// TIA Portal V17 export
// export: Created 2025-06-20T11:17:40.9768226Z, ExportSetting WithDefaults, DisplayName Totally Integrated Automation Portal, DisplayVersion V17 Update 8, DisplayName TIA Portal Openness, DisplayVersion V17 Update 8, DisplayName TIA Portal Version Control Interface, DisplayVersion V17, DisplayName SINAMICS Startdrive Advanced, DisplayVersion V17 SP2, DisplayName SINAMICS Startdrive G110M, G120, G120C, G120D, G120P, G115D, DisplayVersion V17 SP2, DisplayName SINAMICS Startdrive G130, G150, S120, S150, SINAMICS MV, S210, DisplayVersion V17 SP2, DisplayName STEP 7 Professional, DisplayVersion V17 Update 8, DisplayName SINUMERIK ONE STEP 7 Toolbox, DisplayVersion V17 Update 12, DisplayName SINUMERIK ONE PLC Basic Program Plus, DisplayVersion V17 Update 12, DisplayName SINUMERIK 840D sl STEP 7 Toolbox, DisplayVersion V17 Update 12, DisplayName STEP 7 Safety, DisplayVersion V17 Update 6, DisplayName WinCC Advanced, DisplayVersion V17 Update 8
FUNCTION "FC16017_METHOD_CALLS_U3_MEAS_STA_MEAS_N" : Void   // FC16017, LAD
{ S7_Optimized_Access := 'FALSE' }
VERSION : 0.1
// stored: AutoNumber false, IsIECCheckEnabled false, SetENOAutomatically false, UDAEnableTagReadback false
   VAR_TEMP
      AUX_WSTRING_PART_ID_MEAS_STA : WString;
      AUX_WCHARS : Array[0..63] of WChar;
      index : Int;
      AUX_ALARMS : Bool;
      STATUS_BLKMOV : Int;   // STATUS BLKMOV
      ZERO : Int;
   END_VAR
   VAR CONSTANT
      VERSIONS_MAJOR : UInt := 2;
      VERSIONS_MINOR : UInt;
      FC_NUMBER : DInt := 16017;
   END_VAR
   VAR_TEMP   // added for the SCL form of the ladder/FBD networks
      _w1 : Bool;
      _w2 : Bool;
   END_VAR
BEGIN

REGION Network 1: ZERO
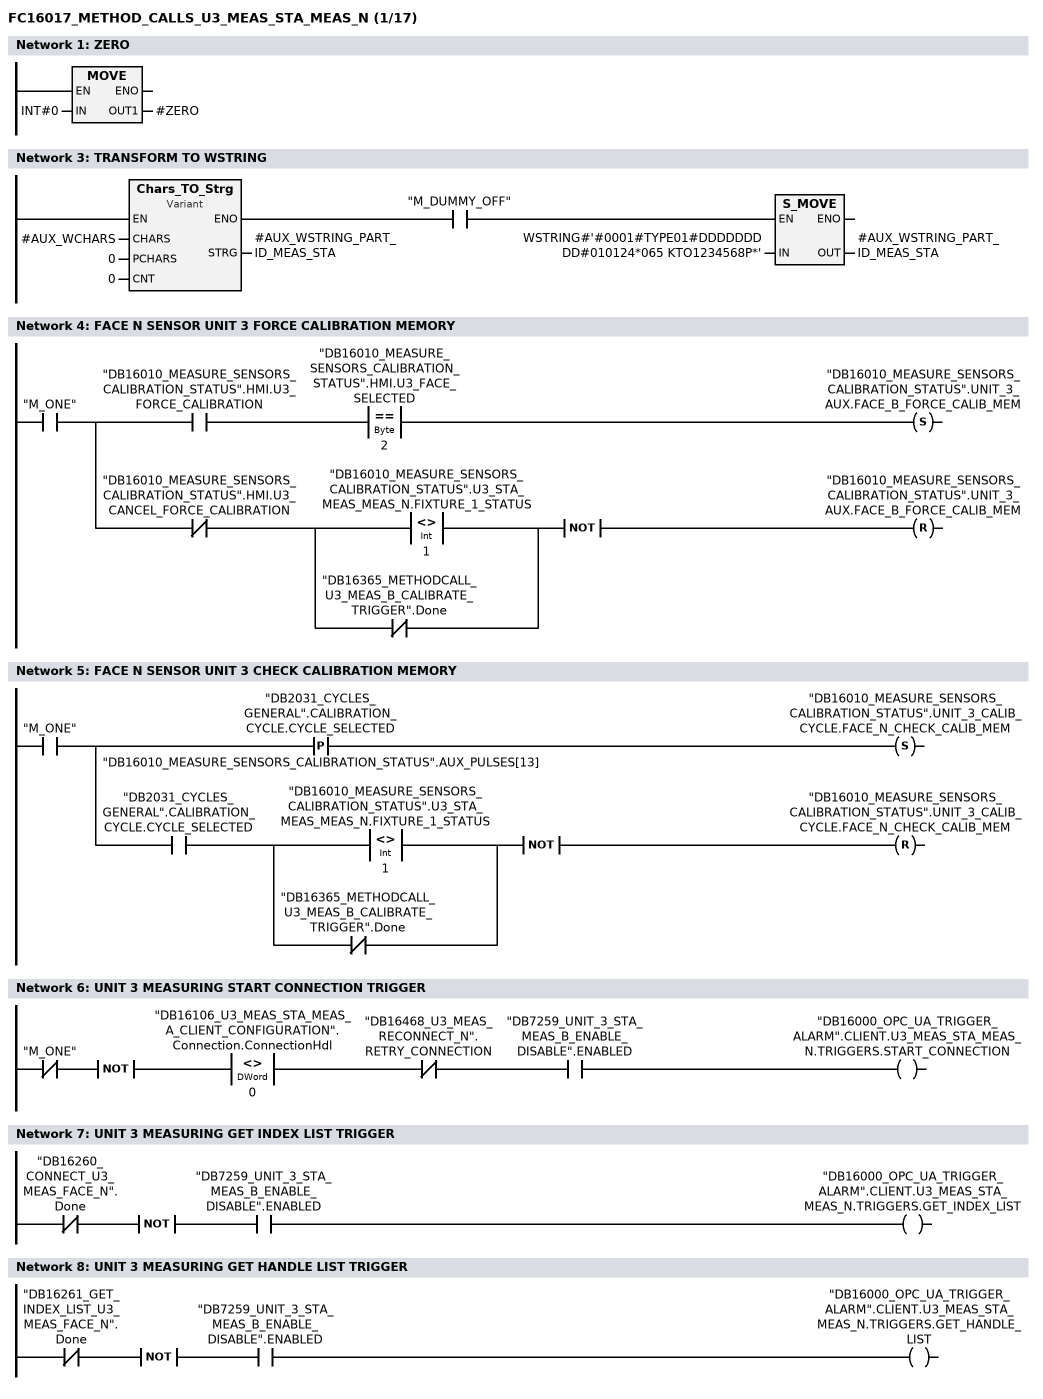
   RUNG wire#powerrail
      { S7_GenerateENO := "TRUE" } Move(in := INT#0, out1 => #ZERO)
   END_RUNG
   // the same network as SCL:
   #ZERO := INT#0;
END_REGION

REGION Network 2 (SCL): TRANSFORM TO WCHARS
   FOR #index := 0 TO 63 DO
       #AUX_WCHARS[#index] := CHAR_TO_WCHAR("DB8000_PART_STATUS".UNIT_3.FIXTURE_1.PART_A.PART_ID[#index]);
   END_FOR;
END_REGION

REGION Network 3: TRANSFORM TO WSTRING
   RUNG wire#powerrail
      { S7_Templates := "[ptr_type := Variant, str_type := WString]" } Chars_TO_Strg(Chars := #AUX_WCHARS, pChars := 0, Cnt := 0, Strg => #AUX_WSTRING_PART_ID_MEAS_STA)
      Contact( "M_DUMMY_OFF" )
      S_Move(in := WSTRING#'#0001#TYPE01#DDDDDDDDD#010124*065 KTO1234568P*', out => #AUX_WSTRING_PART_ID_MEAS_STA)
   END_RUNG
   // the same network as SCL:
   Chars_TO_Strg(Chars := #AUX_WCHARS,
                 pChars := 0,
                 Cnt := 0,
                 Strg => #AUX_WSTRING_PART_ID_MEAS_STA,
                 ENO => #_w1);
   IF #_w1 AND "M_DUMMY_OFF" THEN
       #AUX_WSTRING_PART_ID_MEAS_STA := WSTRING#'#0001#TYPE01#DDDDDDDDD#010124*065 KTO1234568P*';
   END_IF;
END_REGION

REGION Network 4: FACE N SENSOR UNIT 3 FORCE CALIBRATION MEMORY
   RUNG wire#powerrail
      Contact( "M_ONE" )
      wire#w1
      Contact( "DB16010_MEASURE_SENSORS_CALIBRATION_STATUS".HMI.U3_FORCE_CALIBRATION )
      { S7_Templates := "SrcType := Byte" } EQ_Contact(in1 := "DB16010_MEASURE_SENSORS_CALIBRATION_STATUS".HMI.U3_FACE_SELECTED, in2 := 2)
      S_Coil( "DB16010_MEASURE_SENSORS_CALIBRATION_STATUS".UNIT_3_AUX.FACE_B_FORCE_CALIB_MEM )
   END_RUNG
   RUNG wire#w1
      I_Contact( "DB16010_MEASURE_SENSORS_CALIBRATION_STATUS".HMI.U3_CANCEL_FORCE_CALIBRATION )
      wire#w2
      { S7_Templates := "SrcType := Int" } NE_Contact(in1 := "DB16010_MEASURE_SENSORS_CALIBRATION_STATUS".U3_STA_MEAS_MEAS_N.FIXTURE_1_STATUS, in2 := 1)
      wire#w3
      Not()
      R_Coil( "DB16010_MEASURE_SENSORS_CALIBRATION_STATUS".UNIT_3_AUX.FACE_B_FORCE_CALIB_MEM )
   END_RUNG
   RUNG wire#w2
      I_Contact( "DB16365_METHODCALL_U3_MEAS_B_CALIBRATE_TRIGGER".Done )
   END_RUNG wire#w3
   // the same network as SCL:
   IF "M_ONE" AND "DB16010_MEASURE_SENSORS_CALIBRATION_STATUS".HMI.U3_FORCE_CALIBRATION AND ("DB16010_MEASURE_SENSORS_CALIBRATION_STATUS".HMI.U3_FACE_SELECTED = 2) THEN
       "DB16010_MEASURE_SENSORS_CALIBRATION_STATUS".UNIT_3_AUX.FACE_B_FORCE_CALIB_MEM := TRUE;
   END_IF;
   IF NOT ("M_ONE" AND NOT "DB16010_MEASURE_SENSORS_CALIBRATION_STATUS".HMI.U3_CANCEL_FORCE_CALIBRATION AND (("DB16010_MEASURE_SENSORS_CALIBRATION_STATUS".U3_STA_MEAS_MEAS_N.FIXTURE_1_STATUS <> 1) OR NOT "DB16365_METHODCALL_U3_MEAS_B_CALIBRATE_TRIGGER".Done)) THEN
       "DB16010_MEASURE_SENSORS_CALIBRATION_STATUS".UNIT_3_AUX.FACE_B_FORCE_CALIB_MEM := FALSE;
   END_IF;
END_REGION

REGION Network 5: FACE N SENSOR UNIT 3 CHECK CALIBRATION MEMORY
   RUNG wire#powerrail
      Contact( "M_ONE" )
      wire#w1
      P_Contact(operand := "DB2031_CYCLES_GENERAL".CALIBRATION_CYCLE.CYCLE_SELECTED, bit := "DB16010_MEASURE_SENSORS_CALIBRATION_STATUS".AUX_PULSES[13])
      S_Coil( "DB16010_MEASURE_SENSORS_CALIBRATION_STATUS".UNIT_3_CALIB_CYCLE.FACE_N_CHECK_CALIB_MEM )
   END_RUNG
   RUNG wire#w1
      Contact( "DB2031_CYCLES_GENERAL".CALIBRATION_CYCLE.CYCLE_SELECTED )
      wire#w2
      { S7_Templates := "SrcType := Int" } NE_Contact(in1 := "DB16010_MEASURE_SENSORS_CALIBRATION_STATUS".U3_STA_MEAS_MEAS_N.FIXTURE_1_STATUS, in2 := 1)
      wire#w3
      Not()
      R_Coil( "DB16010_MEASURE_SENSORS_CALIBRATION_STATUS".UNIT_3_CALIB_CYCLE.FACE_N_CHECK_CALIB_MEM )
   END_RUNG
   RUNG wire#w2
      I_Contact( "DB16365_METHODCALL_U3_MEAS_B_CALIBRATE_TRIGGER".Done )
   END_RUNG wire#w3
   // the same network as SCL:
   #_w1 := "M_ONE" AND "DB2031_CYCLES_GENERAL".CALIBRATION_CYCLE.CYCLE_SELECTED AND NOT "DB16010_MEASURE_SENSORS_CALIBRATION_STATUS".AUX_PULSES[13];   // rising edge of "DB2031_CYCLES_GENERAL".CALIBRATION_CYCLE.CYCLE_SELECTED
   "DB16010_MEASURE_SENSORS_CALIBRATION_STATUS".AUX_PULSES[13] := "DB2031_CYCLES_GENERAL".CALIBRATION_CYCLE.CYCLE_SELECTED;
   IF #_w1 THEN
       "DB16010_MEASURE_SENSORS_CALIBRATION_STATUS".UNIT_3_CALIB_CYCLE.FACE_N_CHECK_CALIB_MEM := TRUE;
   END_IF;
   IF NOT ("M_ONE" AND "DB2031_CYCLES_GENERAL".CALIBRATION_CYCLE.CYCLE_SELECTED AND (("DB16010_MEASURE_SENSORS_CALIBRATION_STATUS".U3_STA_MEAS_MEAS_N.FIXTURE_1_STATUS <> 1) OR NOT "DB16365_METHODCALL_U3_MEAS_B_CALIBRATE_TRIGGER".Done)) THEN
       "DB16010_MEASURE_SENSORS_CALIBRATION_STATUS".UNIT_3_CALIB_CYCLE.FACE_N_CHECK_CALIB_MEM := FALSE;
   END_IF;
END_REGION

REGION Network 6: UNIT 3 MEASURING START CONNECTION TRIGGER
   RUNG wire#powerrail
      I_Contact( "M_ONE" )
      Not()
      { S7_Templates := "SrcType := DWord" } NE_Contact(in1 := "DB16106_U3_MEAS_STA_MEAS_A_CLIENT_CONFIGURATION".Connection.ConnectionHdl, in2 := 0)
      I_Contact( "DB16468_U3_MEAS_RECONNECT_N".RETRY_CONNECTION )
      Contact( "DB7259_UNIT_3_STA_MEAS_B_ENABLE_DISABLE".ENABLED )
      Coil( "DB16000_OPC_UA_TRIGGER_ALARM".CLIENT.U3_MEAS_STA_MEAS_N.TRIGGERS.START_CONNECTION )
   END_RUNG
   // the same network as SCL:
   "DB16000_OPC_UA_TRIGGER_ALARM".CLIENT.U3_MEAS_STA_MEAS_N.TRIGGERS.START_CONNECTION := NOT (NOT "M_ONE") AND ("DB16106_U3_MEAS_STA_MEAS_A_CLIENT_CONFIGURATION".Connection.ConnectionHdl <> 0) AND NOT "DB16468_U3_MEAS_RECONNECT_N".RETRY_CONNECTION AND "DB7259_UNIT_3_STA_MEAS_B_ENABLE_DISABLE".ENABLED;
END_REGION

REGION Network 7: UNIT 3 MEASURING GET INDEX LIST TRIGGER
   RUNG wire#powerrail
      I_Contact( "DB16260_CONNECT_U3_MEAS_FACE_N".Done )
      Not()
      Contact( "DB7259_UNIT_3_STA_MEAS_B_ENABLE_DISABLE".ENABLED )
      Coil( "DB16000_OPC_UA_TRIGGER_ALARM".CLIENT.U3_MEAS_STA_MEAS_N.TRIGGERS.GET_INDEX_LIST )
   END_RUNG
   // the same network as SCL:
   "DB16000_OPC_UA_TRIGGER_ALARM".CLIENT.U3_MEAS_STA_MEAS_N.TRIGGERS.GET_INDEX_LIST := NOT (NOT "DB16260_CONNECT_U3_MEAS_FACE_N".Done) AND "DB7259_UNIT_3_STA_MEAS_B_ENABLE_DISABLE".ENABLED;
END_REGION

REGION Network 8: UNIT 3 MEASURING GET HANDLE LIST TRIGGER
   RUNG wire#powerrail
      I_Contact( "DB16261_GET_INDEX_LIST_U3_MEAS_FACE_N".Done )
      Not()
      Contact( "DB7259_UNIT_3_STA_MEAS_B_ENABLE_DISABLE".ENABLED )
      Coil( "DB16000_OPC_UA_TRIGGER_ALARM".CLIENT.U3_MEAS_STA_MEAS_N.TRIGGERS.GET_HANDLE_LIST )
   END_RUNG
   // the same network as SCL:
   "DB16000_OPC_UA_TRIGGER_ALARM".CLIENT.U3_MEAS_STA_MEAS_N.TRIGGERS.GET_HANDLE_LIST := NOT (NOT "DB16261_GET_INDEX_LIST_U3_MEAS_FACE_N".Done) AND "DB7259_UNIT_3_STA_MEAS_B_ENABLE_DISABLE".ENABLED;
END_REGION

REGION Network 9: UNIT 3 MEASURING GET METHOD LIST TRIGGER
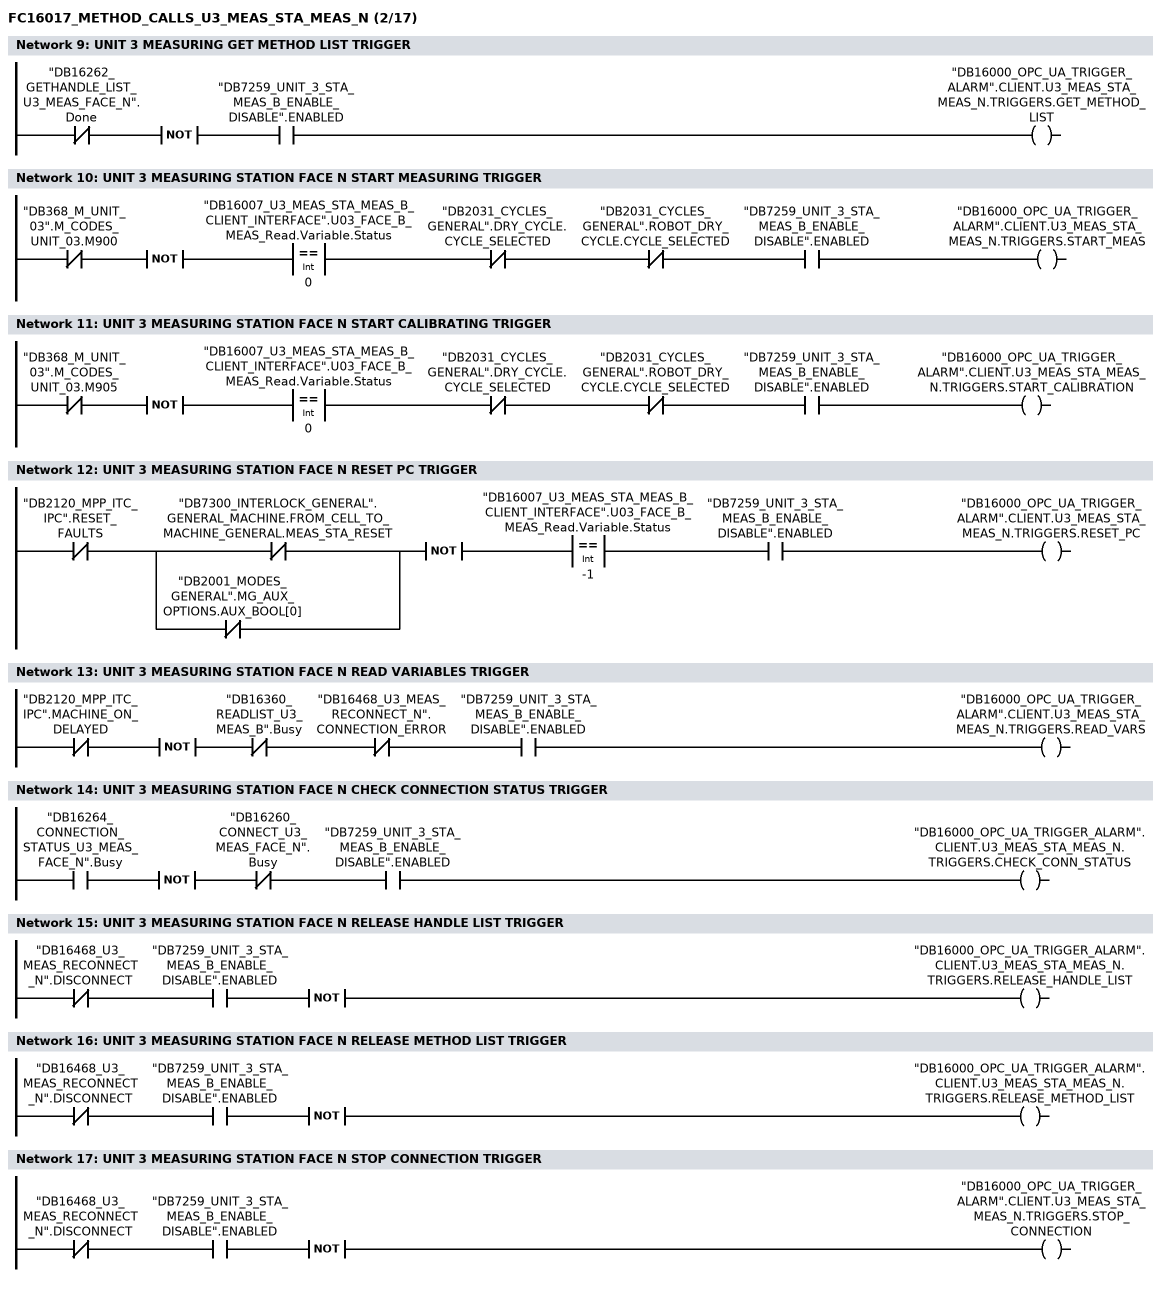
   RUNG wire#powerrail
      I_Contact( "DB16262_GETHANDLE_LIST_U3_MEAS_FACE_N".Done )
      Not()
      Contact( "DB7259_UNIT_3_STA_MEAS_B_ENABLE_DISABLE".ENABLED )
      Coil( "DB16000_OPC_UA_TRIGGER_ALARM".CLIENT.U3_MEAS_STA_MEAS_N.TRIGGERS.GET_METHOD_LIST )
   END_RUNG
   // the same network as SCL:
   "DB16000_OPC_UA_TRIGGER_ALARM".CLIENT.U3_MEAS_STA_MEAS_N.TRIGGERS.GET_METHOD_LIST := NOT (NOT "DB16262_GETHANDLE_LIST_U3_MEAS_FACE_N".Done) AND "DB7259_UNIT_3_STA_MEAS_B_ENABLE_DISABLE".ENABLED;
END_REGION

REGION Network 10: UNIT 3 MEASURING STATION FACE N START MEASURING TRIGGER
   RUNG wire#powerrail
      I_Contact( "DB368_M_UNIT_03".M_CODES_UNIT_03.M900 )
      Not()
      { S7_Templates := "SrcType := Int" } EQ_Contact(in1 := "DB16007_U3_MEAS_STA_MEAS_B_CLIENT_INTERFACE".U03_FACE_B_MEAS_Read.Variable.Status, in2 := 0)
      I_Contact( "DB2031_CYCLES_GENERAL".DRY_CYCLE.CYCLE_SELECTED )
      I_Contact( "DB2031_CYCLES_GENERAL".ROBOT_DRY_CYCLE.CYCLE_SELECTED )
      Contact( "DB7259_UNIT_3_STA_MEAS_B_ENABLE_DISABLE".ENABLED )
      Coil( "DB16000_OPC_UA_TRIGGER_ALARM".CLIENT.U3_MEAS_STA_MEAS_N.TRIGGERS.START_MEAS )
   END_RUNG
   // the same network as SCL:
   "DB16000_OPC_UA_TRIGGER_ALARM".CLIENT.U3_MEAS_STA_MEAS_N.TRIGGERS.START_MEAS := NOT (NOT "DB368_M_UNIT_03".M_CODES_UNIT_03.M900) AND ("DB16007_U3_MEAS_STA_MEAS_B_CLIENT_INTERFACE".U03_FACE_B_MEAS_Read.Variable.Status = 0) AND NOT "DB2031_CYCLES_GENERAL".DRY_CYCLE.CYCLE_SELECTED AND NOT "DB2031_CYCLES_GENERAL".ROBOT_DRY_CYCLE.CYCLE_SELECTED AND "DB7259_UNIT_3_STA_MEAS_B_ENABLE_DISABLE".ENABLED;
END_REGION

REGION Network 11: UNIT 3 MEASURING STATION FACE N START CALIBRATING TRIGGER
   RUNG wire#powerrail
      I_Contact( "DB368_M_UNIT_03".M_CODES_UNIT_03.M905 )
      Not()
      { S7_Templates := "SrcType := Int" } EQ_Contact(in1 := "DB16007_U3_MEAS_STA_MEAS_B_CLIENT_INTERFACE".U03_FACE_B_MEAS_Read.Variable.Status, in2 := 0)
      I_Contact( "DB2031_CYCLES_GENERAL".DRY_CYCLE.CYCLE_SELECTED )
      I_Contact( "DB2031_CYCLES_GENERAL".ROBOT_DRY_CYCLE.CYCLE_SELECTED )
      Contact( "DB7259_UNIT_3_STA_MEAS_B_ENABLE_DISABLE".ENABLED )
      Coil( "DB16000_OPC_UA_TRIGGER_ALARM".CLIENT.U3_MEAS_STA_MEAS_N.TRIGGERS.START_CALIBRATION )
   END_RUNG
   // the same network as SCL:
   "DB16000_OPC_UA_TRIGGER_ALARM".CLIENT.U3_MEAS_STA_MEAS_N.TRIGGERS.START_CALIBRATION := NOT (NOT "DB368_M_UNIT_03".M_CODES_UNIT_03.M905) AND ("DB16007_U3_MEAS_STA_MEAS_B_CLIENT_INTERFACE".U03_FACE_B_MEAS_Read.Variable.Status = 0) AND NOT "DB2031_CYCLES_GENERAL".DRY_CYCLE.CYCLE_SELECTED AND NOT "DB2031_CYCLES_GENERAL".ROBOT_DRY_CYCLE.CYCLE_SELECTED AND "DB7259_UNIT_3_STA_MEAS_B_ENABLE_DISABLE".ENABLED;
END_REGION

REGION Network 12: UNIT 3 MEASURING STATION FACE N RESET PC TRIGGER
   RUNG wire#powerrail
      I_Contact( "DB2120_MPP_ITC_IPC".RESET_FAULTS )
      wire#w1
      I_Contact( "DB7300_INTERLOCK_GENERAL".GENERAL_MACHINE.FROM_CELL_TO_MACHINE_GENERAL.MEAS_STA_RESET )
      wire#w2
      Not()
      { S7_Templates := "SrcType := Int" } EQ_Contact(in1 := "DB16007_U3_MEAS_STA_MEAS_B_CLIENT_INTERFACE".U03_FACE_B_MEAS_Read.Variable.Status, in2 := -1)
      Contact( "DB7259_UNIT_3_STA_MEAS_B_ENABLE_DISABLE".ENABLED )
      Coil( "DB16000_OPC_UA_TRIGGER_ALARM".CLIENT.U3_MEAS_STA_MEAS_N.TRIGGERS.RESET_PC )
   END_RUNG
   RUNG wire#w1
      I_Contact( "DB2001_MODES_GENERAL".MG_AUX_OPTIONS.AUX_BOOL[0] )
   END_RUNG wire#w2
   // the same network as SCL:
   "DB16000_OPC_UA_TRIGGER_ALARM".CLIENT.U3_MEAS_STA_MEAS_N.TRIGGERS.RESET_PC := NOT (NOT "DB2120_MPP_ITC_IPC".RESET_FAULTS AND (NOT "DB7300_INTERLOCK_GENERAL".GENERAL_MACHINE.FROM_CELL_TO_MACHINE_GENERAL.MEAS_STA_RESET OR NOT "DB2001_MODES_GENERAL".MG_AUX_OPTIONS.AUX_BOOL[0])) AND ("DB16007_U3_MEAS_STA_MEAS_B_CLIENT_INTERFACE".U03_FACE_B_MEAS_Read.Variable.Status = (-1)) AND "DB7259_UNIT_3_STA_MEAS_B_ENABLE_DISABLE".ENABLED;
END_REGION

REGION Network 13: UNIT 3 MEASURING STATION FACE N READ VARIABLES TRIGGER
   RUNG wire#powerrail
      I_Contact( "DB2120_MPP_ITC_IPC".MACHINE_ON_DELAYED )
      Not()
      I_Contact( "DB16360_READLIST_U3_MEAS_B".Busy )
      I_Contact( "DB16468_U3_MEAS_RECONNECT_N".CONNECTION_ERROR )
      Contact( "DB7259_UNIT_3_STA_MEAS_B_ENABLE_DISABLE".ENABLED )
      Coil( "DB16000_OPC_UA_TRIGGER_ALARM".CLIENT.U3_MEAS_STA_MEAS_N.TRIGGERS.READ_VARS )
   END_RUNG
   // the same network as SCL:
   "DB16000_OPC_UA_TRIGGER_ALARM".CLIENT.U3_MEAS_STA_MEAS_N.TRIGGERS.READ_VARS := NOT (NOT "DB2120_MPP_ITC_IPC".MACHINE_ON_DELAYED) AND NOT "DB16360_READLIST_U3_MEAS_B".Busy AND NOT "DB16468_U3_MEAS_RECONNECT_N".CONNECTION_ERROR AND "DB7259_UNIT_3_STA_MEAS_B_ENABLE_DISABLE".ENABLED;
END_REGION

REGION Network 14: UNIT 3 MEASURING STATION FACE N CHECK CONNECTION STATUS TRIGGER
   RUNG wire#powerrail
      Contact( "DB16264_CONNECTION_STATUS_U3_MEAS_FACE_N".Busy )
      Not()
      I_Contact( "DB16260_CONNECT_U3_MEAS_FACE_N".Busy )
      Contact( "DB7259_UNIT_3_STA_MEAS_B_ENABLE_DISABLE".ENABLED )
      Coil( "DB16000_OPC_UA_TRIGGER_ALARM".CLIENT.U3_MEAS_STA_MEAS_N.TRIGGERS.CHECK_CONN_STATUS )
   END_RUNG
   // the same network as SCL:
   "DB16000_OPC_UA_TRIGGER_ALARM".CLIENT.U3_MEAS_STA_MEAS_N.TRIGGERS.CHECK_CONN_STATUS := NOT "DB16264_CONNECTION_STATUS_U3_MEAS_FACE_N".Busy AND NOT "DB16260_CONNECT_U3_MEAS_FACE_N".Busy AND "DB7259_UNIT_3_STA_MEAS_B_ENABLE_DISABLE".ENABLED;
END_REGION

REGION Network 15: UNIT 3 MEASURING STATION FACE N RELEASE HANDLE LIST TRIGGER
   RUNG wire#powerrail
      I_Contact( "DB16468_U3_MEAS_RECONNECT_N".DISCONNECT )
      Contact( "DB7259_UNIT_3_STA_MEAS_B_ENABLE_DISABLE".ENABLED )
      Not()
      Coil( "DB16000_OPC_UA_TRIGGER_ALARM".CLIENT.U3_MEAS_STA_MEAS_N.TRIGGERS.RELEASE_HANDLE_LIST )
   END_RUNG
   // the same network as SCL:
   "DB16000_OPC_UA_TRIGGER_ALARM".CLIENT.U3_MEAS_STA_MEAS_N.TRIGGERS.RELEASE_HANDLE_LIST := NOT (NOT "DB16468_U3_MEAS_RECONNECT_N".DISCONNECT AND "DB7259_UNIT_3_STA_MEAS_B_ENABLE_DISABLE".ENABLED);
END_REGION

REGION Network 16: UNIT 3 MEASURING STATION FACE N RELEASE METHOD LIST TRIGGER
   RUNG wire#powerrail
      I_Contact( "DB16468_U3_MEAS_RECONNECT_N".DISCONNECT )
      Contact( "DB7259_UNIT_3_STA_MEAS_B_ENABLE_DISABLE".ENABLED )
      Not()
      Coil( "DB16000_OPC_UA_TRIGGER_ALARM".CLIENT.U3_MEAS_STA_MEAS_N.TRIGGERS.RELEASE_METHOD_LIST )
   END_RUNG
   // the same network as SCL:
   "DB16000_OPC_UA_TRIGGER_ALARM".CLIENT.U3_MEAS_STA_MEAS_N.TRIGGERS.RELEASE_METHOD_LIST := NOT (NOT "DB16468_U3_MEAS_RECONNECT_N".DISCONNECT AND "DB7259_UNIT_3_STA_MEAS_B_ENABLE_DISABLE".ENABLED);
END_REGION

REGION Network 17: UNIT 3 MEASURING STATION FACE N STOP CONNECTION TRIGGER
   RUNG wire#powerrail
      I_Contact( "DB16468_U3_MEAS_RECONNECT_N".DISCONNECT )
      Contact( "DB7259_UNIT_3_STA_MEAS_B_ENABLE_DISABLE".ENABLED )
      Not()
      Coil( "DB16000_OPC_UA_TRIGGER_ALARM".CLIENT.U3_MEAS_STA_MEAS_N.TRIGGERS.STOP_CONNECTION )
   END_RUNG
   // the same network as SCL:
   "DB16000_OPC_UA_TRIGGER_ALARM".CLIENT.U3_MEAS_STA_MEAS_N.TRIGGERS.STOP_CONNECTION := NOT (NOT "DB16468_U3_MEAS_RECONNECT_N".DISCONNECT AND "DB7259_UNIT_3_STA_MEAS_B_ENABLE_DISABLE".ENABLED);
END_REGION

REGION Network 18: UNIT 3 MEASURING STATION FACE N START CALIBRATING ARGUMENTS
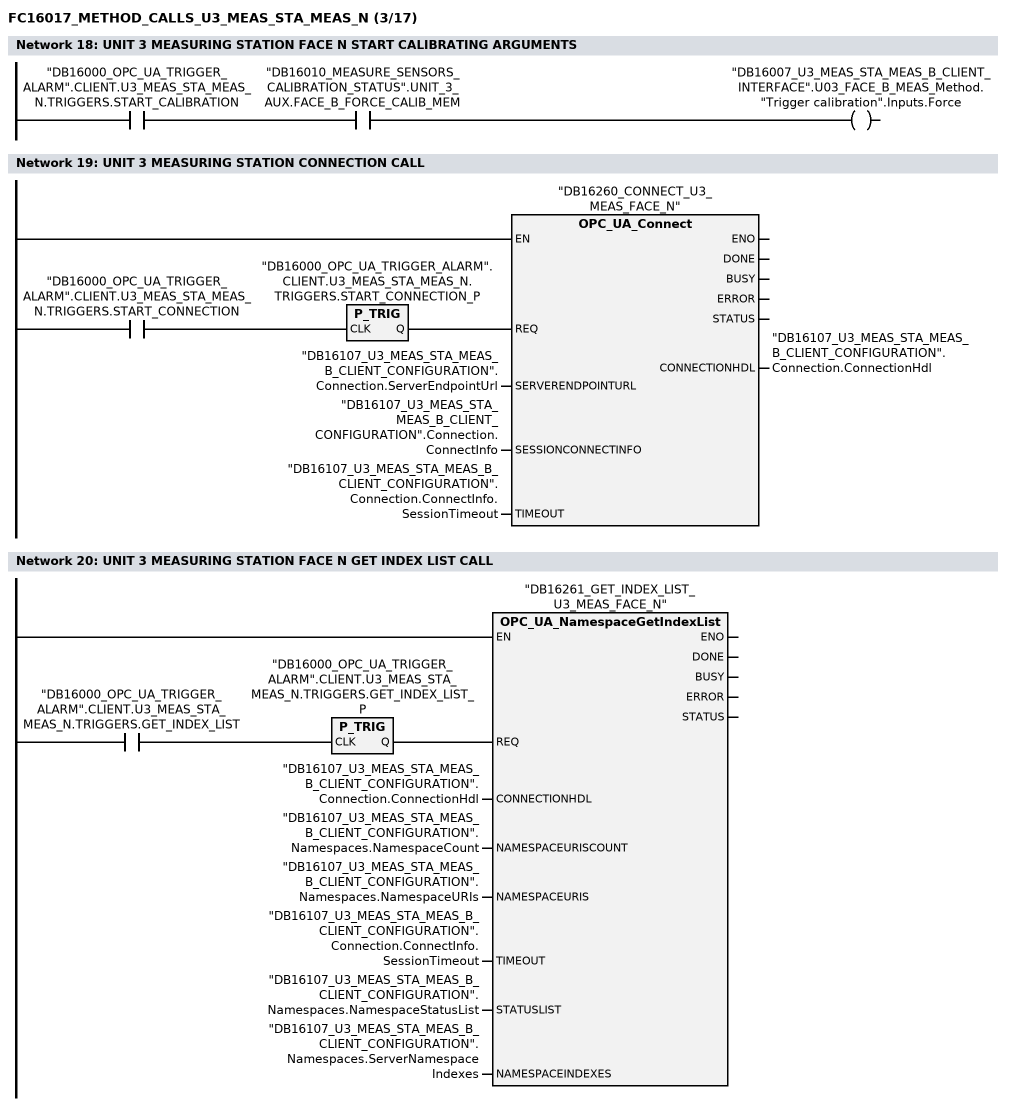
   RUNG wire#powerrail
      Contact( "DB16000_OPC_UA_TRIGGER_ALARM".CLIENT.U3_MEAS_STA_MEAS_N.TRIGGERS.START_CALIBRATION )
      Contact( "DB16010_MEASURE_SENSORS_CALIBRATION_STATUS".UNIT_3_AUX.FACE_B_FORCE_CALIB_MEM )
      Coil( "DB16007_U3_MEAS_STA_MEAS_B_CLIENT_INTERFACE".U03_FACE_B_MEAS_Method."Trigger calibration".Inputs.Force )
   END_RUNG
   // the same network as SCL:
   "DB16007_U3_MEAS_STA_MEAS_B_CLIENT_INTERFACE".U03_FACE_B_MEAS_Method."Trigger calibration".Inputs.Force := "DB16000_OPC_UA_TRIGGER_ALARM".CLIENT.U3_MEAS_STA_MEAS_N.TRIGGERS.START_CALIBRATION AND "DB16010_MEASURE_SENSORS_CALIBRATION_STATUS".UNIT_3_AUX.FACE_B_FORCE_CALIB_MEM;
END_REGION

REGION Network 19: UNIT 3 MEASURING STATION CONNECTION CALL
   RUNG wire#powerrail
      "DB16260_CONNECT_U3_MEAS_FACE_N".OPC_UA_Connect(REQ := wire#w1, ServerEndpointUrl := "DB16107_U3_MEAS_STA_MEAS_B_CLIENT_CONFIGURATION".Connection.ServerEndpointUrl, SessionConnectInfo := "DB16107_U3_MEAS_STA_MEAS_B_CLIENT_CONFIGURATION".Connection.ConnectInfo, Timeout := "DB16107_U3_MEAS_STA_MEAS_B_CLIENT_CONFIGURATION".Connection.ConnectInfo.SessionTimeout, Done =>, Busy =>, Error =>, Status =>, ConnectionHdl => "DB16107_U3_MEAS_STA_MEAS_B_CLIENT_CONFIGURATION".Connection.ConnectionHdl)
   END_RUNG
   RUNG wire#powerrail
      Contact( "DB16000_OPC_UA_TRIGGER_ALARM".CLIENT.U3_MEAS_STA_MEAS_N.TRIGGERS.START_CONNECTION )
      P_Trig( "DB16000_OPC_UA_TRIGGER_ALARM".CLIENT.U3_MEAS_STA_MEAS_N.TRIGGERS.START_CONNECTION_P )
   END_RUNG wire#w1
   // the same network as SCL:
   #_w1 := "DB16000_OPC_UA_TRIGGER_ALARM".CLIENT.U3_MEAS_STA_MEAS_N.TRIGGERS.START_CONNECTION AND NOT "DB16000_OPC_UA_TRIGGER_ALARM".CLIENT.U3_MEAS_STA_MEAS_N.TRIGGERS.START_CONNECTION_P;   // rising edge
   "DB16000_OPC_UA_TRIGGER_ALARM".CLIENT.U3_MEAS_STA_MEAS_N.TRIGGERS.START_CONNECTION_P := "DB16000_OPC_UA_TRIGGER_ALARM".CLIENT.U3_MEAS_STA_MEAS_N.TRIGGERS.START_CONNECTION;
   "DB16260_CONNECT_U3_MEAS_FACE_N"(REQ := #_w1,   // OPC_UA_Connect
                           ServerEndpointUrl := "DB16107_U3_MEAS_STA_MEAS_B_CLIENT_CONFIGURATION".Connection.ServerEndpointUrl,
                           SessionConnectInfo := "DB16107_U3_MEAS_STA_MEAS_B_CLIENT_CONFIGURATION".Connection.ConnectInfo,
                           Timeout := "DB16107_U3_MEAS_STA_MEAS_B_CLIENT_CONFIGURATION".Connection.ConnectInfo.SessionTimeout,
                           ConnectionHdl => "DB16107_U3_MEAS_STA_MEAS_B_CLIENT_CONFIGURATION".Connection.ConnectionHdl);
END_REGION

REGION Network 20: UNIT 3 MEASURING STATION FACE N GET INDEX LIST CALL
   RUNG wire#powerrail
      "DB16261_GET_INDEX_LIST_U3_MEAS_FACE_N".OPC_UA_NamespaceGetIndexList(REQ := wire#w1, ConnectionHdl := "DB16107_U3_MEAS_STA_MEAS_B_CLIENT_CONFIGURATION".Connection.ConnectionHdl, NamespaceUrisCount := "DB16107_U3_MEAS_STA_MEAS_B_CLIENT_CONFIGURATION".Namespaces.NamespaceCount, NamespaceUris := "DB16107_U3_MEAS_STA_MEAS_B_CLIENT_CONFIGURATION".Namespaces.NamespaceURIs, Timeout := "DB16107_U3_MEAS_STA_MEAS_B_CLIENT_CONFIGURATION".Connection.ConnectInfo.SessionTimeout, StatusList := "DB16107_U3_MEAS_STA_MEAS_B_CLIENT_CONFIGURATION".Namespaces.NamespaceStatusList, NamespaceIndexes := "DB16107_U3_MEAS_STA_MEAS_B_CLIENT_CONFIGURATION".Namespaces.ServerNamespaceIndexes, Done =>, Busy =>, Error =>, Status =>)
   END_RUNG
   RUNG wire#powerrail
      Contact( "DB16000_OPC_UA_TRIGGER_ALARM".CLIENT.U3_MEAS_STA_MEAS_N.TRIGGERS.GET_INDEX_LIST )
      P_Trig( "DB16000_OPC_UA_TRIGGER_ALARM".CLIENT.U3_MEAS_STA_MEAS_N.TRIGGERS.GET_INDEX_LIST_P )
   END_RUNG wire#w1
   // the same network as SCL:
   #_w1 := "DB16000_OPC_UA_TRIGGER_ALARM".CLIENT.U3_MEAS_STA_MEAS_N.TRIGGERS.GET_INDEX_LIST AND NOT "DB16000_OPC_UA_TRIGGER_ALARM".CLIENT.U3_MEAS_STA_MEAS_N.TRIGGERS.GET_INDEX_LIST_P;   // rising edge
   "DB16000_OPC_UA_TRIGGER_ALARM".CLIENT.U3_MEAS_STA_MEAS_N.TRIGGERS.GET_INDEX_LIST_P := "DB16000_OPC_UA_TRIGGER_ALARM".CLIENT.U3_MEAS_STA_MEAS_N.TRIGGERS.GET_INDEX_LIST;
   "DB16261_GET_INDEX_LIST_U3_MEAS_FACE_N"(REQ := #_w1,   // OPC_UA_NamespaceGetIndexList
                           ConnectionHdl := "DB16107_U3_MEAS_STA_MEAS_B_CLIENT_CONFIGURATION".Connection.ConnectionHdl,
                           NamespaceUrisCount := "DB16107_U3_MEAS_STA_MEAS_B_CLIENT_CONFIGURATION".Namespaces.NamespaceCount,
                           NamespaceUris := "DB16107_U3_MEAS_STA_MEAS_B_CLIENT_CONFIGURATION".Namespaces.NamespaceURIs,
                           Timeout := "DB16107_U3_MEAS_STA_MEAS_B_CLIENT_CONFIGURATION".Connection.ConnectInfo.SessionTimeout,
                           StatusList := "DB16107_U3_MEAS_STA_MEAS_B_CLIENT_CONFIGURATION".Namespaces.NamespaceStatusList,
                           NamespaceIndexes := "DB16107_U3_MEAS_STA_MEAS_B_CLIENT_CONFIGURATION".Namespaces.ServerNamespaceIndexes);
END_REGION

REGION Network 21: UNIT 3 MEASURING STATION FACE N GET HANDLE LIST CALL
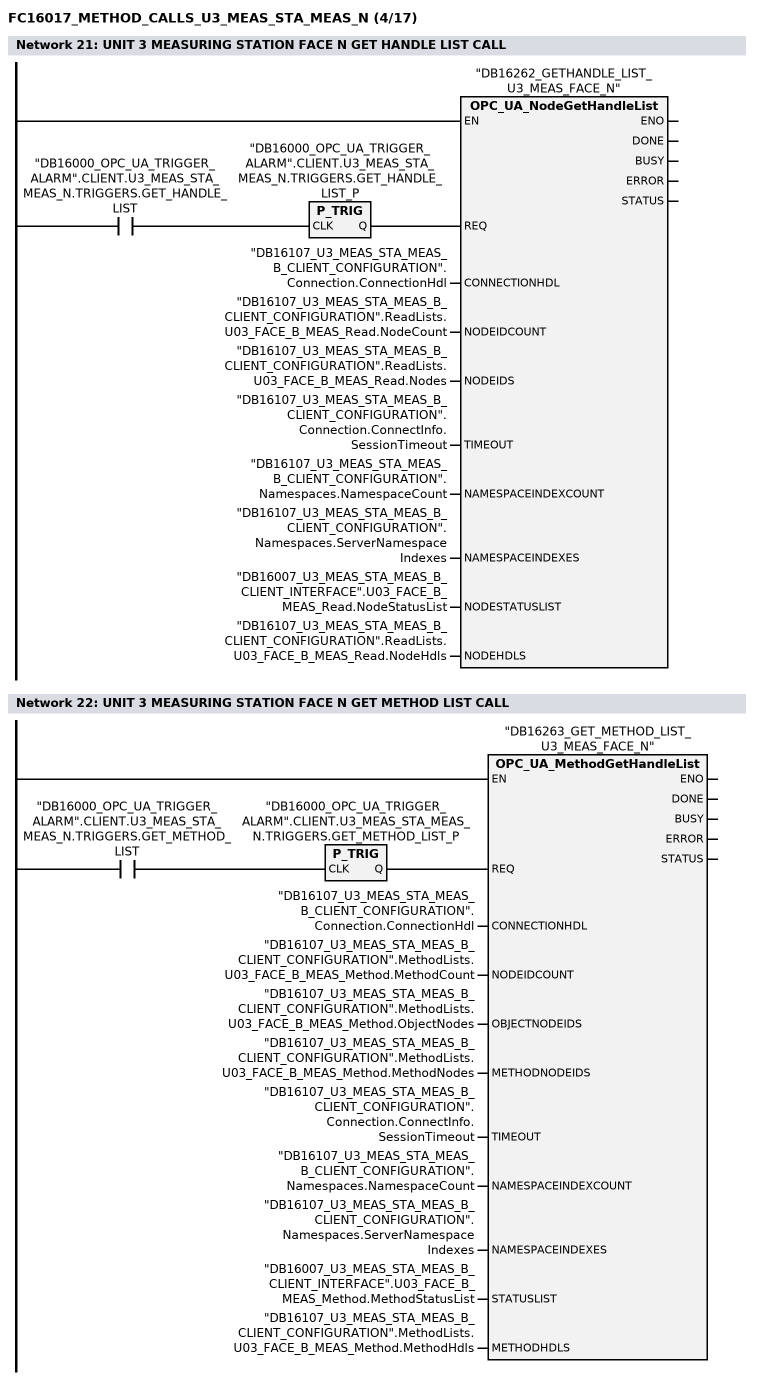
   RUNG wire#powerrail
      "DB16262_GETHANDLE_LIST_U3_MEAS_FACE_N".OPC_UA_NodeGetHandleList(REQ := wire#w1, ConnectionHdl := "DB16107_U3_MEAS_STA_MEAS_B_CLIENT_CONFIGURATION".Connection.ConnectionHdl, NodeIDCount := "DB16107_U3_MEAS_STA_MEAS_B_CLIENT_CONFIGURATION".ReadLists.U03_FACE_B_MEAS_Read.NodeCount, NodeIDs := "DB16107_U3_MEAS_STA_MEAS_B_CLIENT_CONFIGURATION".ReadLists.U03_FACE_B_MEAS_Read.Nodes, Timeout := "DB16107_U3_MEAS_STA_MEAS_B_CLIENT_CONFIGURATION".Connection.ConnectInfo.SessionTimeout, NamespaceIndexCount := "DB16107_U3_MEAS_STA_MEAS_B_CLIENT_CONFIGURATION".Namespaces.NamespaceCount, NamespaceIndexes := "DB16107_U3_MEAS_STA_MEAS_B_CLIENT_CONFIGURATION".Namespaces.ServerNamespaceIndexes, NodeStatusList := "DB16007_U3_MEAS_STA_MEAS_B_CLIENT_INTERFACE".U03_FACE_B_MEAS_Read.NodeStatusList, NodeHdls := "DB16107_U3_MEAS_STA_MEAS_B_CLIENT_CONFIGURATION".ReadLists.U03_FACE_B_MEAS_Read.NodeHdls, Done =>, Busy =>, Error =>, Status =>)
   END_RUNG
   RUNG wire#powerrail
      Contact( "DB16000_OPC_UA_TRIGGER_ALARM".CLIENT.U3_MEAS_STA_MEAS_N.TRIGGERS.GET_HANDLE_LIST )
      P_Trig( "DB16000_OPC_UA_TRIGGER_ALARM".CLIENT.U3_MEAS_STA_MEAS_N.TRIGGERS.GET_HANDLE_LIST_P )
   END_RUNG wire#w1
   // the same network as SCL:
   #_w1 := "DB16000_OPC_UA_TRIGGER_ALARM".CLIENT.U3_MEAS_STA_MEAS_N.TRIGGERS.GET_HANDLE_LIST AND NOT "DB16000_OPC_UA_TRIGGER_ALARM".CLIENT.U3_MEAS_STA_MEAS_N.TRIGGERS.GET_HANDLE_LIST_P;   // rising edge
   "DB16000_OPC_UA_TRIGGER_ALARM".CLIENT.U3_MEAS_STA_MEAS_N.TRIGGERS.GET_HANDLE_LIST_P := "DB16000_OPC_UA_TRIGGER_ALARM".CLIENT.U3_MEAS_STA_MEAS_N.TRIGGERS.GET_HANDLE_LIST;
   "DB16262_GETHANDLE_LIST_U3_MEAS_FACE_N"(REQ := #_w1,   // OPC_UA_NodeGetHandleList
                           ConnectionHdl := "DB16107_U3_MEAS_STA_MEAS_B_CLIENT_CONFIGURATION".Connection.ConnectionHdl,
                           NodeIDCount := "DB16107_U3_MEAS_STA_MEAS_B_CLIENT_CONFIGURATION".ReadLists.U03_FACE_B_MEAS_Read.NodeCount,
                           NodeIDs := "DB16107_U3_MEAS_STA_MEAS_B_CLIENT_CONFIGURATION".ReadLists.U03_FACE_B_MEAS_Read.Nodes,
                           Timeout := "DB16107_U3_MEAS_STA_MEAS_B_CLIENT_CONFIGURATION".Connection.ConnectInfo.SessionTimeout,
                           NamespaceIndexCount := "DB16107_U3_MEAS_STA_MEAS_B_CLIENT_CONFIGURATION".Namespaces.NamespaceCount,
                           NamespaceIndexes := "DB16107_U3_MEAS_STA_MEAS_B_CLIENT_CONFIGURATION".Namespaces.ServerNamespaceIndexes,
                           NodeStatusList := "DB16007_U3_MEAS_STA_MEAS_B_CLIENT_INTERFACE".U03_FACE_B_MEAS_Read.NodeStatusList,
                           NodeHdls := "DB16107_U3_MEAS_STA_MEAS_B_CLIENT_CONFIGURATION".ReadLists.U03_FACE_B_MEAS_Read.NodeHdls);
END_REGION

REGION Network 22: UNIT 3 MEASURING STATION FACE N GET METHOD LIST CALL
   RUNG wire#powerrail
      "DB16263_GET_METHOD_LIST_U3_MEAS_FACE_N".OPC_UA_MethodGetHandleList(REQ := wire#w1, ConnectionHdl := "DB16107_U3_MEAS_STA_MEAS_B_CLIENT_CONFIGURATION".Connection.ConnectionHdl, NodeIDCount := "DB16107_U3_MEAS_STA_MEAS_B_CLIENT_CONFIGURATION".MethodLists.U03_FACE_B_MEAS_Method.MethodCount, ObjectNodeIDs := "DB16107_U3_MEAS_STA_MEAS_B_CLIENT_CONFIGURATION".MethodLists.U03_FACE_B_MEAS_Method.ObjectNodes, MethodNodeIDs := "DB16107_U3_MEAS_STA_MEAS_B_CLIENT_CONFIGURATION".MethodLists.U03_FACE_B_MEAS_Method.MethodNodes, Timeout := "DB16107_U3_MEAS_STA_MEAS_B_CLIENT_CONFIGURATION".Connection.ConnectInfo.SessionTimeout, NamespaceIndexCount := "DB16107_U3_MEAS_STA_MEAS_B_CLIENT_CONFIGURATION".Namespaces.NamespaceCount, NamespaceIndexes := "DB16107_U3_MEAS_STA_MEAS_B_CLIENT_CONFIGURATION".Namespaces.ServerNamespaceIndexes, StatusList := "DB16007_U3_MEAS_STA_MEAS_B_CLIENT_INTERFACE".U03_FACE_B_MEAS_Method.MethodStatusList, MethodHdls := "DB16107_U3_MEAS_STA_MEAS_B_CLIENT_CONFIGURATION".MethodLists.U03_FACE_B_MEAS_Method.MethodHdls, Done =>, Busy =>, Error =>, Status =>)
   END_RUNG
   RUNG wire#powerrail
      Contact( "DB16000_OPC_UA_TRIGGER_ALARM".CLIENT.U3_MEAS_STA_MEAS_N.TRIGGERS.GET_METHOD_LIST )
      P_Trig( "DB16000_OPC_UA_TRIGGER_ALARM".CLIENT.U3_MEAS_STA_MEAS_N.TRIGGERS.GET_METHOD_LIST_P )
   END_RUNG wire#w1
   // the same network as SCL:
   #_w1 := "DB16000_OPC_UA_TRIGGER_ALARM".CLIENT.U3_MEAS_STA_MEAS_N.TRIGGERS.GET_METHOD_LIST AND NOT "DB16000_OPC_UA_TRIGGER_ALARM".CLIENT.U3_MEAS_STA_MEAS_N.TRIGGERS.GET_METHOD_LIST_P;   // rising edge
   "DB16000_OPC_UA_TRIGGER_ALARM".CLIENT.U3_MEAS_STA_MEAS_N.TRIGGERS.GET_METHOD_LIST_P := "DB16000_OPC_UA_TRIGGER_ALARM".CLIENT.U3_MEAS_STA_MEAS_N.TRIGGERS.GET_METHOD_LIST;
   "DB16263_GET_METHOD_LIST_U3_MEAS_FACE_N"(REQ := #_w1,   // OPC_UA_MethodGetHandleList
                           ConnectionHdl := "DB16107_U3_MEAS_STA_MEAS_B_CLIENT_CONFIGURATION".Connection.ConnectionHdl,
                           NodeIDCount := "DB16107_U3_MEAS_STA_MEAS_B_CLIENT_CONFIGURATION".MethodLists.U03_FACE_B_MEAS_Method.MethodCount,
                           ObjectNodeIDs := "DB16107_U3_MEAS_STA_MEAS_B_CLIENT_CONFIGURATION".MethodLists.U03_FACE_B_MEAS_Method.ObjectNodes,
                           MethodNodeIDs := "DB16107_U3_MEAS_STA_MEAS_B_CLIENT_CONFIGURATION".MethodLists.U03_FACE_B_MEAS_Method.MethodNodes,
                           Timeout := "DB16107_U3_MEAS_STA_MEAS_B_CLIENT_CONFIGURATION".Connection.ConnectInfo.SessionTimeout,
                           NamespaceIndexCount := "DB16107_U3_MEAS_STA_MEAS_B_CLIENT_CONFIGURATION".Namespaces.NamespaceCount,
                           NamespaceIndexes := "DB16107_U3_MEAS_STA_MEAS_B_CLIENT_CONFIGURATION".Namespaces.ServerNamespaceIndexes,
                           StatusList := "DB16007_U3_MEAS_STA_MEAS_B_CLIENT_INTERFACE".U03_FACE_B_MEAS_Method.MethodStatusList,
                           MethodHdls := "DB16107_U3_MEAS_STA_MEAS_B_CLIENT_CONFIGURATION".MethodLists.U03_FACE_B_MEAS_Method.MethodHdls);
END_REGION

REGION Network 23: UNIT 3 MEASURING STATION FACE N START MEASURING TRIGGER CALL
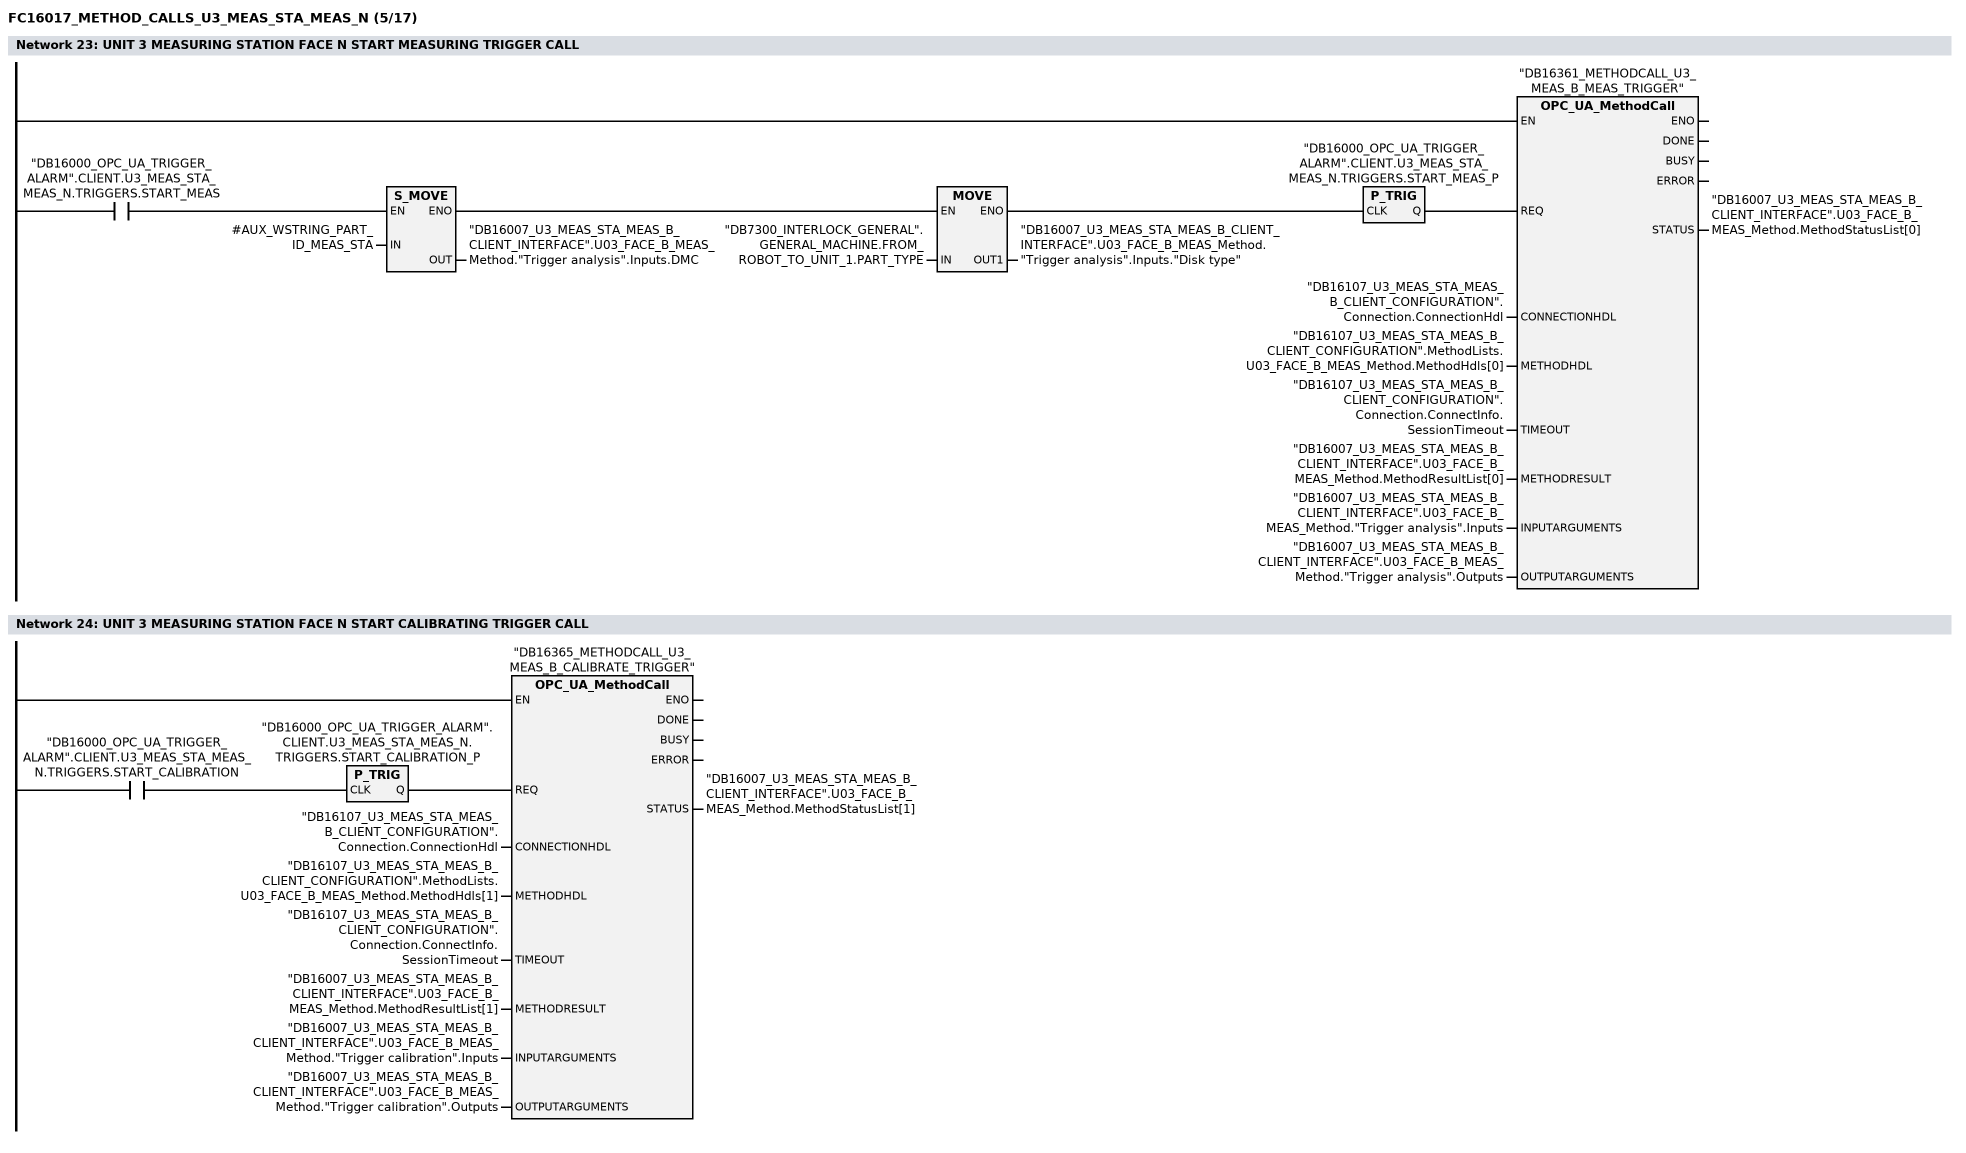
   RUNG wire#powerrail
      "DB16361_METHODCALL_U3_MEAS_B_MEAS_TRIGGER".OPC_UA_MethodCall(REQ := wire#w1, ConnectionHdl := "DB16107_U3_MEAS_STA_MEAS_B_CLIENT_CONFIGURATION".Connection.ConnectionHdl, MethodHdl := "DB16107_U3_MEAS_STA_MEAS_B_CLIENT_CONFIGURATION".MethodLists.U03_FACE_B_MEAS_Method.MethodHdls[0], Timeout := "DB16107_U3_MEAS_STA_MEAS_B_CLIENT_CONFIGURATION".Connection.ConnectInfo.SessionTimeout, MethodResult := "DB16007_U3_MEAS_STA_MEAS_B_CLIENT_INTERFACE".U03_FACE_B_MEAS_Method.MethodResultList[0], InputArguments := "DB16007_U3_MEAS_STA_MEAS_B_CLIENT_INTERFACE".U03_FACE_B_MEAS_Method."Trigger analysis".Inputs, OutputArguments := "DB16007_U3_MEAS_STA_MEAS_B_CLIENT_INTERFACE".U03_FACE_B_MEAS_Method."Trigger analysis".Outputs, Done =>, Busy =>, Error =>, Status => "DB16007_U3_MEAS_STA_MEAS_B_CLIENT_INTERFACE".U03_FACE_B_MEAS_Method.MethodStatusList[0])
   END_RUNG
   RUNG wire#powerrail
      Contact( "DB16000_OPC_UA_TRIGGER_ALARM".CLIENT.U3_MEAS_STA_MEAS_N.TRIGGERS.START_MEAS )
      S_Move(in := #AUX_WSTRING_PART_ID_MEAS_STA, out => "DB16007_U3_MEAS_STA_MEAS_B_CLIENT_INTERFACE".U03_FACE_B_MEAS_Method."Trigger analysis".Inputs.DMC)
      Move(in := "DB7300_INTERLOCK_GENERAL".GENERAL_MACHINE.FROM_ROBOT_TO_UNIT_1.PART_TYPE, out1 => "DB16007_U3_MEAS_STA_MEAS_B_CLIENT_INTERFACE".U03_FACE_B_MEAS_Method."Trigger analysis".Inputs."Disk type")
      P_Trig( "DB16000_OPC_UA_TRIGGER_ALARM".CLIENT.U3_MEAS_STA_MEAS_N.TRIGGERS.START_MEAS_P )
   END_RUNG wire#w1
   // the same network as SCL:
   IF "DB16000_OPC_UA_TRIGGER_ALARM".CLIENT.U3_MEAS_STA_MEAS_N.TRIGGERS.START_MEAS THEN
       "DB16007_U3_MEAS_STA_MEAS_B_CLIENT_INTERFACE".U03_FACE_B_MEAS_Method."Trigger analysis".Inputs.DMC := #AUX_WSTRING_PART_ID_MEAS_STA;
       "DB16007_U3_MEAS_STA_MEAS_B_CLIENT_INTERFACE".U03_FACE_B_MEAS_Method."Trigger analysis".Inputs."Disk type" := "DB7300_INTERLOCK_GENERAL".GENERAL_MACHINE.FROM_ROBOT_TO_UNIT_1.PART_TYPE;
   END_IF;
   #_w1 := "DB16000_OPC_UA_TRIGGER_ALARM".CLIENT.U3_MEAS_STA_MEAS_N.TRIGGERS.START_MEAS AND NOT "DB16000_OPC_UA_TRIGGER_ALARM".CLIENT.U3_MEAS_STA_MEAS_N.TRIGGERS.START_MEAS_P;   // rising edge
   "DB16000_OPC_UA_TRIGGER_ALARM".CLIENT.U3_MEAS_STA_MEAS_N.TRIGGERS.START_MEAS_P := "DB16000_OPC_UA_TRIGGER_ALARM".CLIENT.U3_MEAS_STA_MEAS_N.TRIGGERS.START_MEAS;
   "DB16361_METHODCALL_U3_MEAS_B_MEAS_TRIGGER"(REQ := #_w1,   // OPC_UA_MethodCall
                           ConnectionHdl := "DB16107_U3_MEAS_STA_MEAS_B_CLIENT_CONFIGURATION".Connection.ConnectionHdl,
                           MethodHdl := "DB16107_U3_MEAS_STA_MEAS_B_CLIENT_CONFIGURATION".MethodLists.U03_FACE_B_MEAS_Method.MethodHdls[0],
                           Timeout := "DB16107_U3_MEAS_STA_MEAS_B_CLIENT_CONFIGURATION".Connection.ConnectInfo.SessionTimeout,
                           MethodResult := "DB16007_U3_MEAS_STA_MEAS_B_CLIENT_INTERFACE".U03_FACE_B_MEAS_Method.MethodResultList[0],
                           InputArguments := "DB16007_U3_MEAS_STA_MEAS_B_CLIENT_INTERFACE".U03_FACE_B_MEAS_Method."Trigger analysis".Inputs,
                           OutputArguments := "DB16007_U3_MEAS_STA_MEAS_B_CLIENT_INTERFACE".U03_FACE_B_MEAS_Method."Trigger analysis".Outputs,
                           Status => "DB16007_U3_MEAS_STA_MEAS_B_CLIENT_INTERFACE".U03_FACE_B_MEAS_Method.MethodStatusList[0]);
END_REGION

REGION Network 24: UNIT 3 MEASURING STATION FACE N START CALIBRATING TRIGGER CALL
   RUNG wire#powerrail
      "DB16365_METHODCALL_U3_MEAS_B_CALIBRATE_TRIGGER".OPC_UA_MethodCall(REQ := wire#w1, ConnectionHdl := "DB16107_U3_MEAS_STA_MEAS_B_CLIENT_CONFIGURATION".Connection.ConnectionHdl, MethodHdl := "DB16107_U3_MEAS_STA_MEAS_B_CLIENT_CONFIGURATION".MethodLists.U03_FACE_B_MEAS_Method.MethodHdls[1], Timeout := "DB16107_U3_MEAS_STA_MEAS_B_CLIENT_CONFIGURATION".Connection.ConnectInfo.SessionTimeout, MethodResult := "DB16007_U3_MEAS_STA_MEAS_B_CLIENT_INTERFACE".U03_FACE_B_MEAS_Method.MethodResultList[1], InputArguments := "DB16007_U3_MEAS_STA_MEAS_B_CLIENT_INTERFACE".U03_FACE_B_MEAS_Method."Trigger calibration".Inputs, OutputArguments := "DB16007_U3_MEAS_STA_MEAS_B_CLIENT_INTERFACE".U03_FACE_B_MEAS_Method."Trigger calibration".Outputs, Done =>, Busy =>, Error =>, Status => "DB16007_U3_MEAS_STA_MEAS_B_CLIENT_INTERFACE".U03_FACE_B_MEAS_Method.MethodStatusList[1])
   END_RUNG
   RUNG wire#powerrail
      Contact( "DB16000_OPC_UA_TRIGGER_ALARM".CLIENT.U3_MEAS_STA_MEAS_N.TRIGGERS.START_CALIBRATION )
      P_Trig( "DB16000_OPC_UA_TRIGGER_ALARM".CLIENT.U3_MEAS_STA_MEAS_N.TRIGGERS.START_CALIBRATION_P )
   END_RUNG wire#w1
   // the same network as SCL:
   #_w1 := "DB16000_OPC_UA_TRIGGER_ALARM".CLIENT.U3_MEAS_STA_MEAS_N.TRIGGERS.START_CALIBRATION AND NOT "DB16000_OPC_UA_TRIGGER_ALARM".CLIENT.U3_MEAS_STA_MEAS_N.TRIGGERS.START_CALIBRATION_P;   // rising edge
   "DB16000_OPC_UA_TRIGGER_ALARM".CLIENT.U3_MEAS_STA_MEAS_N.TRIGGERS.START_CALIBRATION_P := "DB16000_OPC_UA_TRIGGER_ALARM".CLIENT.U3_MEAS_STA_MEAS_N.TRIGGERS.START_CALIBRATION;
   "DB16365_METHODCALL_U3_MEAS_B_CALIBRATE_TRIGGER"(REQ := #_w1,   // OPC_UA_MethodCall
                           ConnectionHdl := "DB16107_U3_MEAS_STA_MEAS_B_CLIENT_CONFIGURATION".Connection.ConnectionHdl,
                           MethodHdl := "DB16107_U3_MEAS_STA_MEAS_B_CLIENT_CONFIGURATION".MethodLists.U03_FACE_B_MEAS_Method.MethodHdls[1],
                           Timeout := "DB16107_U3_MEAS_STA_MEAS_B_CLIENT_CONFIGURATION".Connection.ConnectInfo.SessionTimeout,
                           MethodResult := "DB16007_U3_MEAS_STA_MEAS_B_CLIENT_INTERFACE".U03_FACE_B_MEAS_Method.MethodResultList[1],
                           InputArguments := "DB16007_U3_MEAS_STA_MEAS_B_CLIENT_INTERFACE".U03_FACE_B_MEAS_Method."Trigger calibration".Inputs,
                           OutputArguments := "DB16007_U3_MEAS_STA_MEAS_B_CLIENT_INTERFACE".U03_FACE_B_MEAS_Method."Trigger calibration".Outputs,
                           Status => "DB16007_U3_MEAS_STA_MEAS_B_CLIENT_INTERFACE".U03_FACE_B_MEAS_Method.MethodStatusList[1]);
END_REGION

REGION Network 25: UNIT 3 MEASURING STATION FACE N RESET PC TRIGGER CALL
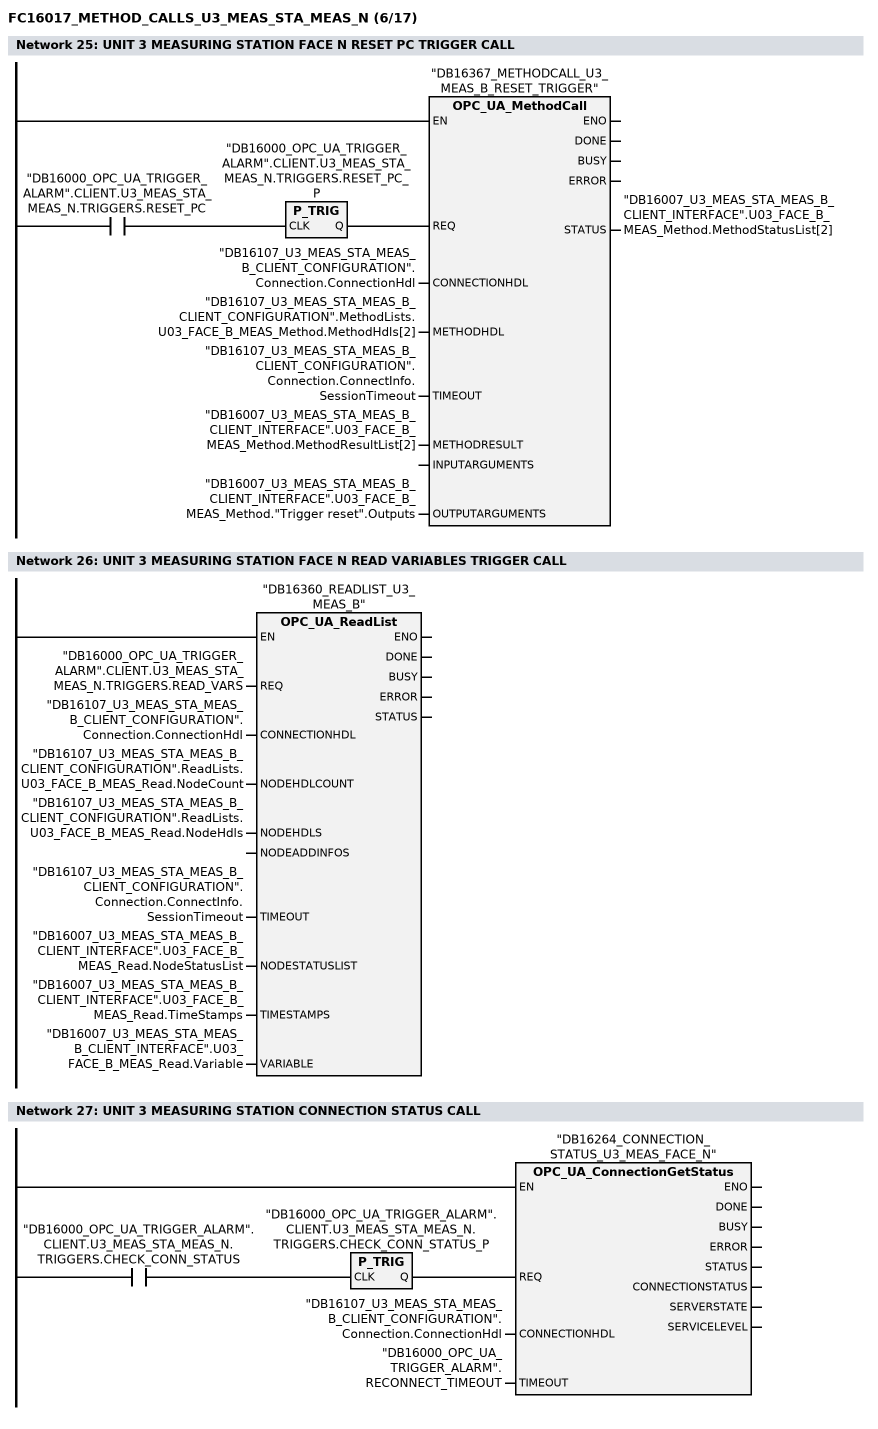
   RUNG wire#powerrail
      "DB16367_METHODCALL_U3_MEAS_B_RESET_TRIGGER".OPC_UA_MethodCall(REQ := wire#w1, ConnectionHdl := "DB16107_U3_MEAS_STA_MEAS_B_CLIENT_CONFIGURATION".Connection.ConnectionHdl, MethodHdl := "DB16107_U3_MEAS_STA_MEAS_B_CLIENT_CONFIGURATION".MethodLists.U03_FACE_B_MEAS_Method.MethodHdls[2], Timeout := "DB16107_U3_MEAS_STA_MEAS_B_CLIENT_CONFIGURATION".Connection.ConnectInfo.SessionTimeout, MethodResult := "DB16007_U3_MEAS_STA_MEAS_B_CLIENT_INTERFACE".U03_FACE_B_MEAS_Method.MethodResultList[2], InputArguments :=, OutputArguments := "DB16007_U3_MEAS_STA_MEAS_B_CLIENT_INTERFACE".U03_FACE_B_MEAS_Method."Trigger reset".Outputs, Done =>, Busy =>, Error =>, Status => "DB16007_U3_MEAS_STA_MEAS_B_CLIENT_INTERFACE".U03_FACE_B_MEAS_Method.MethodStatusList[2])
   END_RUNG
   RUNG wire#powerrail
      Contact( "DB16000_OPC_UA_TRIGGER_ALARM".CLIENT.U3_MEAS_STA_MEAS_N.TRIGGERS.RESET_PC )
      P_Trig( "DB16000_OPC_UA_TRIGGER_ALARM".CLIENT.U3_MEAS_STA_MEAS_N.TRIGGERS.RESET_PC_P )
   END_RUNG wire#w1
   // the same network as SCL:
   #_w1 := "DB16000_OPC_UA_TRIGGER_ALARM".CLIENT.U3_MEAS_STA_MEAS_N.TRIGGERS.RESET_PC AND NOT "DB16000_OPC_UA_TRIGGER_ALARM".CLIENT.U3_MEAS_STA_MEAS_N.TRIGGERS.RESET_PC_P;   // rising edge
   "DB16000_OPC_UA_TRIGGER_ALARM".CLIENT.U3_MEAS_STA_MEAS_N.TRIGGERS.RESET_PC_P := "DB16000_OPC_UA_TRIGGER_ALARM".CLIENT.U3_MEAS_STA_MEAS_N.TRIGGERS.RESET_PC;
   "DB16367_METHODCALL_U3_MEAS_B_RESET_TRIGGER"(REQ := #_w1,   // OPC_UA_MethodCall
                           ConnectionHdl := "DB16107_U3_MEAS_STA_MEAS_B_CLIENT_CONFIGURATION".Connection.ConnectionHdl,
                           MethodHdl := "DB16107_U3_MEAS_STA_MEAS_B_CLIENT_CONFIGURATION".MethodLists.U03_FACE_B_MEAS_Method.MethodHdls[2],
                           Timeout := "DB16107_U3_MEAS_STA_MEAS_B_CLIENT_CONFIGURATION".Connection.ConnectInfo.SessionTimeout,
                           MethodResult := "DB16007_U3_MEAS_STA_MEAS_B_CLIENT_INTERFACE".U03_FACE_B_MEAS_Method.MethodResultList[2],
                           OutputArguments := "DB16007_U3_MEAS_STA_MEAS_B_CLIENT_INTERFACE".U03_FACE_B_MEAS_Method."Trigger reset".Outputs,
                           Status => "DB16007_U3_MEAS_STA_MEAS_B_CLIENT_INTERFACE".U03_FACE_B_MEAS_Method.MethodStatusList[2]);
END_REGION

REGION Network 26: UNIT 3 MEASURING STATION FACE N READ VARIABLES TRIGGER CALL
   RUNG wire#powerrail
      "DB16360_READLIST_U3_MEAS_B".OPC_UA_ReadList(REQ := "DB16000_OPC_UA_TRIGGER_ALARM".CLIENT.U3_MEAS_STA_MEAS_N.TRIGGERS.READ_VARS, ConnectionHdl := "DB16107_U3_MEAS_STA_MEAS_B_CLIENT_CONFIGURATION".Connection.ConnectionHdl, NodeHdlCount := "DB16107_U3_MEAS_STA_MEAS_B_CLIENT_CONFIGURATION".ReadLists.U03_FACE_B_MEAS_Read.NodeCount, NodeHdls := "DB16107_U3_MEAS_STA_MEAS_B_CLIENT_CONFIGURATION".ReadLists.U03_FACE_B_MEAS_Read.NodeHdls, NodeAddInfos :=, Timeout := "DB16107_U3_MEAS_STA_MEAS_B_CLIENT_CONFIGURATION".Connection.ConnectInfo.SessionTimeout, NodeStatusList := "DB16007_U3_MEAS_STA_MEAS_B_CLIENT_INTERFACE".U03_FACE_B_MEAS_Read.NodeStatusList, TimeStamps := "DB16007_U3_MEAS_STA_MEAS_B_CLIENT_INTERFACE".U03_FACE_B_MEAS_Read.TimeStamps, Variable := "DB16007_U3_MEAS_STA_MEAS_B_CLIENT_INTERFACE".U03_FACE_B_MEAS_Read.Variable, Done =>, Busy =>, Error =>, Status =>)
   END_RUNG
   // the same network as SCL:
   "DB16360_READLIST_U3_MEAS_B"(REQ := "DB16000_OPC_UA_TRIGGER_ALARM".CLIENT.U3_MEAS_STA_MEAS_N.TRIGGERS.READ_VARS,   // OPC_UA_ReadList
                           ConnectionHdl := "DB16107_U3_MEAS_STA_MEAS_B_CLIENT_CONFIGURATION".Connection.ConnectionHdl,
                           NodeHdlCount := "DB16107_U3_MEAS_STA_MEAS_B_CLIENT_CONFIGURATION".ReadLists.U03_FACE_B_MEAS_Read.NodeCount,
                           NodeHdls := "DB16107_U3_MEAS_STA_MEAS_B_CLIENT_CONFIGURATION".ReadLists.U03_FACE_B_MEAS_Read.NodeHdls,
                           Timeout := "DB16107_U3_MEAS_STA_MEAS_B_CLIENT_CONFIGURATION".Connection.ConnectInfo.SessionTimeout,
                           NodeStatusList := "DB16007_U3_MEAS_STA_MEAS_B_CLIENT_INTERFACE".U03_FACE_B_MEAS_Read.NodeStatusList,
                           TimeStamps := "DB16007_U3_MEAS_STA_MEAS_B_CLIENT_INTERFACE".U03_FACE_B_MEAS_Read.TimeStamps,
                           Variable := "DB16007_U3_MEAS_STA_MEAS_B_CLIENT_INTERFACE".U03_FACE_B_MEAS_Read.Variable);
END_REGION

REGION Network 27: UNIT 3 MEASURING STATION CONNECTION STATUS CALL
   RUNG wire#powerrail
      "DB16264_CONNECTION_STATUS_U3_MEAS_FACE_N".OPC_UA_ConnectionGetStatus(REQ := wire#w1, ConnectionHdl := "DB16107_U3_MEAS_STA_MEAS_B_CLIENT_CONFIGURATION".Connection.ConnectionHdl, Timeout := "DB16000_OPC_UA_TRIGGER_ALARM".RECONNECT_TIMEOUT, Done =>, Busy =>, Error =>, Status =>, ConnectionStatus =>, ServerState =>, ServiceLevel =>)
   END_RUNG
   RUNG wire#powerrail
      Contact( "DB16000_OPC_UA_TRIGGER_ALARM".CLIENT.U3_MEAS_STA_MEAS_N.TRIGGERS.CHECK_CONN_STATUS )
      P_Trig( "DB16000_OPC_UA_TRIGGER_ALARM".CLIENT.U3_MEAS_STA_MEAS_N.TRIGGERS.CHECK_CONN_STATUS_P )
   END_RUNG wire#w1
   // the same network as SCL:
   #_w1 := "DB16000_OPC_UA_TRIGGER_ALARM".CLIENT.U3_MEAS_STA_MEAS_N.TRIGGERS.CHECK_CONN_STATUS AND NOT "DB16000_OPC_UA_TRIGGER_ALARM".CLIENT.U3_MEAS_STA_MEAS_N.TRIGGERS.CHECK_CONN_STATUS_P;   // rising edge
   "DB16000_OPC_UA_TRIGGER_ALARM".CLIENT.U3_MEAS_STA_MEAS_N.TRIGGERS.CHECK_CONN_STATUS_P := "DB16000_OPC_UA_TRIGGER_ALARM".CLIENT.U3_MEAS_STA_MEAS_N.TRIGGERS.CHECK_CONN_STATUS;
   "DB16264_CONNECTION_STATUS_U3_MEAS_FACE_N"(REQ := #_w1,   // OPC_UA_ConnectionGetStatus
                           ConnectionHdl := "DB16107_U3_MEAS_STA_MEAS_B_CLIENT_CONFIGURATION".Connection.ConnectionHdl,
                           Timeout := "DB16000_OPC_UA_TRIGGER_ALARM".RECONNECT_TIMEOUT);
END_REGION

REGION Network 28: UNIT 3 MEASURING STATION RELEASE HANDLE LIST CALL
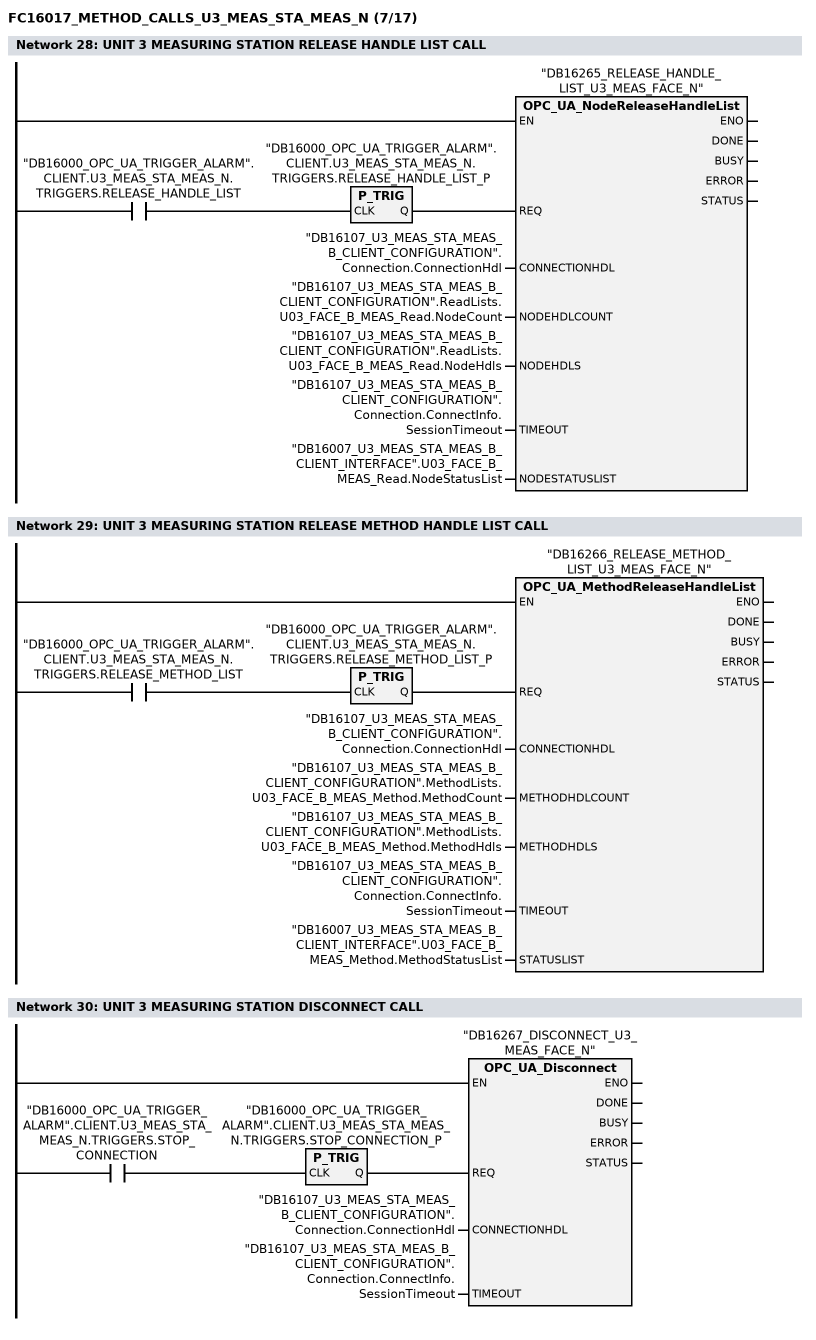
   RUNG wire#powerrail
      "DB16265_RELEASE_HANDLE_LIST_U3_MEAS_FACE_N".OPC_UA_NodeReleaseHandleList(REQ := wire#w1, ConnectionHdl := "DB16107_U3_MEAS_STA_MEAS_B_CLIENT_CONFIGURATION".Connection.ConnectionHdl, NodeHdlCount := "DB16107_U3_MEAS_STA_MEAS_B_CLIENT_CONFIGURATION".ReadLists.U03_FACE_B_MEAS_Read.NodeCount, NodeHdls := "DB16107_U3_MEAS_STA_MEAS_B_CLIENT_CONFIGURATION".ReadLists.U03_FACE_B_MEAS_Read.NodeHdls, Timeout := "DB16107_U3_MEAS_STA_MEAS_B_CLIENT_CONFIGURATION".Connection.ConnectInfo.SessionTimeout, NodeStatusList := "DB16007_U3_MEAS_STA_MEAS_B_CLIENT_INTERFACE".U03_FACE_B_MEAS_Read.NodeStatusList, Done =>, Busy =>, Error =>, Status =>)
   END_RUNG
   RUNG wire#powerrail
      Contact( "DB16000_OPC_UA_TRIGGER_ALARM".CLIENT.U3_MEAS_STA_MEAS_N.TRIGGERS.RELEASE_HANDLE_LIST )
      P_Trig( "DB16000_OPC_UA_TRIGGER_ALARM".CLIENT.U3_MEAS_STA_MEAS_N.TRIGGERS.RELEASE_HANDLE_LIST_P )
   END_RUNG wire#w1
   // the same network as SCL:
   #_w1 := "DB16000_OPC_UA_TRIGGER_ALARM".CLIENT.U3_MEAS_STA_MEAS_N.TRIGGERS.RELEASE_HANDLE_LIST AND NOT "DB16000_OPC_UA_TRIGGER_ALARM".CLIENT.U3_MEAS_STA_MEAS_N.TRIGGERS.RELEASE_HANDLE_LIST_P;   // rising edge
   "DB16000_OPC_UA_TRIGGER_ALARM".CLIENT.U3_MEAS_STA_MEAS_N.TRIGGERS.RELEASE_HANDLE_LIST_P := "DB16000_OPC_UA_TRIGGER_ALARM".CLIENT.U3_MEAS_STA_MEAS_N.TRIGGERS.RELEASE_HANDLE_LIST;
   "DB16265_RELEASE_HANDLE_LIST_U3_MEAS_FACE_N"(REQ := #_w1,   // OPC_UA_NodeReleaseHandleList
                           ConnectionHdl := "DB16107_U3_MEAS_STA_MEAS_B_CLIENT_CONFIGURATION".Connection.ConnectionHdl,
                           NodeHdlCount := "DB16107_U3_MEAS_STA_MEAS_B_CLIENT_CONFIGURATION".ReadLists.U03_FACE_B_MEAS_Read.NodeCount,
                           NodeHdls := "DB16107_U3_MEAS_STA_MEAS_B_CLIENT_CONFIGURATION".ReadLists.U03_FACE_B_MEAS_Read.NodeHdls,
                           Timeout := "DB16107_U3_MEAS_STA_MEAS_B_CLIENT_CONFIGURATION".Connection.ConnectInfo.SessionTimeout,
                           NodeStatusList := "DB16007_U3_MEAS_STA_MEAS_B_CLIENT_INTERFACE".U03_FACE_B_MEAS_Read.NodeStatusList);
END_REGION

REGION Network 29: UNIT 3 MEASURING STATION RELEASE METHOD HANDLE LIST CALL
   RUNG wire#powerrail
      "DB16266_RELEASE_METHOD_LIST_U3_MEAS_FACE_N".OPC_UA_MethodReleaseHandleList(REQ := wire#w1, ConnectionHdl := "DB16107_U3_MEAS_STA_MEAS_B_CLIENT_CONFIGURATION".Connection.ConnectionHdl, MethodHdlCount := "DB16107_U3_MEAS_STA_MEAS_B_CLIENT_CONFIGURATION".MethodLists.U03_FACE_B_MEAS_Method.MethodCount, MethodHdls := "DB16107_U3_MEAS_STA_MEAS_B_CLIENT_CONFIGURATION".MethodLists.U03_FACE_B_MEAS_Method.MethodHdls, Timeout := "DB16107_U3_MEAS_STA_MEAS_B_CLIENT_CONFIGURATION".Connection.ConnectInfo.SessionTimeout, StatusList := "DB16007_U3_MEAS_STA_MEAS_B_CLIENT_INTERFACE".U03_FACE_B_MEAS_Method.MethodStatusList, Done =>, Busy =>, Error =>, Status =>)
   END_RUNG
   RUNG wire#powerrail
      Contact( "DB16000_OPC_UA_TRIGGER_ALARM".CLIENT.U3_MEAS_STA_MEAS_N.TRIGGERS.RELEASE_METHOD_LIST )
      P_Trig( "DB16000_OPC_UA_TRIGGER_ALARM".CLIENT.U3_MEAS_STA_MEAS_N.TRIGGERS.RELEASE_METHOD_LIST_P )
   END_RUNG wire#w1
   // the same network as SCL:
   #_w1 := "DB16000_OPC_UA_TRIGGER_ALARM".CLIENT.U3_MEAS_STA_MEAS_N.TRIGGERS.RELEASE_METHOD_LIST AND NOT "DB16000_OPC_UA_TRIGGER_ALARM".CLIENT.U3_MEAS_STA_MEAS_N.TRIGGERS.RELEASE_METHOD_LIST_P;   // rising edge
   "DB16000_OPC_UA_TRIGGER_ALARM".CLIENT.U3_MEAS_STA_MEAS_N.TRIGGERS.RELEASE_METHOD_LIST_P := "DB16000_OPC_UA_TRIGGER_ALARM".CLIENT.U3_MEAS_STA_MEAS_N.TRIGGERS.RELEASE_METHOD_LIST;
   "DB16266_RELEASE_METHOD_LIST_U3_MEAS_FACE_N"(REQ := #_w1,   // OPC_UA_MethodReleaseHandleList
                           ConnectionHdl := "DB16107_U3_MEAS_STA_MEAS_B_CLIENT_CONFIGURATION".Connection.ConnectionHdl,
                           MethodHdlCount := "DB16107_U3_MEAS_STA_MEAS_B_CLIENT_CONFIGURATION".MethodLists.U03_FACE_B_MEAS_Method.MethodCount,
                           MethodHdls := "DB16107_U3_MEAS_STA_MEAS_B_CLIENT_CONFIGURATION".MethodLists.U03_FACE_B_MEAS_Method.MethodHdls,
                           Timeout := "DB16107_U3_MEAS_STA_MEAS_B_CLIENT_CONFIGURATION".Connection.ConnectInfo.SessionTimeout,
                           StatusList := "DB16007_U3_MEAS_STA_MEAS_B_CLIENT_INTERFACE".U03_FACE_B_MEAS_Method.MethodStatusList);
END_REGION

REGION Network 30: UNIT 3 MEASURING STATION DISCONNECT CALL
   RUNG wire#powerrail
      "DB16267_DISCONNECT_U3_MEAS_FACE_N".OPC_UA_Disconnect(REQ := wire#w1, ConnectionHdl := "DB16107_U3_MEAS_STA_MEAS_B_CLIENT_CONFIGURATION".Connection.ConnectionHdl, Timeout := "DB16107_U3_MEAS_STA_MEAS_B_CLIENT_CONFIGURATION".Connection.ConnectInfo.SessionTimeout, Done =>, Busy =>, Error =>, Status =>)
   END_RUNG
   RUNG wire#powerrail
      Contact( "DB16000_OPC_UA_TRIGGER_ALARM".CLIENT.U3_MEAS_STA_MEAS_N.TRIGGERS.STOP_CONNECTION )
      P_Trig( "DB16000_OPC_UA_TRIGGER_ALARM".CLIENT.U3_MEAS_STA_MEAS_N.TRIGGERS.STOP_CONNECTION_P )
   END_RUNG wire#w1
   // the same network as SCL:
   #_w1 := "DB16000_OPC_UA_TRIGGER_ALARM".CLIENT.U3_MEAS_STA_MEAS_N.TRIGGERS.STOP_CONNECTION AND NOT "DB16000_OPC_UA_TRIGGER_ALARM".CLIENT.U3_MEAS_STA_MEAS_N.TRIGGERS.STOP_CONNECTION_P;   // rising edge
   "DB16000_OPC_UA_TRIGGER_ALARM".CLIENT.U3_MEAS_STA_MEAS_N.TRIGGERS.STOP_CONNECTION_P := "DB16000_OPC_UA_TRIGGER_ALARM".CLIENT.U3_MEAS_STA_MEAS_N.TRIGGERS.STOP_CONNECTION;
   "DB16267_DISCONNECT_U3_MEAS_FACE_N"(REQ := #_w1,   // OPC_UA_Disconnect
                           ConnectionHdl := "DB16107_U3_MEAS_STA_MEAS_B_CLIENT_CONFIGURATION".Connection.ConnectionHdl,
                           Timeout := "DB16107_U3_MEAS_STA_MEAS_B_CLIENT_CONFIGURATION".Connection.ConnectInfo.SessionTimeout);
END_REGION

REGION Network 31: UNIT 3 MEASURING STATION RECONNECT
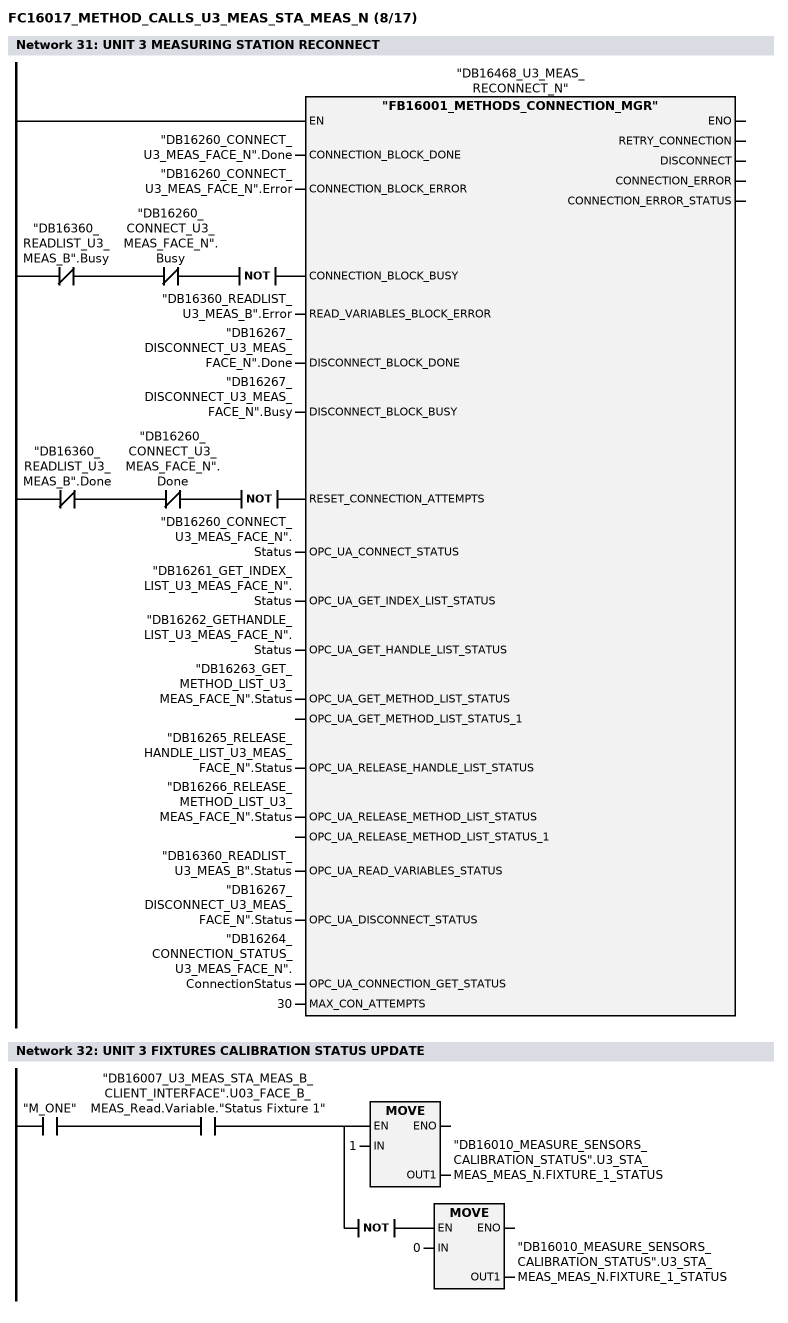
   RUNG wire#powerrail
      "DB16468_U3_MEAS_RECONNECT_N"(CONNECTION_BLOCK_BUSY := wire#w1, RESET_CONNECTION_ATTEMPTS := wire#w2, CONNECTION_BLOCK_DONE := "DB16260_CONNECT_U3_MEAS_FACE_N".Done, CONNECTION_BLOCK_ERROR := "DB16260_CONNECT_U3_MEAS_FACE_N".Error, READ_VARIABLES_BLOCK_ERROR := "DB16360_READLIST_U3_MEAS_B".Error, DISCONNECT_BLOCK_DONE := "DB16267_DISCONNECT_U3_MEAS_FACE_N".Done, DISCONNECT_BLOCK_BUSY := "DB16267_DISCONNECT_U3_MEAS_FACE_N".Busy, OPC_UA_CONNECT_STATUS := "DB16260_CONNECT_U3_MEAS_FACE_N".Status, OPC_UA_GET_INDEX_LIST_STATUS := "DB16261_GET_INDEX_LIST_U3_MEAS_FACE_N".Status, OPC_UA_GET_HANDLE_LIST_STATUS := "DB16262_GETHANDLE_LIST_U3_MEAS_FACE_N".Status, OPC_UA_GET_METHOD_LIST_STATUS := "DB16263_GET_METHOD_LIST_U3_MEAS_FACE_N".Status, OPC_UA_GET_METHOD_LIST_STATUS_1 :=, OPC_UA_RELEASE_HANDLE_LIST_STATUS := "DB16265_RELEASE_HANDLE_LIST_U3_MEAS_FACE_N".Status, OPC_UA_RELEASE_METHOD_LIST_STATUS := "DB16266_RELEASE_METHOD_LIST_U3_MEAS_FACE_N".Status, OPC_UA_RELEASE_METHOD_LIST_STATUS_1 :=, OPC_UA_READ_VARIABLES_STATUS := "DB16360_READLIST_U3_MEAS_B".Status, OPC_UA_DISCONNECT_STATUS := "DB16267_DISCONNECT_U3_MEAS_FACE_N".Status, OPC_UA_CONNECTION_GET_STATUS := "DB16264_CONNECTION_STATUS_U3_MEAS_FACE_N".ConnectionStatus, MAX_CON_ATTEMPTS := 30, RETRY_CONNECTION =>, DISCONNECT =>, CONNECTION_ERROR =>, CONNECTION_ERROR_STATUS =>)
   END_RUNG
   RUNG wire#powerrail
      I_Contact( "DB16360_READLIST_U3_MEAS_B".Busy )
      I_Contact( "DB16260_CONNECT_U3_MEAS_FACE_N".Busy )
      Not()
   END_RUNG wire#w1
   RUNG wire#powerrail
      I_Contact( "DB16360_READLIST_U3_MEAS_B".Done )
      I_Contact( "DB16260_CONNECT_U3_MEAS_FACE_N".Done )
      Not()
   END_RUNG wire#w2
   // the same network as SCL:
   "DB16468_U3_MEAS_RECONNECT_N"(CONNECTION_BLOCK_DONE := "DB16260_CONNECT_U3_MEAS_FACE_N".Done,   // "FB16001_METHODS_CONNECTION_MGR"
                           CONNECTION_BLOCK_ERROR := "DB16260_CONNECT_U3_MEAS_FACE_N".Error,
                           CONNECTION_BLOCK_BUSY := NOT (NOT "DB16360_READLIST_U3_MEAS_B".Busy AND NOT "DB16260_CONNECT_U3_MEAS_FACE_N".Busy),
                           READ_VARIABLES_BLOCK_ERROR := "DB16360_READLIST_U3_MEAS_B".Error,
                           DISCONNECT_BLOCK_DONE := "DB16267_DISCONNECT_U3_MEAS_FACE_N".Done,
                           DISCONNECT_BLOCK_BUSY := "DB16267_DISCONNECT_U3_MEAS_FACE_N".Busy,
                           RESET_CONNECTION_ATTEMPTS := NOT (NOT "DB16360_READLIST_U3_MEAS_B".Done AND NOT "DB16260_CONNECT_U3_MEAS_FACE_N".Done),
                           OPC_UA_CONNECT_STATUS := "DB16260_CONNECT_U3_MEAS_FACE_N".Status,
                           OPC_UA_GET_INDEX_LIST_STATUS := "DB16261_GET_INDEX_LIST_U3_MEAS_FACE_N".Status,
                           OPC_UA_GET_HANDLE_LIST_STATUS := "DB16262_GETHANDLE_LIST_U3_MEAS_FACE_N".Status,
                           OPC_UA_GET_METHOD_LIST_STATUS := "DB16263_GET_METHOD_LIST_U3_MEAS_FACE_N".Status,
                           OPC_UA_RELEASE_HANDLE_LIST_STATUS := "DB16265_RELEASE_HANDLE_LIST_U3_MEAS_FACE_N".Status,
                           OPC_UA_RELEASE_METHOD_LIST_STATUS := "DB16266_RELEASE_METHOD_LIST_U3_MEAS_FACE_N".Status,
                           OPC_UA_READ_VARIABLES_STATUS := "DB16360_READLIST_U3_MEAS_B".Status,
                           OPC_UA_DISCONNECT_STATUS := "DB16267_DISCONNECT_U3_MEAS_FACE_N".Status,
                           OPC_UA_CONNECTION_GET_STATUS := "DB16264_CONNECTION_STATUS_U3_MEAS_FACE_N".ConnectionStatus,
                           MAX_CON_ATTEMPTS := 30);
END_REGION

REGION Network 32: UNIT 3 FIXTURES CALIBRATION STATUS UPDATE
   RUNG wire#powerrail
      Contact( "M_ONE" )
      Contact( "DB16007_U3_MEAS_STA_MEAS_B_CLIENT_INTERFACE".U03_FACE_B_MEAS_Read.Variable."Status Fixture 1" )
      wire#w1
      Move(in := 1, out1 => "DB16010_MEASURE_SENSORS_CALIBRATION_STATUS".U3_STA_MEAS_MEAS_N.FIXTURE_1_STATUS)
   END_RUNG
   RUNG wire#w1
      Not()
      Move(in := 0, out1 => "DB16010_MEASURE_SENSORS_CALIBRATION_STATUS".U3_STA_MEAS_MEAS_N.FIXTURE_1_STATUS)
   END_RUNG
   // the same network as SCL:
   #_w1 := "M_ONE" AND "DB16007_U3_MEAS_STA_MEAS_B_CLIENT_INTERFACE".U03_FACE_B_MEAS_Read.Variable."Status Fixture 1";
   IF #_w1 THEN
       "DB16010_MEASURE_SENSORS_CALIBRATION_STATUS".U3_STA_MEAS_MEAS_N.FIXTURE_1_STATUS := 1;
   END_IF;
   IF NOT #_w1 THEN
       "DB16010_MEASURE_SENSORS_CALIBRATION_STATUS".U3_STA_MEAS_MEAS_N.FIXTURE_1_STATUS := 0;
   END_IF;
END_REGION

REGION Network 33: UNIT 3 MEASURING STATION FACE B COMPUTER CONNECTION ALARM
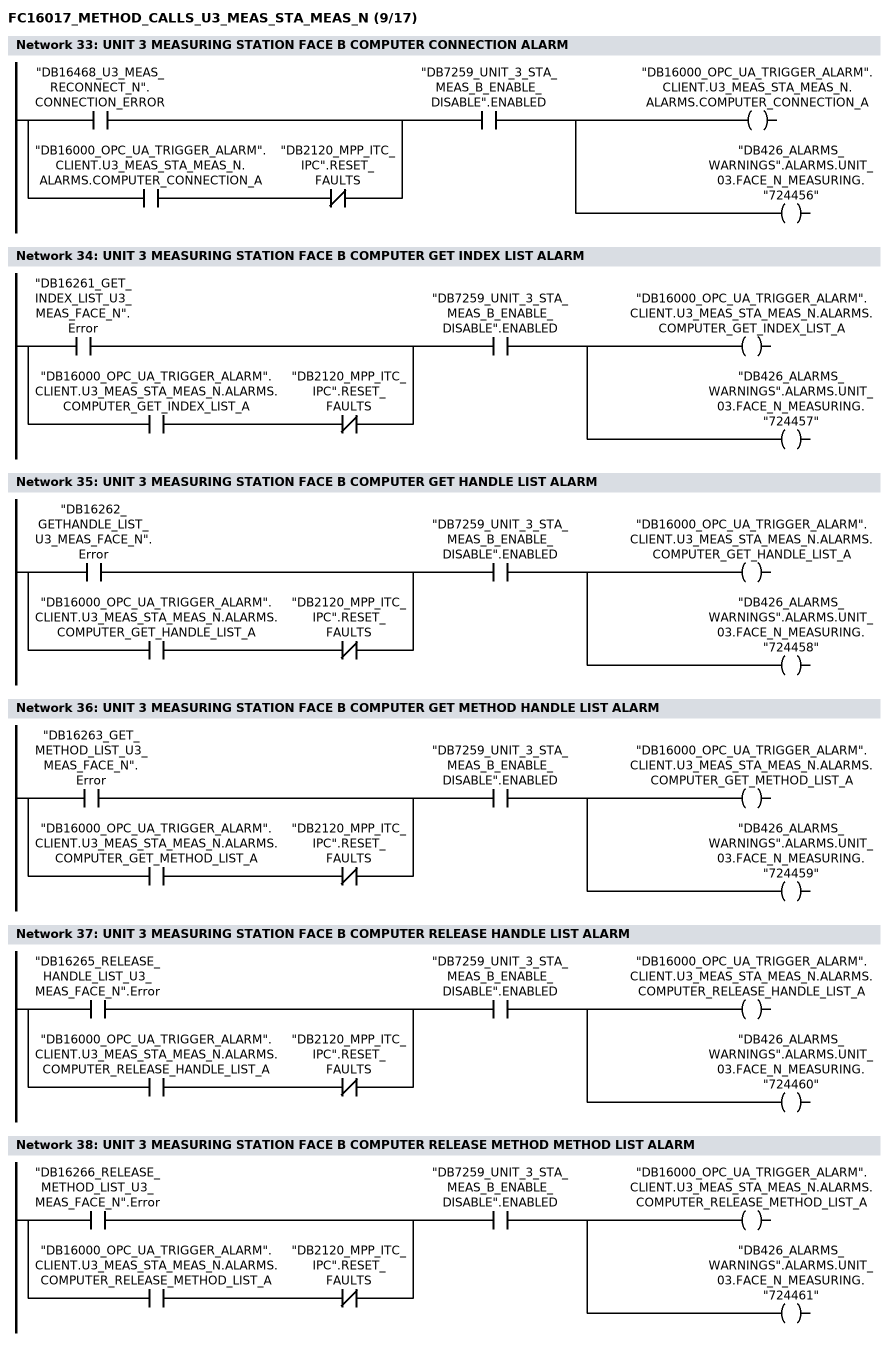
   RUNG wire#powerrail
      Contact( "DB16468_U3_MEAS_RECONNECT_N".CONNECTION_ERROR )
      wire#w1
      Contact( "DB7259_UNIT_3_STA_MEAS_B_ENABLE_DISABLE".ENABLED )
      wire#w2
      Coil( "DB16000_OPC_UA_TRIGGER_ALARM".CLIENT.U3_MEAS_STA_MEAS_N.ALARMS.COMPUTER_CONNECTION_A )
   END_RUNG
   RUNG wire#powerrail
      Contact( "DB16000_OPC_UA_TRIGGER_ALARM".CLIENT.U3_MEAS_STA_MEAS_N.ALARMS.COMPUTER_CONNECTION_A )
      I_Contact( "DB2120_MPP_ITC_IPC".RESET_FAULTS )
   END_RUNG wire#w1
   RUNG wire#w2
      Coil( "DB426_ALARMS_WARNINGS".ALARMS.UNIT_03.FACE_N_MEASURING."724456" )
   END_RUNG
   // the same network as SCL:
   "DB16000_OPC_UA_TRIGGER_ALARM".CLIENT.U3_MEAS_STA_MEAS_N.ALARMS.COMPUTER_CONNECTION_A := ("DB16468_U3_MEAS_RECONNECT_N".CONNECTION_ERROR OR ("DB16000_OPC_UA_TRIGGER_ALARM".CLIENT.U3_MEAS_STA_MEAS_N.ALARMS.COMPUTER_CONNECTION_A AND NOT "DB2120_MPP_ITC_IPC".RESET_FAULTS)) AND "DB7259_UNIT_3_STA_MEAS_B_ENABLE_DISABLE".ENABLED;
   "DB426_ALARMS_WARNINGS".ALARMS.UNIT_03.FACE_N_MEASURING."724456" := "DB16000_OPC_UA_TRIGGER_ALARM".CLIENT.U3_MEAS_STA_MEAS_N.ALARMS.COMPUTER_CONNECTION_A;
END_REGION

REGION Network 34: UNIT 3 MEASURING STATION FACE B COMPUTER GET INDEX LIST ALARM
   RUNG wire#powerrail
      Contact( "DB16261_GET_INDEX_LIST_U3_MEAS_FACE_N".Error )
      wire#w1
      Contact( "DB7259_UNIT_3_STA_MEAS_B_ENABLE_DISABLE".ENABLED )
      wire#w2
      Coil( "DB16000_OPC_UA_TRIGGER_ALARM".CLIENT.U3_MEAS_STA_MEAS_N.ALARMS.COMPUTER_GET_INDEX_LIST_A )
   END_RUNG
   RUNG wire#powerrail
      Contact( "DB16000_OPC_UA_TRIGGER_ALARM".CLIENT.U3_MEAS_STA_MEAS_N.ALARMS.COMPUTER_GET_INDEX_LIST_A )
      I_Contact( "DB2120_MPP_ITC_IPC".RESET_FAULTS )
   END_RUNG wire#w1
   RUNG wire#w2
      Coil( "DB426_ALARMS_WARNINGS".ALARMS.UNIT_03.FACE_N_MEASURING."724457" )
   END_RUNG
   // the same network as SCL:
   "DB16000_OPC_UA_TRIGGER_ALARM".CLIENT.U3_MEAS_STA_MEAS_N.ALARMS.COMPUTER_GET_INDEX_LIST_A := ("DB16261_GET_INDEX_LIST_U3_MEAS_FACE_N".Error OR ("DB16000_OPC_UA_TRIGGER_ALARM".CLIENT.U3_MEAS_STA_MEAS_N.ALARMS.COMPUTER_GET_INDEX_LIST_A AND NOT "DB2120_MPP_ITC_IPC".RESET_FAULTS)) AND "DB7259_UNIT_3_STA_MEAS_B_ENABLE_DISABLE".ENABLED;
   "DB426_ALARMS_WARNINGS".ALARMS.UNIT_03.FACE_N_MEASURING."724457" := "DB16000_OPC_UA_TRIGGER_ALARM".CLIENT.U3_MEAS_STA_MEAS_N.ALARMS.COMPUTER_GET_INDEX_LIST_A;
END_REGION

REGION Network 35: UNIT 3 MEASURING STATION FACE B COMPUTER GET HANDLE LIST ALARM
   RUNG wire#powerrail
      Contact( "DB16262_GETHANDLE_LIST_U3_MEAS_FACE_N".Error )
      wire#w1
      Contact( "DB7259_UNIT_3_STA_MEAS_B_ENABLE_DISABLE".ENABLED )
      wire#w2
      Coil( "DB16000_OPC_UA_TRIGGER_ALARM".CLIENT.U3_MEAS_STA_MEAS_N.ALARMS.COMPUTER_GET_HANDLE_LIST_A )
   END_RUNG
   RUNG wire#powerrail
      Contact( "DB16000_OPC_UA_TRIGGER_ALARM".CLIENT.U3_MEAS_STA_MEAS_N.ALARMS.COMPUTER_GET_HANDLE_LIST_A )
      I_Contact( "DB2120_MPP_ITC_IPC".RESET_FAULTS )
   END_RUNG wire#w1
   RUNG wire#w2
      Coil( "DB426_ALARMS_WARNINGS".ALARMS.UNIT_03.FACE_N_MEASURING."724458" )
   END_RUNG
   // the same network as SCL:
   "DB16000_OPC_UA_TRIGGER_ALARM".CLIENT.U3_MEAS_STA_MEAS_N.ALARMS.COMPUTER_GET_HANDLE_LIST_A := ("DB16262_GETHANDLE_LIST_U3_MEAS_FACE_N".Error OR ("DB16000_OPC_UA_TRIGGER_ALARM".CLIENT.U3_MEAS_STA_MEAS_N.ALARMS.COMPUTER_GET_HANDLE_LIST_A AND NOT "DB2120_MPP_ITC_IPC".RESET_FAULTS)) AND "DB7259_UNIT_3_STA_MEAS_B_ENABLE_DISABLE".ENABLED;
   "DB426_ALARMS_WARNINGS".ALARMS.UNIT_03.FACE_N_MEASURING."724458" := "DB16000_OPC_UA_TRIGGER_ALARM".CLIENT.U3_MEAS_STA_MEAS_N.ALARMS.COMPUTER_GET_HANDLE_LIST_A;
END_REGION

REGION Network 36: UNIT 3 MEASURING STATION FACE B COMPUTER GET METHOD HANDLE LIST ALARM
   RUNG wire#powerrail
      Contact( "DB16263_GET_METHOD_LIST_U3_MEAS_FACE_N".Error )
      wire#w1
      Contact( "DB7259_UNIT_3_STA_MEAS_B_ENABLE_DISABLE".ENABLED )
      wire#w2
      Coil( "DB16000_OPC_UA_TRIGGER_ALARM".CLIENT.U3_MEAS_STA_MEAS_N.ALARMS.COMPUTER_GET_METHOD_LIST_A )
   END_RUNG
   RUNG wire#powerrail
      Contact( "DB16000_OPC_UA_TRIGGER_ALARM".CLIENT.U3_MEAS_STA_MEAS_N.ALARMS.COMPUTER_GET_METHOD_LIST_A )
      I_Contact( "DB2120_MPP_ITC_IPC".RESET_FAULTS )
   END_RUNG wire#w1
   RUNG wire#w2
      Coil( "DB426_ALARMS_WARNINGS".ALARMS.UNIT_03.FACE_N_MEASURING."724459" )
   END_RUNG
   // the same network as SCL:
   "DB16000_OPC_UA_TRIGGER_ALARM".CLIENT.U3_MEAS_STA_MEAS_N.ALARMS.COMPUTER_GET_METHOD_LIST_A := ("DB16263_GET_METHOD_LIST_U3_MEAS_FACE_N".Error OR ("DB16000_OPC_UA_TRIGGER_ALARM".CLIENT.U3_MEAS_STA_MEAS_N.ALARMS.COMPUTER_GET_METHOD_LIST_A AND NOT "DB2120_MPP_ITC_IPC".RESET_FAULTS)) AND "DB7259_UNIT_3_STA_MEAS_B_ENABLE_DISABLE".ENABLED;
   "DB426_ALARMS_WARNINGS".ALARMS.UNIT_03.FACE_N_MEASURING."724459" := "DB16000_OPC_UA_TRIGGER_ALARM".CLIENT.U3_MEAS_STA_MEAS_N.ALARMS.COMPUTER_GET_METHOD_LIST_A;
END_REGION

REGION Network 37: UNIT 3 MEASURING STATION FACE B COMPUTER RELEASE HANDLE LIST ALARM
   RUNG wire#powerrail
      Contact( "DB16265_RELEASE_HANDLE_LIST_U3_MEAS_FACE_N".Error )
      wire#w1
      Contact( "DB7259_UNIT_3_STA_MEAS_B_ENABLE_DISABLE".ENABLED )
      wire#w2
      Coil( "DB16000_OPC_UA_TRIGGER_ALARM".CLIENT.U3_MEAS_STA_MEAS_N.ALARMS.COMPUTER_RELEASE_HANDLE_LIST_A )
   END_RUNG
   RUNG wire#powerrail
      Contact( "DB16000_OPC_UA_TRIGGER_ALARM".CLIENT.U3_MEAS_STA_MEAS_N.ALARMS.COMPUTER_RELEASE_HANDLE_LIST_A )
      I_Contact( "DB2120_MPP_ITC_IPC".RESET_FAULTS )
   END_RUNG wire#w1
   RUNG wire#w2
      Coil( "DB426_ALARMS_WARNINGS".ALARMS.UNIT_03.FACE_N_MEASURING."724460" )
   END_RUNG
   // the same network as SCL:
   "DB16000_OPC_UA_TRIGGER_ALARM".CLIENT.U3_MEAS_STA_MEAS_N.ALARMS.COMPUTER_RELEASE_HANDLE_LIST_A := ("DB16265_RELEASE_HANDLE_LIST_U3_MEAS_FACE_N".Error OR ("DB16000_OPC_UA_TRIGGER_ALARM".CLIENT.U3_MEAS_STA_MEAS_N.ALARMS.COMPUTER_RELEASE_HANDLE_LIST_A AND NOT "DB2120_MPP_ITC_IPC".RESET_FAULTS)) AND "DB7259_UNIT_3_STA_MEAS_B_ENABLE_DISABLE".ENABLED;
   "DB426_ALARMS_WARNINGS".ALARMS.UNIT_03.FACE_N_MEASURING."724460" := "DB16000_OPC_UA_TRIGGER_ALARM".CLIENT.U3_MEAS_STA_MEAS_N.ALARMS.COMPUTER_RELEASE_HANDLE_LIST_A;
END_REGION

REGION Network 38: UNIT 3 MEASURING STATION FACE B COMPUTER RELEASE METHOD METHOD LIST ALARM
   RUNG wire#powerrail
      Contact( "DB16266_RELEASE_METHOD_LIST_U3_MEAS_FACE_N".Error )
      wire#w1
      Contact( "DB7259_UNIT_3_STA_MEAS_B_ENABLE_DISABLE".ENABLED )
      wire#w2
      Coil( "DB16000_OPC_UA_TRIGGER_ALARM".CLIENT.U3_MEAS_STA_MEAS_N.ALARMS.COMPUTER_RELEASE_METHOD_LIST_A )
   END_RUNG
   RUNG wire#powerrail
      Contact( "DB16000_OPC_UA_TRIGGER_ALARM".CLIENT.U3_MEAS_STA_MEAS_N.ALARMS.COMPUTER_RELEASE_METHOD_LIST_A )
      I_Contact( "DB2120_MPP_ITC_IPC".RESET_FAULTS )
   END_RUNG wire#w1
   RUNG wire#w2
      Coil( "DB426_ALARMS_WARNINGS".ALARMS.UNIT_03.FACE_N_MEASURING."724461" )
   END_RUNG
   // the same network as SCL:
   "DB16000_OPC_UA_TRIGGER_ALARM".CLIENT.U3_MEAS_STA_MEAS_N.ALARMS.COMPUTER_RELEASE_METHOD_LIST_A := ("DB16266_RELEASE_METHOD_LIST_U3_MEAS_FACE_N".Error OR ("DB16000_OPC_UA_TRIGGER_ALARM".CLIENT.U3_MEAS_STA_MEAS_N.ALARMS.COMPUTER_RELEASE_METHOD_LIST_A AND NOT "DB2120_MPP_ITC_IPC".RESET_FAULTS)) AND "DB7259_UNIT_3_STA_MEAS_B_ENABLE_DISABLE".ENABLED;
   "DB426_ALARMS_WARNINGS".ALARMS.UNIT_03.FACE_N_MEASURING."724461" := "DB16000_OPC_UA_TRIGGER_ALARM".CLIENT.U3_MEAS_STA_MEAS_N.ALARMS.COMPUTER_RELEASE_METHOD_LIST_A;
END_REGION

REGION Network 39: UNIT 3 MEASURING STATION FACE B COMPUTER DISCONNECT ALARM
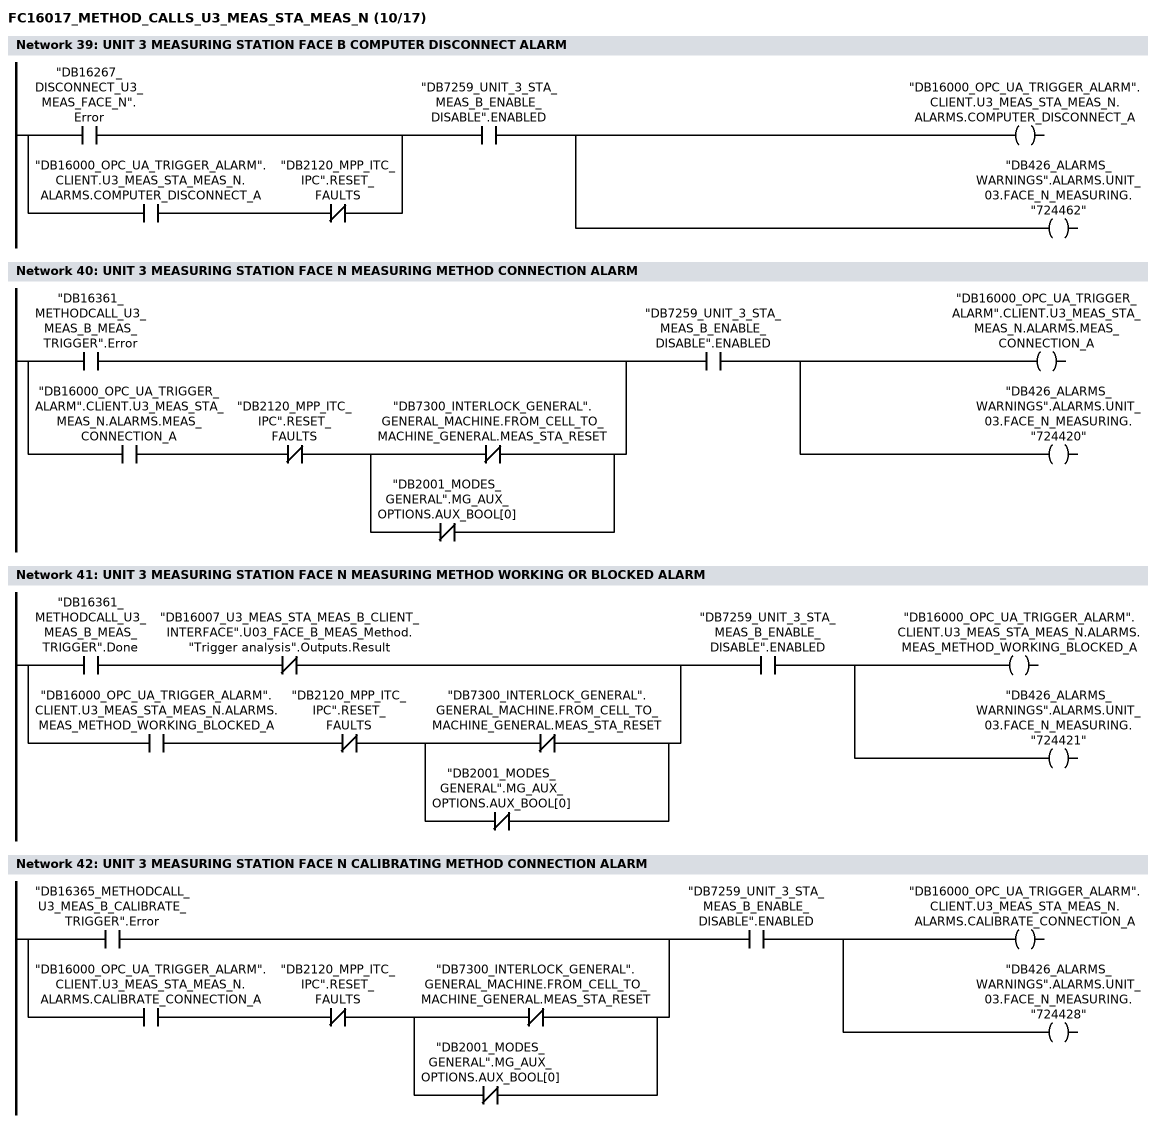
   RUNG wire#powerrail
      Contact( "DB16267_DISCONNECT_U3_MEAS_FACE_N".Error )
      wire#w1
      Contact( "DB7259_UNIT_3_STA_MEAS_B_ENABLE_DISABLE".ENABLED )
      wire#w2
      Coil( "DB16000_OPC_UA_TRIGGER_ALARM".CLIENT.U3_MEAS_STA_MEAS_N.ALARMS.COMPUTER_DISCONNECT_A )
   END_RUNG
   RUNG wire#powerrail
      Contact( "DB16000_OPC_UA_TRIGGER_ALARM".CLIENT.U3_MEAS_STA_MEAS_N.ALARMS.COMPUTER_DISCONNECT_A )
      I_Contact( "DB2120_MPP_ITC_IPC".RESET_FAULTS )
   END_RUNG wire#w1
   RUNG wire#w2
      Coil( "DB426_ALARMS_WARNINGS".ALARMS.UNIT_03.FACE_N_MEASURING."724462" )
   END_RUNG
   // the same network as SCL:
   "DB16000_OPC_UA_TRIGGER_ALARM".CLIENT.U3_MEAS_STA_MEAS_N.ALARMS.COMPUTER_DISCONNECT_A := ("DB16267_DISCONNECT_U3_MEAS_FACE_N".Error OR ("DB16000_OPC_UA_TRIGGER_ALARM".CLIENT.U3_MEAS_STA_MEAS_N.ALARMS.COMPUTER_DISCONNECT_A AND NOT "DB2120_MPP_ITC_IPC".RESET_FAULTS)) AND "DB7259_UNIT_3_STA_MEAS_B_ENABLE_DISABLE".ENABLED;
   "DB426_ALARMS_WARNINGS".ALARMS.UNIT_03.FACE_N_MEASURING."724462" := "DB16000_OPC_UA_TRIGGER_ALARM".CLIENT.U3_MEAS_STA_MEAS_N.ALARMS.COMPUTER_DISCONNECT_A;
END_REGION

REGION Network 40: UNIT 3 MEASURING STATION FACE N MEASURING METHOD CONNECTION ALARM
   RUNG wire#powerrail
      Contact( "DB16361_METHODCALL_U3_MEAS_B_MEAS_TRIGGER".Error )
      wire#w1
      Contact( "DB7259_UNIT_3_STA_MEAS_B_ENABLE_DISABLE".ENABLED )
      wire#w3
      Coil( "DB16000_OPC_UA_TRIGGER_ALARM".CLIENT.U3_MEAS_STA_MEAS_N.ALARMS.MEAS_CONNECTION_A )
   END_RUNG
   RUNG wire#powerrail
      Contact( "DB16000_OPC_UA_TRIGGER_ALARM".CLIENT.U3_MEAS_STA_MEAS_N.ALARMS.MEAS_CONNECTION_A )
      I_Contact( "DB2120_MPP_ITC_IPC".RESET_FAULTS )
      wire#w2
      I_Contact( "DB7300_INTERLOCK_GENERAL".GENERAL_MACHINE.FROM_CELL_TO_MACHINE_GENERAL.MEAS_STA_RESET )
   END_RUNG wire#w1
   RUNG wire#w2
      I_Contact( "DB2001_MODES_GENERAL".MG_AUX_OPTIONS.AUX_BOOL[0] )
   END_RUNG wire#w1
   RUNG wire#w3
      Coil( "DB426_ALARMS_WARNINGS".ALARMS.UNIT_03.FACE_N_MEASURING."724420" )
   END_RUNG
   // the same network as SCL:
   "DB16000_OPC_UA_TRIGGER_ALARM".CLIENT.U3_MEAS_STA_MEAS_N.ALARMS.MEAS_CONNECTION_A := ("DB16361_METHODCALL_U3_MEAS_B_MEAS_TRIGGER".Error OR ("DB16000_OPC_UA_TRIGGER_ALARM".CLIENT.U3_MEAS_STA_MEAS_N.ALARMS.MEAS_CONNECTION_A AND NOT "DB2120_MPP_ITC_IPC".RESET_FAULTS AND (NOT "DB7300_INTERLOCK_GENERAL".GENERAL_MACHINE.FROM_CELL_TO_MACHINE_GENERAL.MEAS_STA_RESET OR NOT "DB2001_MODES_GENERAL".MG_AUX_OPTIONS.AUX_BOOL[0]))) AND "DB7259_UNIT_3_STA_MEAS_B_ENABLE_DISABLE".ENABLED;
   "DB426_ALARMS_WARNINGS".ALARMS.UNIT_03.FACE_N_MEASURING."724420" := "DB16000_OPC_UA_TRIGGER_ALARM".CLIENT.U3_MEAS_STA_MEAS_N.ALARMS.MEAS_CONNECTION_A;
END_REGION

REGION Network 41: UNIT 3 MEASURING STATION FACE N MEASURING METHOD WORKING OR BLOCKED ALARM
   RUNG wire#powerrail
      Contact( "DB16361_METHODCALL_U3_MEAS_B_MEAS_TRIGGER".Done )
      I_Contact( "DB16007_U3_MEAS_STA_MEAS_B_CLIENT_INTERFACE".U03_FACE_B_MEAS_Method."Trigger analysis".Outputs.Result )
      wire#w1
      Contact( "DB7259_UNIT_3_STA_MEAS_B_ENABLE_DISABLE".ENABLED )
      wire#w3
      Coil( "DB16000_OPC_UA_TRIGGER_ALARM".CLIENT.U3_MEAS_STA_MEAS_N.ALARMS.MEAS_METHOD_WORKING_BLOCKED_A )
   END_RUNG
   RUNG wire#powerrail
      Contact( "DB16000_OPC_UA_TRIGGER_ALARM".CLIENT.U3_MEAS_STA_MEAS_N.ALARMS.MEAS_METHOD_WORKING_BLOCKED_A )
      I_Contact( "DB2120_MPP_ITC_IPC".RESET_FAULTS )
      wire#w2
      I_Contact( "DB7300_INTERLOCK_GENERAL".GENERAL_MACHINE.FROM_CELL_TO_MACHINE_GENERAL.MEAS_STA_RESET )
   END_RUNG wire#w1
   RUNG wire#w2
      I_Contact( "DB2001_MODES_GENERAL".MG_AUX_OPTIONS.AUX_BOOL[0] )
   END_RUNG wire#w1
   RUNG wire#w3
      Coil( "DB426_ALARMS_WARNINGS".ALARMS.UNIT_03.FACE_N_MEASURING."724421" )
   END_RUNG
   // the same network as SCL:
   "DB16000_OPC_UA_TRIGGER_ALARM".CLIENT.U3_MEAS_STA_MEAS_N.ALARMS.MEAS_METHOD_WORKING_BLOCKED_A := (("DB16361_METHODCALL_U3_MEAS_B_MEAS_TRIGGER".Done AND NOT "DB16007_U3_MEAS_STA_MEAS_B_CLIENT_INTERFACE".U03_FACE_B_MEAS_Method."Trigger analysis".Outputs.Result) OR ("DB16000_OPC_UA_TRIGGER_ALARM".CLIENT.U3_MEAS_STA_MEAS_N.ALARMS.MEAS_METHOD_WORKING_BLOCKED_A AND NOT "DB2120_MPP_ITC_IPC".RESET_FAULTS AND (NOT "DB7300_INTERLOCK_GENERAL".GENERAL_MACHINE.FROM_CELL_TO_MACHINE_GENERAL.MEAS_STA_RESET OR NOT "DB2001_MODES_GENERAL".MG_AUX_OPTIONS.AUX_BOOL[0]))) AND "DB7259_UNIT_3_STA_MEAS_B_ENABLE_DISABLE".ENABLED;
   "DB426_ALARMS_WARNINGS".ALARMS.UNIT_03.FACE_N_MEASURING."724421" := "DB16000_OPC_UA_TRIGGER_ALARM".CLIENT.U3_MEAS_STA_MEAS_N.ALARMS.MEAS_METHOD_WORKING_BLOCKED_A;
END_REGION

REGION Network 42: UNIT 3 MEASURING STATION FACE N CALIBRATING METHOD CONNECTION ALARM
   RUNG wire#powerrail
      Contact( "DB16365_METHODCALL_U3_MEAS_B_CALIBRATE_TRIGGER".Error )
      wire#w1
      Contact( "DB7259_UNIT_3_STA_MEAS_B_ENABLE_DISABLE".ENABLED )
      wire#w3
      Coil( "DB16000_OPC_UA_TRIGGER_ALARM".CLIENT.U3_MEAS_STA_MEAS_N.ALARMS.CALIBRATE_CONNECTION_A )
   END_RUNG
   RUNG wire#powerrail
      Contact( "DB16000_OPC_UA_TRIGGER_ALARM".CLIENT.U3_MEAS_STA_MEAS_N.ALARMS.CALIBRATE_CONNECTION_A )
      I_Contact( "DB2120_MPP_ITC_IPC".RESET_FAULTS )
      wire#w2
      I_Contact( "DB7300_INTERLOCK_GENERAL".GENERAL_MACHINE.FROM_CELL_TO_MACHINE_GENERAL.MEAS_STA_RESET )
   END_RUNG wire#w1
   RUNG wire#w2
      I_Contact( "DB2001_MODES_GENERAL".MG_AUX_OPTIONS.AUX_BOOL[0] )
   END_RUNG wire#w1
   RUNG wire#w3
      Coil( "DB426_ALARMS_WARNINGS".ALARMS.UNIT_03.FACE_N_MEASURING."724428" )
   END_RUNG
   // the same network as SCL:
   "DB16000_OPC_UA_TRIGGER_ALARM".CLIENT.U3_MEAS_STA_MEAS_N.ALARMS.CALIBRATE_CONNECTION_A := ("DB16365_METHODCALL_U3_MEAS_B_CALIBRATE_TRIGGER".Error OR ("DB16000_OPC_UA_TRIGGER_ALARM".CLIENT.U3_MEAS_STA_MEAS_N.ALARMS.CALIBRATE_CONNECTION_A AND NOT "DB2120_MPP_ITC_IPC".RESET_FAULTS AND (NOT "DB7300_INTERLOCK_GENERAL".GENERAL_MACHINE.FROM_CELL_TO_MACHINE_GENERAL.MEAS_STA_RESET OR NOT "DB2001_MODES_GENERAL".MG_AUX_OPTIONS.AUX_BOOL[0]))) AND "DB7259_UNIT_3_STA_MEAS_B_ENABLE_DISABLE".ENABLED;
   "DB426_ALARMS_WARNINGS".ALARMS.UNIT_03.FACE_N_MEASURING."724428" := "DB16000_OPC_UA_TRIGGER_ALARM".CLIENT.U3_MEAS_STA_MEAS_N.ALARMS.CALIBRATE_CONNECTION_A;
END_REGION

REGION Network 43: UNIT 3 MEASURING STATION FACE N CALIBRATING METHOD WORKING OR BLOCKED ALARM
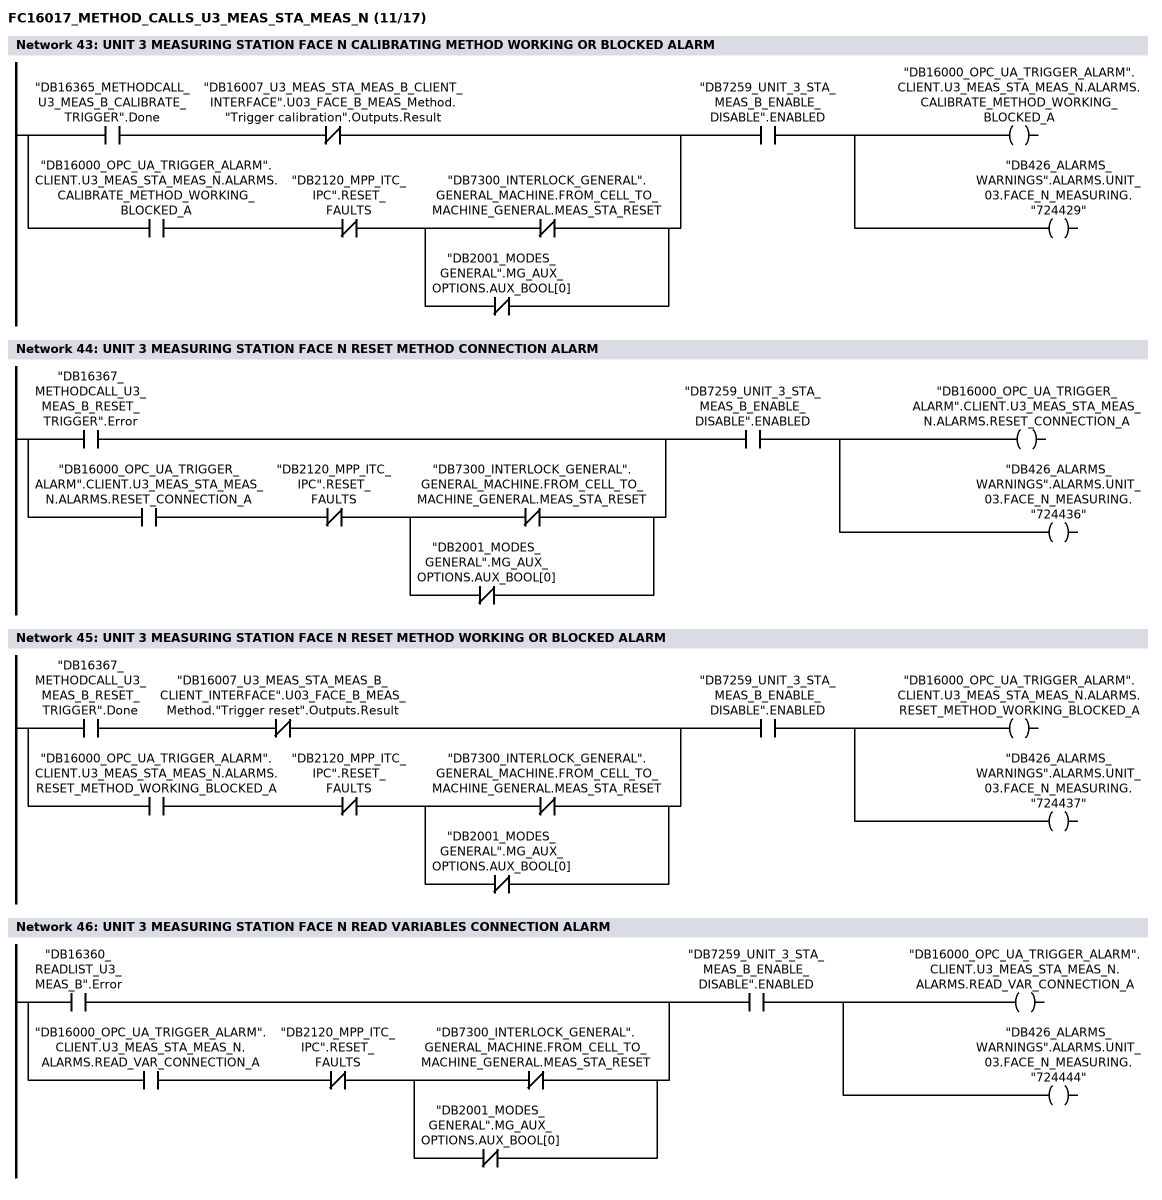
   RUNG wire#powerrail
      Contact( "DB16365_METHODCALL_U3_MEAS_B_CALIBRATE_TRIGGER".Done )
      I_Contact( "DB16007_U3_MEAS_STA_MEAS_B_CLIENT_INTERFACE".U03_FACE_B_MEAS_Method."Trigger calibration".Outputs.Result )
      wire#w1
      Contact( "DB7259_UNIT_3_STA_MEAS_B_ENABLE_DISABLE".ENABLED )
      wire#w3
      Coil( "DB16000_OPC_UA_TRIGGER_ALARM".CLIENT.U3_MEAS_STA_MEAS_N.ALARMS.CALIBRATE_METHOD_WORKING_BLOCKED_A )
   END_RUNG
   RUNG wire#powerrail
      Contact( "DB16000_OPC_UA_TRIGGER_ALARM".CLIENT.U3_MEAS_STA_MEAS_N.ALARMS.CALIBRATE_METHOD_WORKING_BLOCKED_A )
      I_Contact( "DB2120_MPP_ITC_IPC".RESET_FAULTS )
      wire#w2
      I_Contact( "DB7300_INTERLOCK_GENERAL".GENERAL_MACHINE.FROM_CELL_TO_MACHINE_GENERAL.MEAS_STA_RESET )
   END_RUNG wire#w1
   RUNG wire#w2
      I_Contact( "DB2001_MODES_GENERAL".MG_AUX_OPTIONS.AUX_BOOL[0] )
   END_RUNG wire#w1
   RUNG wire#w3
      Coil( "DB426_ALARMS_WARNINGS".ALARMS.UNIT_03.FACE_N_MEASURING."724429" )
   END_RUNG
   // the same network as SCL:
   "DB16000_OPC_UA_TRIGGER_ALARM".CLIENT.U3_MEAS_STA_MEAS_N.ALARMS.CALIBRATE_METHOD_WORKING_BLOCKED_A := (("DB16365_METHODCALL_U3_MEAS_B_CALIBRATE_TRIGGER".Done AND NOT "DB16007_U3_MEAS_STA_MEAS_B_CLIENT_INTERFACE".U03_FACE_B_MEAS_Method."Trigger calibration".Outputs.Result) OR ("DB16000_OPC_UA_TRIGGER_ALARM".CLIENT.U3_MEAS_STA_MEAS_N.ALARMS.CALIBRATE_METHOD_WORKING_BLOCKED_A AND NOT "DB2120_MPP_ITC_IPC".RESET_FAULTS AND (NOT "DB7300_INTERLOCK_GENERAL".GENERAL_MACHINE.FROM_CELL_TO_MACHINE_GENERAL.MEAS_STA_RESET OR NOT "DB2001_MODES_GENERAL".MG_AUX_OPTIONS.AUX_BOOL[0]))) AND "DB7259_UNIT_3_STA_MEAS_B_ENABLE_DISABLE".ENABLED;
   "DB426_ALARMS_WARNINGS".ALARMS.UNIT_03.FACE_N_MEASURING."724429" := "DB16000_OPC_UA_TRIGGER_ALARM".CLIENT.U3_MEAS_STA_MEAS_N.ALARMS.CALIBRATE_METHOD_WORKING_BLOCKED_A;
END_REGION

REGION Network 44: UNIT 3 MEASURING STATION FACE N RESET METHOD CONNECTION ALARM
   RUNG wire#powerrail
      Contact( "DB16367_METHODCALL_U3_MEAS_B_RESET_TRIGGER".Error )
      wire#w1
      Contact( "DB7259_UNIT_3_STA_MEAS_B_ENABLE_DISABLE".ENABLED )
      wire#w3
      Coil( "DB16000_OPC_UA_TRIGGER_ALARM".CLIENT.U3_MEAS_STA_MEAS_N.ALARMS.RESET_CONNECTION_A )
   END_RUNG
   RUNG wire#powerrail
      Contact( "DB16000_OPC_UA_TRIGGER_ALARM".CLIENT.U3_MEAS_STA_MEAS_N.ALARMS.RESET_CONNECTION_A )
      I_Contact( "DB2120_MPP_ITC_IPC".RESET_FAULTS )
      wire#w2
      I_Contact( "DB7300_INTERLOCK_GENERAL".GENERAL_MACHINE.FROM_CELL_TO_MACHINE_GENERAL.MEAS_STA_RESET )
   END_RUNG wire#w1
   RUNG wire#w2
      I_Contact( "DB2001_MODES_GENERAL".MG_AUX_OPTIONS.AUX_BOOL[0] )
   END_RUNG wire#w1
   RUNG wire#w3
      Coil( "DB426_ALARMS_WARNINGS".ALARMS.UNIT_03.FACE_N_MEASURING."724436" )
   END_RUNG
   // the same network as SCL:
   "DB16000_OPC_UA_TRIGGER_ALARM".CLIENT.U3_MEAS_STA_MEAS_N.ALARMS.RESET_CONNECTION_A := ("DB16367_METHODCALL_U3_MEAS_B_RESET_TRIGGER".Error OR ("DB16000_OPC_UA_TRIGGER_ALARM".CLIENT.U3_MEAS_STA_MEAS_N.ALARMS.RESET_CONNECTION_A AND NOT "DB2120_MPP_ITC_IPC".RESET_FAULTS AND (NOT "DB7300_INTERLOCK_GENERAL".GENERAL_MACHINE.FROM_CELL_TO_MACHINE_GENERAL.MEAS_STA_RESET OR NOT "DB2001_MODES_GENERAL".MG_AUX_OPTIONS.AUX_BOOL[0]))) AND "DB7259_UNIT_3_STA_MEAS_B_ENABLE_DISABLE".ENABLED;
   "DB426_ALARMS_WARNINGS".ALARMS.UNIT_03.FACE_N_MEASURING."724436" := "DB16000_OPC_UA_TRIGGER_ALARM".CLIENT.U3_MEAS_STA_MEAS_N.ALARMS.RESET_CONNECTION_A;
END_REGION

REGION Network 45: UNIT 3 MEASURING STATION FACE N RESET METHOD WORKING OR BLOCKED ALARM
   RUNG wire#powerrail
      Contact( "DB16367_METHODCALL_U3_MEAS_B_RESET_TRIGGER".Done )
      I_Contact( "DB16007_U3_MEAS_STA_MEAS_B_CLIENT_INTERFACE".U03_FACE_B_MEAS_Method."Trigger reset".Outputs.Result )
      wire#w1
      Contact( "DB7259_UNIT_3_STA_MEAS_B_ENABLE_DISABLE".ENABLED )
      wire#w3
      Coil( "DB16000_OPC_UA_TRIGGER_ALARM".CLIENT.U3_MEAS_STA_MEAS_N.ALARMS.RESET_METHOD_WORKING_BLOCKED_A )
   END_RUNG
   RUNG wire#powerrail
      Contact( "DB16000_OPC_UA_TRIGGER_ALARM".CLIENT.U3_MEAS_STA_MEAS_N.ALARMS.RESET_METHOD_WORKING_BLOCKED_A )
      I_Contact( "DB2120_MPP_ITC_IPC".RESET_FAULTS )
      wire#w2
      I_Contact( "DB7300_INTERLOCK_GENERAL".GENERAL_MACHINE.FROM_CELL_TO_MACHINE_GENERAL.MEAS_STA_RESET )
   END_RUNG wire#w1
   RUNG wire#w2
      I_Contact( "DB2001_MODES_GENERAL".MG_AUX_OPTIONS.AUX_BOOL[0] )
   END_RUNG wire#w1
   RUNG wire#w3
      Coil( "DB426_ALARMS_WARNINGS".ALARMS.UNIT_03.FACE_N_MEASURING."724437" )
   END_RUNG
   // the same network as SCL:
   "DB16000_OPC_UA_TRIGGER_ALARM".CLIENT.U3_MEAS_STA_MEAS_N.ALARMS.RESET_METHOD_WORKING_BLOCKED_A := (("DB16367_METHODCALL_U3_MEAS_B_RESET_TRIGGER".Done AND NOT "DB16007_U3_MEAS_STA_MEAS_B_CLIENT_INTERFACE".U03_FACE_B_MEAS_Method."Trigger reset".Outputs.Result) OR ("DB16000_OPC_UA_TRIGGER_ALARM".CLIENT.U3_MEAS_STA_MEAS_N.ALARMS.RESET_METHOD_WORKING_BLOCKED_A AND NOT "DB2120_MPP_ITC_IPC".RESET_FAULTS AND (NOT "DB7300_INTERLOCK_GENERAL".GENERAL_MACHINE.FROM_CELL_TO_MACHINE_GENERAL.MEAS_STA_RESET OR NOT "DB2001_MODES_GENERAL".MG_AUX_OPTIONS.AUX_BOOL[0]))) AND "DB7259_UNIT_3_STA_MEAS_B_ENABLE_DISABLE".ENABLED;
   "DB426_ALARMS_WARNINGS".ALARMS.UNIT_03.FACE_N_MEASURING."724437" := "DB16000_OPC_UA_TRIGGER_ALARM".CLIENT.U3_MEAS_STA_MEAS_N.ALARMS.RESET_METHOD_WORKING_BLOCKED_A;
END_REGION

REGION Network 46: UNIT 3 MEASURING STATION FACE N READ VARIABLES CONNECTION ALARM
   RUNG wire#powerrail
      Contact( "DB16360_READLIST_U3_MEAS_B".Error )
      wire#w1
      Contact( "DB7259_UNIT_3_STA_MEAS_B_ENABLE_DISABLE".ENABLED )
      wire#w3
      Coil( "DB16000_OPC_UA_TRIGGER_ALARM".CLIENT.U3_MEAS_STA_MEAS_N.ALARMS.READ_VAR_CONNECTION_A )
   END_RUNG
   RUNG wire#powerrail
      Contact( "DB16000_OPC_UA_TRIGGER_ALARM".CLIENT.U3_MEAS_STA_MEAS_N.ALARMS.READ_VAR_CONNECTION_A )
      I_Contact( "DB2120_MPP_ITC_IPC".RESET_FAULTS )
      wire#w2
      I_Contact( "DB7300_INTERLOCK_GENERAL".GENERAL_MACHINE.FROM_CELL_TO_MACHINE_GENERAL.MEAS_STA_RESET )
   END_RUNG wire#w1
   RUNG wire#w2
      I_Contact( "DB2001_MODES_GENERAL".MG_AUX_OPTIONS.AUX_BOOL[0] )
   END_RUNG wire#w1
   RUNG wire#w3
      Coil( "DB426_ALARMS_WARNINGS".ALARMS.UNIT_03.FACE_N_MEASURING."724444" )
   END_RUNG
   // the same network as SCL:
   "DB16000_OPC_UA_TRIGGER_ALARM".CLIENT.U3_MEAS_STA_MEAS_N.ALARMS.READ_VAR_CONNECTION_A := ("DB16360_READLIST_U3_MEAS_B".Error OR ("DB16000_OPC_UA_TRIGGER_ALARM".CLIENT.U3_MEAS_STA_MEAS_N.ALARMS.READ_VAR_CONNECTION_A AND NOT "DB2120_MPP_ITC_IPC".RESET_FAULTS AND (NOT "DB7300_INTERLOCK_GENERAL".GENERAL_MACHINE.FROM_CELL_TO_MACHINE_GENERAL.MEAS_STA_RESET OR NOT "DB2001_MODES_GENERAL".MG_AUX_OPTIONS.AUX_BOOL[0]))) AND "DB7259_UNIT_3_STA_MEAS_B_ENABLE_DISABLE".ENABLED;
   "DB426_ALARMS_WARNINGS".ALARMS.UNIT_03.FACE_N_MEASURING."724444" := "DB16000_OPC_UA_TRIGGER_ALARM".CLIENT.U3_MEAS_STA_MEAS_N.ALARMS.READ_VAR_CONNECTION_A;
END_REGION

REGION Network 47: UNIT 3 MEASURING STATION FACE N READ VARIABLES WORKING OR BLOCKED ALARM
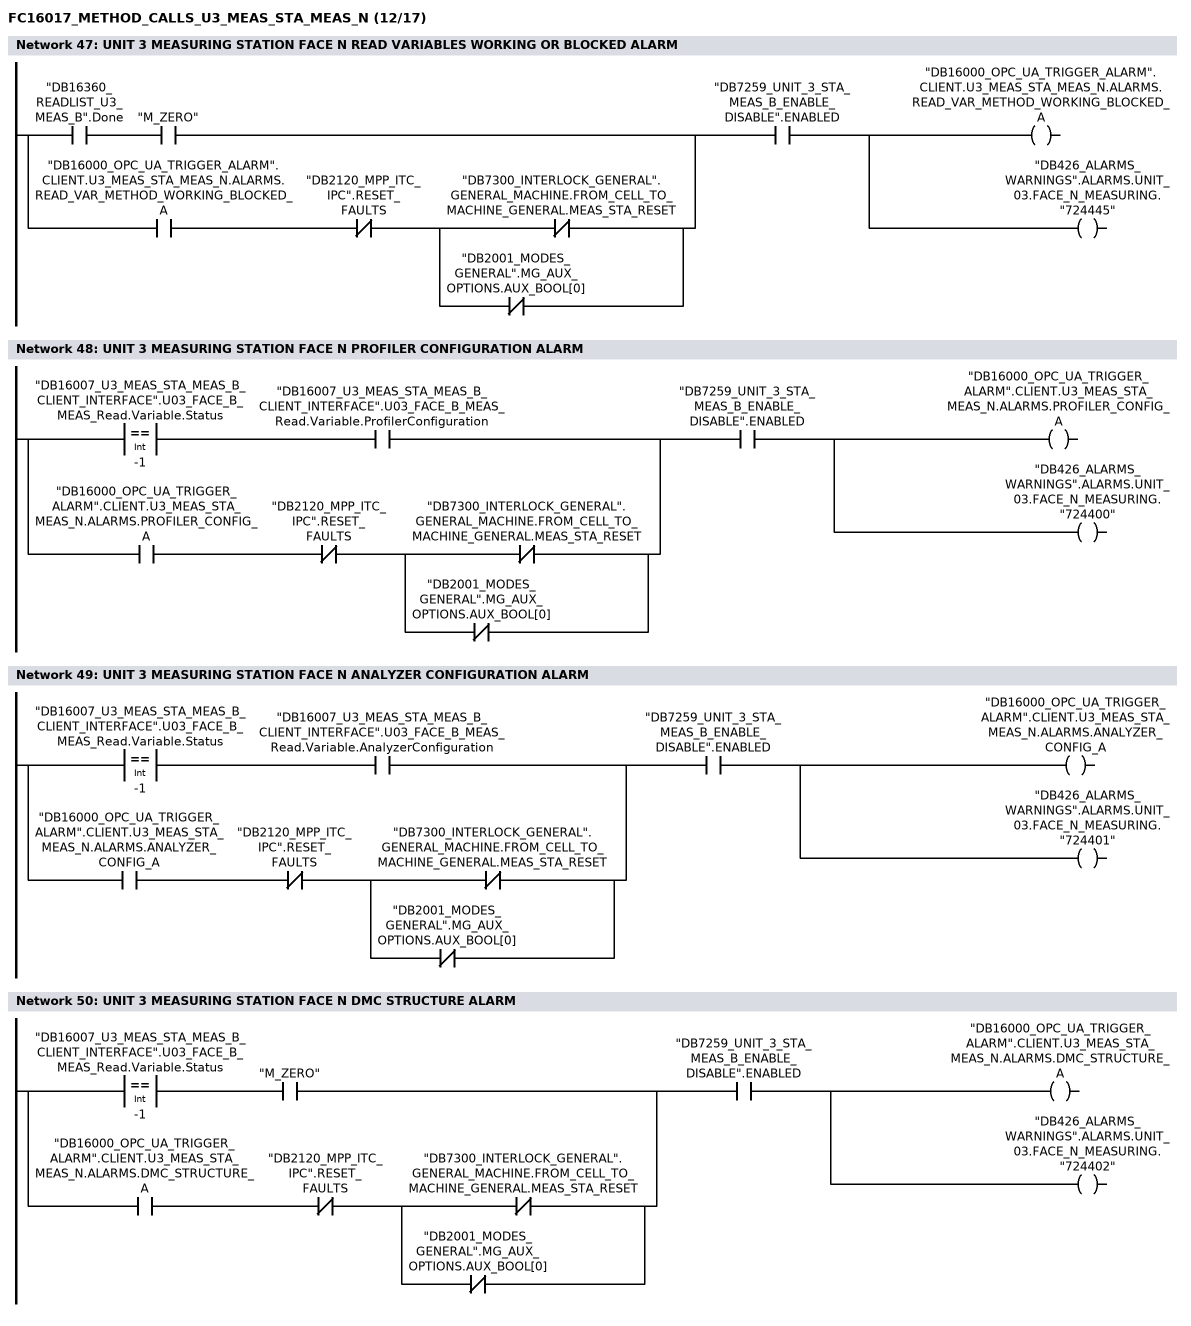
   RUNG wire#powerrail
      Contact( "DB16360_READLIST_U3_MEAS_B".Done )
      Contact( "M_ZERO" )
      wire#w1
      Contact( "DB7259_UNIT_3_STA_MEAS_B_ENABLE_DISABLE".ENABLED )
      wire#w3
      Coil( "DB16000_OPC_UA_TRIGGER_ALARM".CLIENT.U3_MEAS_STA_MEAS_N.ALARMS.READ_VAR_METHOD_WORKING_BLOCKED_A )
   END_RUNG
   RUNG wire#powerrail
      Contact( "DB16000_OPC_UA_TRIGGER_ALARM".CLIENT.U3_MEAS_STA_MEAS_N.ALARMS.READ_VAR_METHOD_WORKING_BLOCKED_A )
      I_Contact( "DB2120_MPP_ITC_IPC".RESET_FAULTS )
      wire#w2
      I_Contact( "DB7300_INTERLOCK_GENERAL".GENERAL_MACHINE.FROM_CELL_TO_MACHINE_GENERAL.MEAS_STA_RESET )
   END_RUNG wire#w1
   RUNG wire#w2
      I_Contact( "DB2001_MODES_GENERAL".MG_AUX_OPTIONS.AUX_BOOL[0] )
   END_RUNG wire#w1
   RUNG wire#w3
      Coil( "DB426_ALARMS_WARNINGS".ALARMS.UNIT_03.FACE_N_MEASURING."724445" )
   END_RUNG
   // the same network as SCL:
   "DB16000_OPC_UA_TRIGGER_ALARM".CLIENT.U3_MEAS_STA_MEAS_N.ALARMS.READ_VAR_METHOD_WORKING_BLOCKED_A := (("DB16360_READLIST_U3_MEAS_B".Done AND "M_ZERO") OR ("DB16000_OPC_UA_TRIGGER_ALARM".CLIENT.U3_MEAS_STA_MEAS_N.ALARMS.READ_VAR_METHOD_WORKING_BLOCKED_A AND NOT "DB2120_MPP_ITC_IPC".RESET_FAULTS AND (NOT "DB7300_INTERLOCK_GENERAL".GENERAL_MACHINE.FROM_CELL_TO_MACHINE_GENERAL.MEAS_STA_RESET OR NOT "DB2001_MODES_GENERAL".MG_AUX_OPTIONS.AUX_BOOL[0]))) AND "DB7259_UNIT_3_STA_MEAS_B_ENABLE_DISABLE".ENABLED;
   "DB426_ALARMS_WARNINGS".ALARMS.UNIT_03.FACE_N_MEASURING."724445" := "DB16000_OPC_UA_TRIGGER_ALARM".CLIENT.U3_MEAS_STA_MEAS_N.ALARMS.READ_VAR_METHOD_WORKING_BLOCKED_A;
END_REGION

REGION Network 48: UNIT 3 MEASURING STATION FACE N PROFILER CONFIGURATION ALARM
   RUNG wire#powerrail
      { S7_Templates := "SrcType := Int" } EQ_Contact(in1 := "DB16007_U3_MEAS_STA_MEAS_B_CLIENT_INTERFACE".U03_FACE_B_MEAS_Read.Variable.Status, in2 := -1)
      Contact( "DB16007_U3_MEAS_STA_MEAS_B_CLIENT_INTERFACE".U03_FACE_B_MEAS_Read.Variable.ProfilerConfiguration )
      wire#w1
      Contact( "DB7259_UNIT_3_STA_MEAS_B_ENABLE_DISABLE".ENABLED )
      wire#w3
      Coil( "DB16000_OPC_UA_TRIGGER_ALARM".CLIENT.U3_MEAS_STA_MEAS_N.ALARMS.PROFILER_CONFIG_A )
   END_RUNG
   RUNG wire#powerrail
      Contact( "DB16000_OPC_UA_TRIGGER_ALARM".CLIENT.U3_MEAS_STA_MEAS_N.ALARMS.PROFILER_CONFIG_A )
      I_Contact( "DB2120_MPP_ITC_IPC".RESET_FAULTS )
      wire#w2
      I_Contact( "DB7300_INTERLOCK_GENERAL".GENERAL_MACHINE.FROM_CELL_TO_MACHINE_GENERAL.MEAS_STA_RESET )
   END_RUNG wire#w1
   RUNG wire#w2
      I_Contact( "DB2001_MODES_GENERAL".MG_AUX_OPTIONS.AUX_BOOL[0] )
   END_RUNG wire#w1
   RUNG wire#w3
      Coil( "DB426_ALARMS_WARNINGS".ALARMS.UNIT_03.FACE_N_MEASURING."724400" )
   END_RUNG
   // the same network as SCL:
   "DB16000_OPC_UA_TRIGGER_ALARM".CLIENT.U3_MEAS_STA_MEAS_N.ALARMS.PROFILER_CONFIG_A := ((("DB16007_U3_MEAS_STA_MEAS_B_CLIENT_INTERFACE".U03_FACE_B_MEAS_Read.Variable.Status = (-1)) AND "DB16007_U3_MEAS_STA_MEAS_B_CLIENT_INTERFACE".U03_FACE_B_MEAS_Read.Variable.ProfilerConfiguration) OR ("DB16000_OPC_UA_TRIGGER_ALARM".CLIENT.U3_MEAS_STA_MEAS_N.ALARMS.PROFILER_CONFIG_A AND NOT "DB2120_MPP_ITC_IPC".RESET_FAULTS AND (NOT "DB7300_INTERLOCK_GENERAL".GENERAL_MACHINE.FROM_CELL_TO_MACHINE_GENERAL.MEAS_STA_RESET OR NOT "DB2001_MODES_GENERAL".MG_AUX_OPTIONS.AUX_BOOL[0]))) AND "DB7259_UNIT_3_STA_MEAS_B_ENABLE_DISABLE".ENABLED;
   "DB426_ALARMS_WARNINGS".ALARMS.UNIT_03.FACE_N_MEASURING."724400" := "DB16000_OPC_UA_TRIGGER_ALARM".CLIENT.U3_MEAS_STA_MEAS_N.ALARMS.PROFILER_CONFIG_A;
END_REGION

REGION Network 49: UNIT 3 MEASURING STATION FACE N ANALYZER CONFIGURATION ALARM
   RUNG wire#powerrail
      { S7_Templates := "SrcType := Int" } EQ_Contact(in1 := "DB16007_U3_MEAS_STA_MEAS_B_CLIENT_INTERFACE".U03_FACE_B_MEAS_Read.Variable.Status, in2 := -1)
      Contact( "DB16007_U3_MEAS_STA_MEAS_B_CLIENT_INTERFACE".U03_FACE_B_MEAS_Read.Variable.AnalyzerConfiguration )
      wire#w1
      Contact( "DB7259_UNIT_3_STA_MEAS_B_ENABLE_DISABLE".ENABLED )
      wire#w3
      Coil( "DB16000_OPC_UA_TRIGGER_ALARM".CLIENT.U3_MEAS_STA_MEAS_N.ALARMS.ANALYZER_CONFIG_A )
   END_RUNG
   RUNG wire#powerrail
      Contact( "DB16000_OPC_UA_TRIGGER_ALARM".CLIENT.U3_MEAS_STA_MEAS_N.ALARMS.ANALYZER_CONFIG_A )
      I_Contact( "DB2120_MPP_ITC_IPC".RESET_FAULTS )
      wire#w2
      I_Contact( "DB7300_INTERLOCK_GENERAL".GENERAL_MACHINE.FROM_CELL_TO_MACHINE_GENERAL.MEAS_STA_RESET )
   END_RUNG wire#w1
   RUNG wire#w2
      I_Contact( "DB2001_MODES_GENERAL".MG_AUX_OPTIONS.AUX_BOOL[0] )
   END_RUNG wire#w1
   RUNG wire#w3
      Coil( "DB426_ALARMS_WARNINGS".ALARMS.UNIT_03.FACE_N_MEASURING."724401" )
   END_RUNG
   // the same network as SCL:
   "DB16000_OPC_UA_TRIGGER_ALARM".CLIENT.U3_MEAS_STA_MEAS_N.ALARMS.ANALYZER_CONFIG_A := ((("DB16007_U3_MEAS_STA_MEAS_B_CLIENT_INTERFACE".U03_FACE_B_MEAS_Read.Variable.Status = (-1)) AND "DB16007_U3_MEAS_STA_MEAS_B_CLIENT_INTERFACE".U03_FACE_B_MEAS_Read.Variable.AnalyzerConfiguration) OR ("DB16000_OPC_UA_TRIGGER_ALARM".CLIENT.U3_MEAS_STA_MEAS_N.ALARMS.ANALYZER_CONFIG_A AND NOT "DB2120_MPP_ITC_IPC".RESET_FAULTS AND (NOT "DB7300_INTERLOCK_GENERAL".GENERAL_MACHINE.FROM_CELL_TO_MACHINE_GENERAL.MEAS_STA_RESET OR NOT "DB2001_MODES_GENERAL".MG_AUX_OPTIONS.AUX_BOOL[0]))) AND "DB7259_UNIT_3_STA_MEAS_B_ENABLE_DISABLE".ENABLED;
   "DB426_ALARMS_WARNINGS".ALARMS.UNIT_03.FACE_N_MEASURING."724401" := "DB16000_OPC_UA_TRIGGER_ALARM".CLIENT.U3_MEAS_STA_MEAS_N.ALARMS.ANALYZER_CONFIG_A;
END_REGION

REGION Network 50: UNIT 3 MEASURING STATION FACE N DMC STRUCTURE ALARM
   RUNG wire#powerrail
      { S7_Templates := "SrcType := Int" } EQ_Contact(in1 := "DB16007_U3_MEAS_STA_MEAS_B_CLIENT_INTERFACE".U03_FACE_B_MEAS_Read.Variable.Status, in2 := -1)
      Contact( "M_ZERO" )
      wire#w1
      Contact( "DB7259_UNIT_3_STA_MEAS_B_ENABLE_DISABLE".ENABLED )
      wire#w3
      Coil( "DB16000_OPC_UA_TRIGGER_ALARM".CLIENT.U3_MEAS_STA_MEAS_N.ALARMS.DMC_STRUCTURE_A )
   END_RUNG
   RUNG wire#powerrail
      Contact( "DB16000_OPC_UA_TRIGGER_ALARM".CLIENT.U3_MEAS_STA_MEAS_N.ALARMS.DMC_STRUCTURE_A )
      I_Contact( "DB2120_MPP_ITC_IPC".RESET_FAULTS )
      wire#w2
      I_Contact( "DB7300_INTERLOCK_GENERAL".GENERAL_MACHINE.FROM_CELL_TO_MACHINE_GENERAL.MEAS_STA_RESET )
   END_RUNG wire#w1
   RUNG wire#w2
      I_Contact( "DB2001_MODES_GENERAL".MG_AUX_OPTIONS.AUX_BOOL[0] )
   END_RUNG wire#w1
   RUNG wire#w3
      Coil( "DB426_ALARMS_WARNINGS".ALARMS.UNIT_03.FACE_N_MEASURING."724402" )
   END_RUNG
   // the same network as SCL:
   "DB16000_OPC_UA_TRIGGER_ALARM".CLIENT.U3_MEAS_STA_MEAS_N.ALARMS.DMC_STRUCTURE_A := ((("DB16007_U3_MEAS_STA_MEAS_B_CLIENT_INTERFACE".U03_FACE_B_MEAS_Read.Variable.Status = (-1)) AND "M_ZERO") OR ("DB16000_OPC_UA_TRIGGER_ALARM".CLIENT.U3_MEAS_STA_MEAS_N.ALARMS.DMC_STRUCTURE_A AND NOT "DB2120_MPP_ITC_IPC".RESET_FAULTS AND (NOT "DB7300_INTERLOCK_GENERAL".GENERAL_MACHINE.FROM_CELL_TO_MACHINE_GENERAL.MEAS_STA_RESET OR NOT "DB2001_MODES_GENERAL".MG_AUX_OPTIONS.AUX_BOOL[0]))) AND "DB7259_UNIT_3_STA_MEAS_B_ENABLE_DISABLE".ENABLED;
   "DB426_ALARMS_WARNINGS".ALARMS.UNIT_03.FACE_N_MEASURING."724402" := "DB16000_OPC_UA_TRIGGER_ALARM".CLIENT.U3_MEAS_STA_MEAS_N.ALARMS.DMC_STRUCTURE_A;
END_REGION

REGION Network 51: UNIT 3 MEASURING STATION FACE N ACQUISITON ALARM
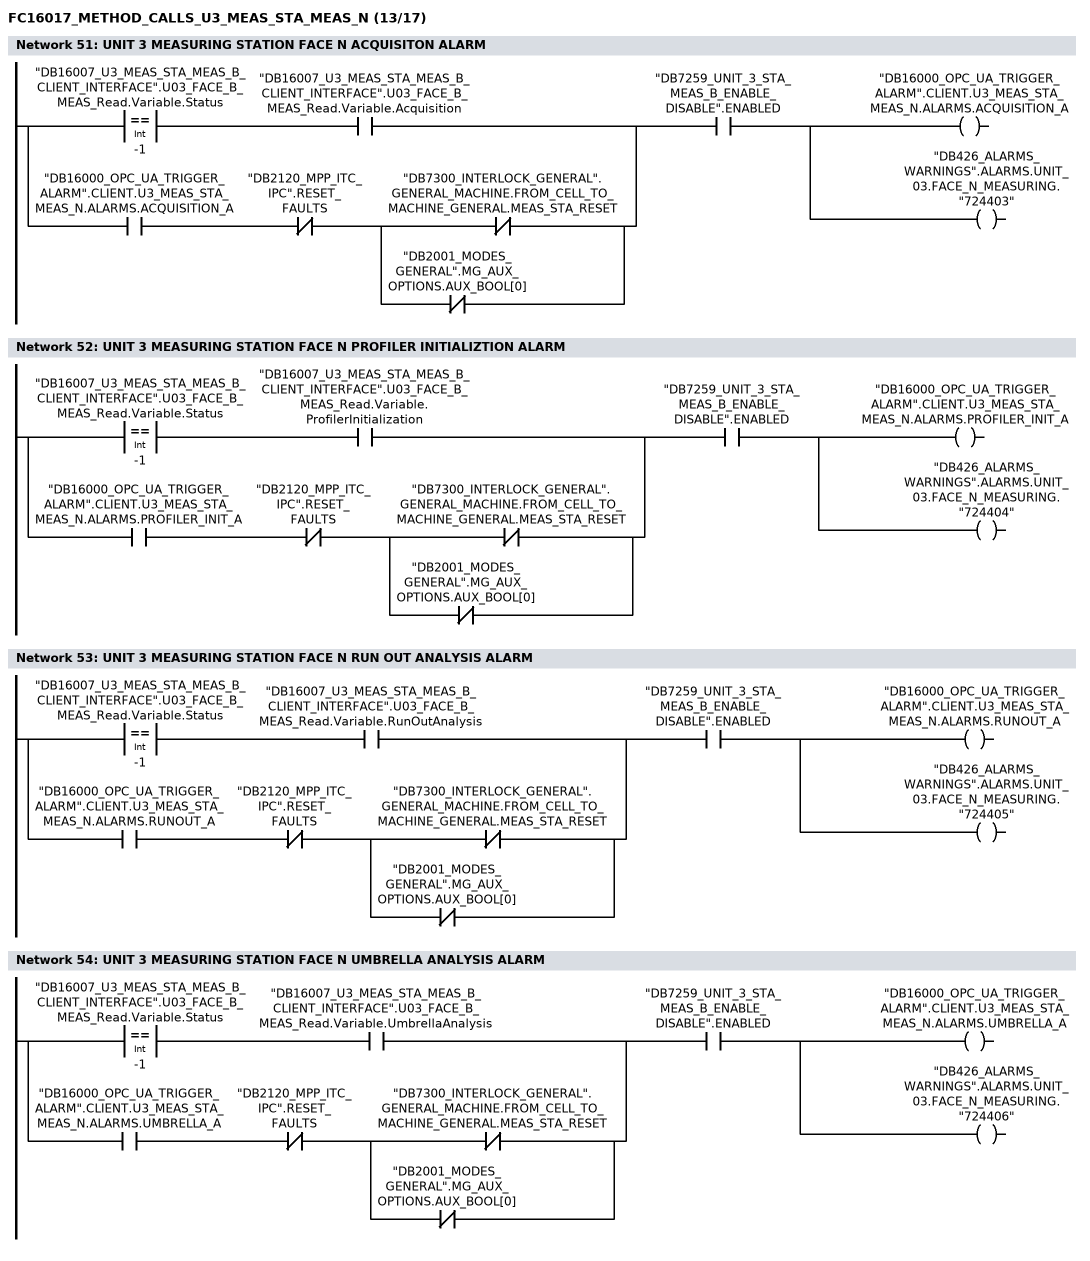
   RUNG wire#powerrail
      { S7_Templates := "SrcType := Int" } EQ_Contact(in1 := "DB16007_U3_MEAS_STA_MEAS_B_CLIENT_INTERFACE".U03_FACE_B_MEAS_Read.Variable.Status, in2 := -1)
      Contact( "DB16007_U3_MEAS_STA_MEAS_B_CLIENT_INTERFACE".U03_FACE_B_MEAS_Read.Variable.Acquisition )
      wire#w1
      Contact( "DB7259_UNIT_3_STA_MEAS_B_ENABLE_DISABLE".ENABLED )
      wire#w3
      Coil( "DB16000_OPC_UA_TRIGGER_ALARM".CLIENT.U3_MEAS_STA_MEAS_N.ALARMS.ACQUISITION_A )
   END_RUNG
   RUNG wire#powerrail
      Contact( "DB16000_OPC_UA_TRIGGER_ALARM".CLIENT.U3_MEAS_STA_MEAS_N.ALARMS.ACQUISITION_A )
      I_Contact( "DB2120_MPP_ITC_IPC".RESET_FAULTS )
      wire#w2
      I_Contact( "DB7300_INTERLOCK_GENERAL".GENERAL_MACHINE.FROM_CELL_TO_MACHINE_GENERAL.MEAS_STA_RESET )
   END_RUNG wire#w1
   RUNG wire#w2
      I_Contact( "DB2001_MODES_GENERAL".MG_AUX_OPTIONS.AUX_BOOL[0] )
   END_RUNG wire#w1
   RUNG wire#w3
      Coil( "DB426_ALARMS_WARNINGS".ALARMS.UNIT_03.FACE_N_MEASURING."724403" )
   END_RUNG
   // the same network as SCL:
   "DB16000_OPC_UA_TRIGGER_ALARM".CLIENT.U3_MEAS_STA_MEAS_N.ALARMS.ACQUISITION_A := ((("DB16007_U3_MEAS_STA_MEAS_B_CLIENT_INTERFACE".U03_FACE_B_MEAS_Read.Variable.Status = (-1)) AND "DB16007_U3_MEAS_STA_MEAS_B_CLIENT_INTERFACE".U03_FACE_B_MEAS_Read.Variable.Acquisition) OR ("DB16000_OPC_UA_TRIGGER_ALARM".CLIENT.U3_MEAS_STA_MEAS_N.ALARMS.ACQUISITION_A AND NOT "DB2120_MPP_ITC_IPC".RESET_FAULTS AND (NOT "DB7300_INTERLOCK_GENERAL".GENERAL_MACHINE.FROM_CELL_TO_MACHINE_GENERAL.MEAS_STA_RESET OR NOT "DB2001_MODES_GENERAL".MG_AUX_OPTIONS.AUX_BOOL[0]))) AND "DB7259_UNIT_3_STA_MEAS_B_ENABLE_DISABLE".ENABLED;
   "DB426_ALARMS_WARNINGS".ALARMS.UNIT_03.FACE_N_MEASURING."724403" := "DB16000_OPC_UA_TRIGGER_ALARM".CLIENT.U3_MEAS_STA_MEAS_N.ALARMS.ACQUISITION_A;
END_REGION

REGION Network 52: UNIT 3 MEASURING STATION FACE N PROFILER INITIALIZTION ALARM
   RUNG wire#powerrail
      { S7_Templates := "SrcType := Int" } EQ_Contact(in1 := "DB16007_U3_MEAS_STA_MEAS_B_CLIENT_INTERFACE".U03_FACE_B_MEAS_Read.Variable.Status, in2 := -1)
      Contact( "DB16007_U3_MEAS_STA_MEAS_B_CLIENT_INTERFACE".U03_FACE_B_MEAS_Read.Variable.ProfilerInitialization )
      wire#w1
      Contact( "DB7259_UNIT_3_STA_MEAS_B_ENABLE_DISABLE".ENABLED )
      wire#w3
      Coil( "DB16000_OPC_UA_TRIGGER_ALARM".CLIENT.U3_MEAS_STA_MEAS_N.ALARMS.PROFILER_INIT_A )
   END_RUNG
   RUNG wire#powerrail
      Contact( "DB16000_OPC_UA_TRIGGER_ALARM".CLIENT.U3_MEAS_STA_MEAS_N.ALARMS.PROFILER_INIT_A )
      I_Contact( "DB2120_MPP_ITC_IPC".RESET_FAULTS )
      wire#w2
      I_Contact( "DB7300_INTERLOCK_GENERAL".GENERAL_MACHINE.FROM_CELL_TO_MACHINE_GENERAL.MEAS_STA_RESET )
   END_RUNG wire#w1
   RUNG wire#w2
      I_Contact( "DB2001_MODES_GENERAL".MG_AUX_OPTIONS.AUX_BOOL[0] )
   END_RUNG wire#w1
   RUNG wire#w3
      Coil( "DB426_ALARMS_WARNINGS".ALARMS.UNIT_03.FACE_N_MEASURING."724404" )
   END_RUNG
   // the same network as SCL:
   "DB16000_OPC_UA_TRIGGER_ALARM".CLIENT.U3_MEAS_STA_MEAS_N.ALARMS.PROFILER_INIT_A := ((("DB16007_U3_MEAS_STA_MEAS_B_CLIENT_INTERFACE".U03_FACE_B_MEAS_Read.Variable.Status = (-1)) AND "DB16007_U3_MEAS_STA_MEAS_B_CLIENT_INTERFACE".U03_FACE_B_MEAS_Read.Variable.ProfilerInitialization) OR ("DB16000_OPC_UA_TRIGGER_ALARM".CLIENT.U3_MEAS_STA_MEAS_N.ALARMS.PROFILER_INIT_A AND NOT "DB2120_MPP_ITC_IPC".RESET_FAULTS AND (NOT "DB7300_INTERLOCK_GENERAL".GENERAL_MACHINE.FROM_CELL_TO_MACHINE_GENERAL.MEAS_STA_RESET OR NOT "DB2001_MODES_GENERAL".MG_AUX_OPTIONS.AUX_BOOL[0]))) AND "DB7259_UNIT_3_STA_MEAS_B_ENABLE_DISABLE".ENABLED;
   "DB426_ALARMS_WARNINGS".ALARMS.UNIT_03.FACE_N_MEASURING."724404" := "DB16000_OPC_UA_TRIGGER_ALARM".CLIENT.U3_MEAS_STA_MEAS_N.ALARMS.PROFILER_INIT_A;
END_REGION

REGION Network 53: UNIT 3 MEASURING STATION FACE N RUN OUT ANALYSIS ALARM
   RUNG wire#powerrail
      { S7_Templates := "SrcType := Int" } EQ_Contact(in1 := "DB16007_U3_MEAS_STA_MEAS_B_CLIENT_INTERFACE".U03_FACE_B_MEAS_Read.Variable.Status, in2 := -1)
      Contact( "DB16007_U3_MEAS_STA_MEAS_B_CLIENT_INTERFACE".U03_FACE_B_MEAS_Read.Variable.RunOutAnalysis )
      wire#w1
      Contact( "DB7259_UNIT_3_STA_MEAS_B_ENABLE_DISABLE".ENABLED )
      wire#w3
      Coil( "DB16000_OPC_UA_TRIGGER_ALARM".CLIENT.U3_MEAS_STA_MEAS_N.ALARMS.RUNOUT_A )
   END_RUNG
   RUNG wire#powerrail
      Contact( "DB16000_OPC_UA_TRIGGER_ALARM".CLIENT.U3_MEAS_STA_MEAS_N.ALARMS.RUNOUT_A )
      I_Contact( "DB2120_MPP_ITC_IPC".RESET_FAULTS )
      wire#w2
      I_Contact( "DB7300_INTERLOCK_GENERAL".GENERAL_MACHINE.FROM_CELL_TO_MACHINE_GENERAL.MEAS_STA_RESET )
   END_RUNG wire#w1
   RUNG wire#w2
      I_Contact( "DB2001_MODES_GENERAL".MG_AUX_OPTIONS.AUX_BOOL[0] )
   END_RUNG wire#w1
   RUNG wire#w3
      Coil( "DB426_ALARMS_WARNINGS".ALARMS.UNIT_03.FACE_N_MEASURING."724405" )
   END_RUNG
   // the same network as SCL:
   "DB16000_OPC_UA_TRIGGER_ALARM".CLIENT.U3_MEAS_STA_MEAS_N.ALARMS.RUNOUT_A := ((("DB16007_U3_MEAS_STA_MEAS_B_CLIENT_INTERFACE".U03_FACE_B_MEAS_Read.Variable.Status = (-1)) AND "DB16007_U3_MEAS_STA_MEAS_B_CLIENT_INTERFACE".U03_FACE_B_MEAS_Read.Variable.RunOutAnalysis) OR ("DB16000_OPC_UA_TRIGGER_ALARM".CLIENT.U3_MEAS_STA_MEAS_N.ALARMS.RUNOUT_A AND NOT "DB2120_MPP_ITC_IPC".RESET_FAULTS AND (NOT "DB7300_INTERLOCK_GENERAL".GENERAL_MACHINE.FROM_CELL_TO_MACHINE_GENERAL.MEAS_STA_RESET OR NOT "DB2001_MODES_GENERAL".MG_AUX_OPTIONS.AUX_BOOL[0]))) AND "DB7259_UNIT_3_STA_MEAS_B_ENABLE_DISABLE".ENABLED;
   "DB426_ALARMS_WARNINGS".ALARMS.UNIT_03.FACE_N_MEASURING."724405" := "DB16000_OPC_UA_TRIGGER_ALARM".CLIENT.U3_MEAS_STA_MEAS_N.ALARMS.RUNOUT_A;
END_REGION

REGION Network 54: UNIT 3 MEASURING STATION FACE N UMBRELLA ANALYSIS ALARM
   RUNG wire#powerrail
      { S7_Templates := "SrcType := Int" } EQ_Contact(in1 := "DB16007_U3_MEAS_STA_MEAS_B_CLIENT_INTERFACE".U03_FACE_B_MEAS_Read.Variable.Status, in2 := -1)
      Contact( "DB16007_U3_MEAS_STA_MEAS_B_CLIENT_INTERFACE".U03_FACE_B_MEAS_Read.Variable.UmbrellaAnalysis )
      wire#w1
      Contact( "DB7259_UNIT_3_STA_MEAS_B_ENABLE_DISABLE".ENABLED )
      wire#w3
      Coil( "DB16000_OPC_UA_TRIGGER_ALARM".CLIENT.U3_MEAS_STA_MEAS_N.ALARMS.UMBRELLA_A )
   END_RUNG
   RUNG wire#powerrail
      Contact( "DB16000_OPC_UA_TRIGGER_ALARM".CLIENT.U3_MEAS_STA_MEAS_N.ALARMS.UMBRELLA_A )
      I_Contact( "DB2120_MPP_ITC_IPC".RESET_FAULTS )
      wire#w2
      I_Contact( "DB7300_INTERLOCK_GENERAL".GENERAL_MACHINE.FROM_CELL_TO_MACHINE_GENERAL.MEAS_STA_RESET )
   END_RUNG wire#w1
   RUNG wire#w2
      I_Contact( "DB2001_MODES_GENERAL".MG_AUX_OPTIONS.AUX_BOOL[0] )
   END_RUNG wire#w1
   RUNG wire#w3
      Coil( "DB426_ALARMS_WARNINGS".ALARMS.UNIT_03.FACE_N_MEASURING."724406" )
   END_RUNG
   // the same network as SCL:
   "DB16000_OPC_UA_TRIGGER_ALARM".CLIENT.U3_MEAS_STA_MEAS_N.ALARMS.UMBRELLA_A := ((("DB16007_U3_MEAS_STA_MEAS_B_CLIENT_INTERFACE".U03_FACE_B_MEAS_Read.Variable.Status = (-1)) AND "DB16007_U3_MEAS_STA_MEAS_B_CLIENT_INTERFACE".U03_FACE_B_MEAS_Read.Variable.UmbrellaAnalysis) OR ("DB16000_OPC_UA_TRIGGER_ALARM".CLIENT.U3_MEAS_STA_MEAS_N.ALARMS.UMBRELLA_A AND NOT "DB2120_MPP_ITC_IPC".RESET_FAULTS AND (NOT "DB7300_INTERLOCK_GENERAL".GENERAL_MACHINE.FROM_CELL_TO_MACHINE_GENERAL.MEAS_STA_RESET OR NOT "DB2001_MODES_GENERAL".MG_AUX_OPTIONS.AUX_BOOL[0]))) AND "DB7259_UNIT_3_STA_MEAS_B_ENABLE_DISABLE".ENABLED;
   "DB426_ALARMS_WARNINGS".ALARMS.UNIT_03.FACE_N_MEASURING."724406" := "DB16000_OPC_UA_TRIGGER_ALARM".CLIENT.U3_MEAS_STA_MEAS_N.ALARMS.UMBRELLA_A;
END_REGION

REGION Network 55: UNIT 3 MEASURING STATION FACE N LAYER GROWTH ANALYSIS ALARM
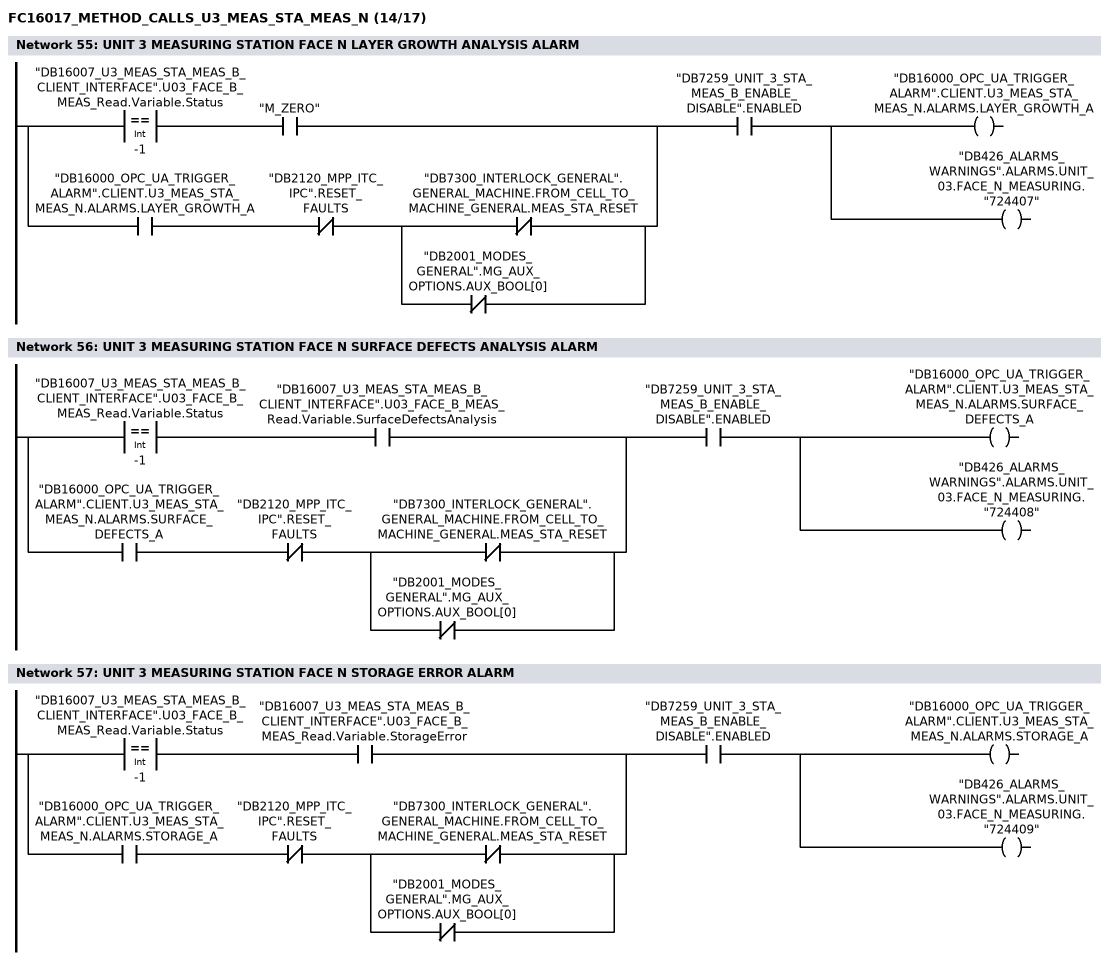
   RUNG wire#powerrail
      { S7_Templates := "SrcType := Int" } EQ_Contact(in1 := "DB16007_U3_MEAS_STA_MEAS_B_CLIENT_INTERFACE".U03_FACE_B_MEAS_Read.Variable.Status, in2 := -1)
      Contact( "M_ZERO" )
      wire#w1
      Contact( "DB7259_UNIT_3_STA_MEAS_B_ENABLE_DISABLE".ENABLED )
      wire#w3
      Coil( "DB16000_OPC_UA_TRIGGER_ALARM".CLIENT.U3_MEAS_STA_MEAS_N.ALARMS.LAYER_GROWTH_A )
   END_RUNG
   RUNG wire#powerrail
      Contact( "DB16000_OPC_UA_TRIGGER_ALARM".CLIENT.U3_MEAS_STA_MEAS_N.ALARMS.LAYER_GROWTH_A )
      I_Contact( "DB2120_MPP_ITC_IPC".RESET_FAULTS )
      wire#w2
      I_Contact( "DB7300_INTERLOCK_GENERAL".GENERAL_MACHINE.FROM_CELL_TO_MACHINE_GENERAL.MEAS_STA_RESET )
   END_RUNG wire#w1
   RUNG wire#w2
      I_Contact( "DB2001_MODES_GENERAL".MG_AUX_OPTIONS.AUX_BOOL[0] )
   END_RUNG wire#w1
   RUNG wire#w3
      Coil( "DB426_ALARMS_WARNINGS".ALARMS.UNIT_03.FACE_N_MEASURING."724407" )
   END_RUNG
   // the same network as SCL:
   "DB16000_OPC_UA_TRIGGER_ALARM".CLIENT.U3_MEAS_STA_MEAS_N.ALARMS.LAYER_GROWTH_A := ((("DB16007_U3_MEAS_STA_MEAS_B_CLIENT_INTERFACE".U03_FACE_B_MEAS_Read.Variable.Status = (-1)) AND "M_ZERO") OR ("DB16000_OPC_UA_TRIGGER_ALARM".CLIENT.U3_MEAS_STA_MEAS_N.ALARMS.LAYER_GROWTH_A AND NOT "DB2120_MPP_ITC_IPC".RESET_FAULTS AND (NOT "DB7300_INTERLOCK_GENERAL".GENERAL_MACHINE.FROM_CELL_TO_MACHINE_GENERAL.MEAS_STA_RESET OR NOT "DB2001_MODES_GENERAL".MG_AUX_OPTIONS.AUX_BOOL[0]))) AND "DB7259_UNIT_3_STA_MEAS_B_ENABLE_DISABLE".ENABLED;
   "DB426_ALARMS_WARNINGS".ALARMS.UNIT_03.FACE_N_MEASURING."724407" := "DB16000_OPC_UA_TRIGGER_ALARM".CLIENT.U3_MEAS_STA_MEAS_N.ALARMS.LAYER_GROWTH_A;
END_REGION

REGION Network 56: UNIT 3 MEASURING STATION FACE N SURFACE DEFECTS ANALYSIS ALARM
   RUNG wire#powerrail
      { S7_Templates := "SrcType := Int" } EQ_Contact(in1 := "DB16007_U3_MEAS_STA_MEAS_B_CLIENT_INTERFACE".U03_FACE_B_MEAS_Read.Variable.Status, in2 := -1)
      Contact( "DB16007_U3_MEAS_STA_MEAS_B_CLIENT_INTERFACE".U03_FACE_B_MEAS_Read.Variable.SurfaceDefectsAnalysis )
      wire#w1
      Contact( "DB7259_UNIT_3_STA_MEAS_B_ENABLE_DISABLE".ENABLED )
      wire#w3
      Coil( "DB16000_OPC_UA_TRIGGER_ALARM".CLIENT.U3_MEAS_STA_MEAS_N.ALARMS.SURFACE_DEFECTS_A )
   END_RUNG
   RUNG wire#powerrail
      Contact( "DB16000_OPC_UA_TRIGGER_ALARM".CLIENT.U3_MEAS_STA_MEAS_N.ALARMS.SURFACE_DEFECTS_A )
      I_Contact( "DB2120_MPP_ITC_IPC".RESET_FAULTS )
      wire#w2
      I_Contact( "DB7300_INTERLOCK_GENERAL".GENERAL_MACHINE.FROM_CELL_TO_MACHINE_GENERAL.MEAS_STA_RESET )
   END_RUNG wire#w1
   RUNG wire#w2
      I_Contact( "DB2001_MODES_GENERAL".MG_AUX_OPTIONS.AUX_BOOL[0] )
   END_RUNG wire#w1
   RUNG wire#w3
      Coil( "DB426_ALARMS_WARNINGS".ALARMS.UNIT_03.FACE_N_MEASURING."724408" )
   END_RUNG
   // the same network as SCL:
   "DB16000_OPC_UA_TRIGGER_ALARM".CLIENT.U3_MEAS_STA_MEAS_N.ALARMS.SURFACE_DEFECTS_A := ((("DB16007_U3_MEAS_STA_MEAS_B_CLIENT_INTERFACE".U03_FACE_B_MEAS_Read.Variable.Status = (-1)) AND "DB16007_U3_MEAS_STA_MEAS_B_CLIENT_INTERFACE".U03_FACE_B_MEAS_Read.Variable.SurfaceDefectsAnalysis) OR ("DB16000_OPC_UA_TRIGGER_ALARM".CLIENT.U3_MEAS_STA_MEAS_N.ALARMS.SURFACE_DEFECTS_A AND NOT "DB2120_MPP_ITC_IPC".RESET_FAULTS AND (NOT "DB7300_INTERLOCK_GENERAL".GENERAL_MACHINE.FROM_CELL_TO_MACHINE_GENERAL.MEAS_STA_RESET OR NOT "DB2001_MODES_GENERAL".MG_AUX_OPTIONS.AUX_BOOL[0]))) AND "DB7259_UNIT_3_STA_MEAS_B_ENABLE_DISABLE".ENABLED;
   "DB426_ALARMS_WARNINGS".ALARMS.UNIT_03.FACE_N_MEASURING."724408" := "DB16000_OPC_UA_TRIGGER_ALARM".CLIENT.U3_MEAS_STA_MEAS_N.ALARMS.SURFACE_DEFECTS_A;
END_REGION

REGION Network 57: UNIT 3 MEASURING STATION FACE N STORAGE ERROR ALARM
   RUNG wire#powerrail
      { S7_Templates := "SrcType := Int" } EQ_Contact(in1 := "DB16007_U3_MEAS_STA_MEAS_B_CLIENT_INTERFACE".U03_FACE_B_MEAS_Read.Variable.Status, in2 := -1)
      Contact( "DB16007_U3_MEAS_STA_MEAS_B_CLIENT_INTERFACE".U03_FACE_B_MEAS_Read.Variable.StorageError )
      wire#w1
      Contact( "DB7259_UNIT_3_STA_MEAS_B_ENABLE_DISABLE".ENABLED )
      wire#w3
      Coil( "DB16000_OPC_UA_TRIGGER_ALARM".CLIENT.U3_MEAS_STA_MEAS_N.ALARMS.STORAGE_A )
   END_RUNG
   RUNG wire#powerrail
      Contact( "DB16000_OPC_UA_TRIGGER_ALARM".CLIENT.U3_MEAS_STA_MEAS_N.ALARMS.STORAGE_A )
      I_Contact( "DB2120_MPP_ITC_IPC".RESET_FAULTS )
      wire#w2
      I_Contact( "DB7300_INTERLOCK_GENERAL".GENERAL_MACHINE.FROM_CELL_TO_MACHINE_GENERAL.MEAS_STA_RESET )
   END_RUNG wire#w1
   RUNG wire#w2
      I_Contact( "DB2001_MODES_GENERAL".MG_AUX_OPTIONS.AUX_BOOL[0] )
   END_RUNG wire#w1
   RUNG wire#w3
      Coil( "DB426_ALARMS_WARNINGS".ALARMS.UNIT_03.FACE_N_MEASURING."724409" )
   END_RUNG
   // the same network as SCL:
   "DB16000_OPC_UA_TRIGGER_ALARM".CLIENT.U3_MEAS_STA_MEAS_N.ALARMS.STORAGE_A := ((("DB16007_U3_MEAS_STA_MEAS_B_CLIENT_INTERFACE".U03_FACE_B_MEAS_Read.Variable.Status = (-1)) AND "DB16007_U3_MEAS_STA_MEAS_B_CLIENT_INTERFACE".U03_FACE_B_MEAS_Read.Variable.StorageError) OR ("DB16000_OPC_UA_TRIGGER_ALARM".CLIENT.U3_MEAS_STA_MEAS_N.ALARMS.STORAGE_A AND NOT "DB2120_MPP_ITC_IPC".RESET_FAULTS AND (NOT "DB7300_INTERLOCK_GENERAL".GENERAL_MACHINE.FROM_CELL_TO_MACHINE_GENERAL.MEAS_STA_RESET OR NOT "DB2001_MODES_GENERAL".MG_AUX_OPTIONS.AUX_BOOL[0]))) AND "DB7259_UNIT_3_STA_MEAS_B_ENABLE_DISABLE".ENABLED;
   "DB426_ALARMS_WARNINGS".ALARMS.UNIT_03.FACE_N_MEASURING."724409" := "DB16000_OPC_UA_TRIGGER_ALARM".CLIENT.U3_MEAS_STA_MEAS_N.ALARMS.STORAGE_A;
END_REGION

REGION Network 58: UNIT 3 MEASURING STATION FACE N MISSING CALIBRATION ALARM
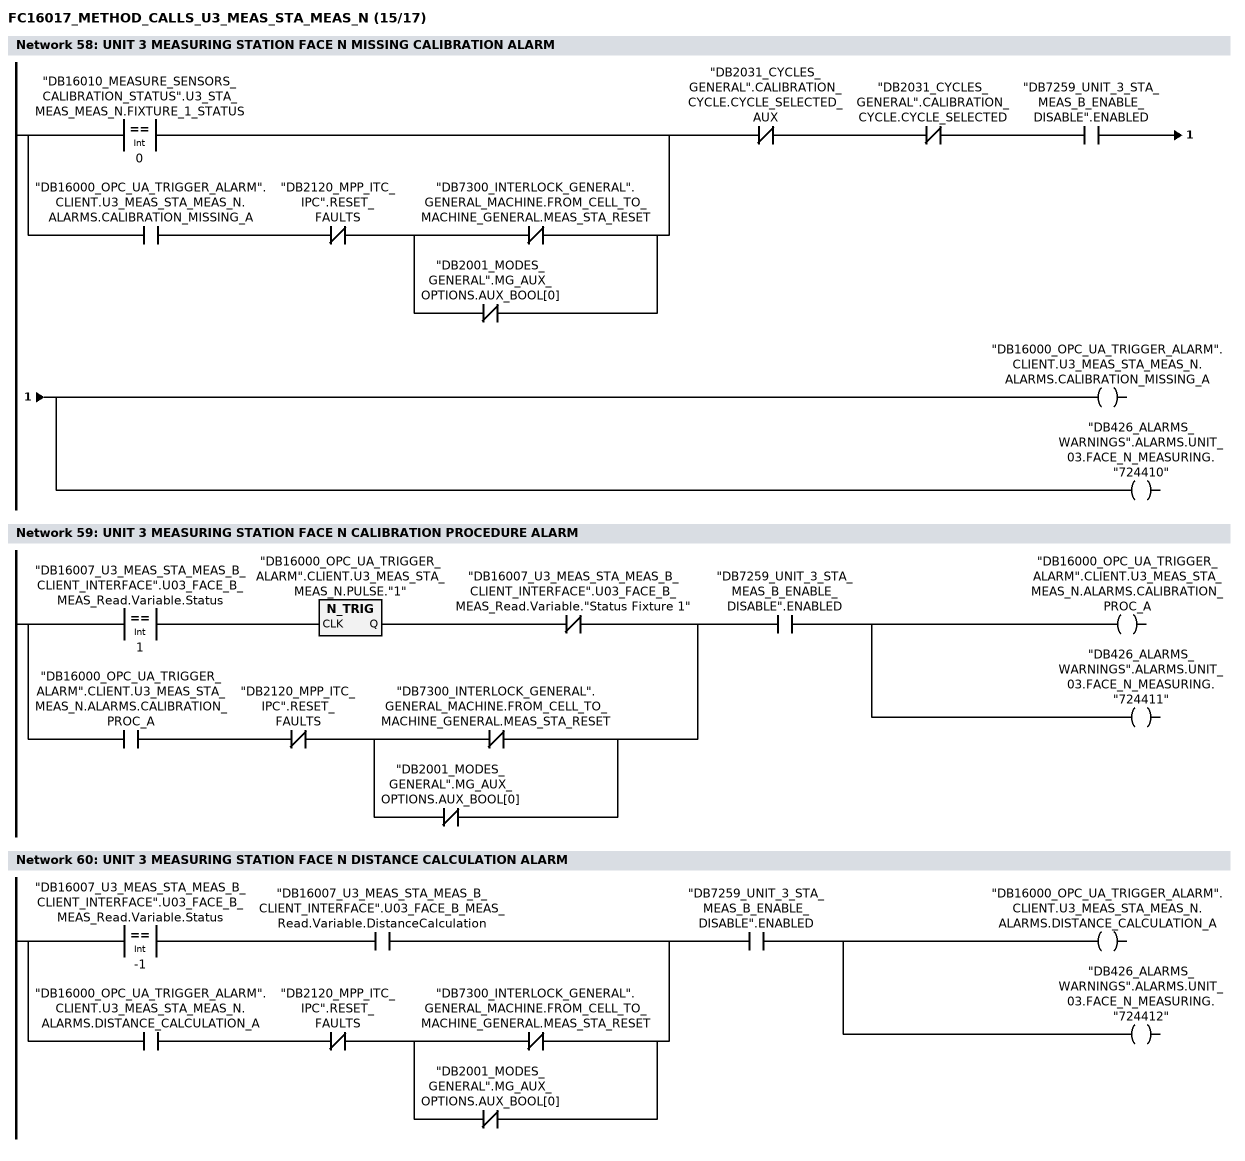
   RUNG wire#powerrail
      { S7_Templates := "SrcType := Int" } EQ_Contact(in1 := "DB16010_MEASURE_SENSORS_CALIBRATION_STATUS".U3_STA_MEAS_MEAS_N.FIXTURE_1_STATUS, in2 := 0)
      wire#w1
      I_Contact( "DB2031_CYCLES_GENERAL".CALIBRATION_CYCLE.CYCLE_SELECTED_AUX )
      I_Contact( "DB2031_CYCLES_GENERAL".CALIBRATION_CYCLE.CYCLE_SELECTED )
      Contact( "DB7259_UNIT_3_STA_MEAS_B_ENABLE_DISABLE".ENABLED )
      wire#w3
      Coil( "DB16000_OPC_UA_TRIGGER_ALARM".CLIENT.U3_MEAS_STA_MEAS_N.ALARMS.CALIBRATION_MISSING_A )
   END_RUNG
   RUNG wire#powerrail
      Contact( "DB16000_OPC_UA_TRIGGER_ALARM".CLIENT.U3_MEAS_STA_MEAS_N.ALARMS.CALIBRATION_MISSING_A )
      I_Contact( "DB2120_MPP_ITC_IPC".RESET_FAULTS )
      wire#w2
      I_Contact( "DB7300_INTERLOCK_GENERAL".GENERAL_MACHINE.FROM_CELL_TO_MACHINE_GENERAL.MEAS_STA_RESET )
   END_RUNG wire#w1
   RUNG wire#w2
      I_Contact( "DB2001_MODES_GENERAL".MG_AUX_OPTIONS.AUX_BOOL[0] )
   END_RUNG wire#w1
   RUNG wire#w3
      Coil( "DB426_ALARMS_WARNINGS".ALARMS.UNIT_03.FACE_N_MEASURING."724410" )
   END_RUNG
   // the same network as SCL:
   "DB16000_OPC_UA_TRIGGER_ALARM".CLIENT.U3_MEAS_STA_MEAS_N.ALARMS.CALIBRATION_MISSING_A := (("DB16010_MEASURE_SENSORS_CALIBRATION_STATUS".U3_STA_MEAS_MEAS_N.FIXTURE_1_STATUS = 0) OR ("DB16000_OPC_UA_TRIGGER_ALARM".CLIENT.U3_MEAS_STA_MEAS_N.ALARMS.CALIBRATION_MISSING_A AND NOT "DB2120_MPP_ITC_IPC".RESET_FAULTS AND (NOT "DB7300_INTERLOCK_GENERAL".GENERAL_MACHINE.FROM_CELL_TO_MACHINE_GENERAL.MEAS_STA_RESET OR NOT "DB2001_MODES_GENERAL".MG_AUX_OPTIONS.AUX_BOOL[0]))) AND NOT "DB2031_CYCLES_GENERAL".CALIBRATION_CYCLE.CYCLE_SELECTED_AUX AND NOT "DB2031_CYCLES_GENERAL".CALIBRATION_CYCLE.CYCLE_SELECTED AND "DB7259_UNIT_3_STA_MEAS_B_ENABLE_DISABLE".ENABLED;
   "DB426_ALARMS_WARNINGS".ALARMS.UNIT_03.FACE_N_MEASURING."724410" := "DB16000_OPC_UA_TRIGGER_ALARM".CLIENT.U3_MEAS_STA_MEAS_N.ALARMS.CALIBRATION_MISSING_A;
END_REGION

REGION Network 59: UNIT 3 MEASURING STATION FACE N CALIBRATION PROCEDURE ALARM
   RUNG wire#powerrail
      { S7_Templates := "SrcType := Int" } EQ_Contact(in1 := "DB16007_U3_MEAS_STA_MEAS_B_CLIENT_INTERFACE".U03_FACE_B_MEAS_Read.Variable.Status, in2 := 1)
      N_Trig( "DB16000_OPC_UA_TRIGGER_ALARM".CLIENT.U3_MEAS_STA_MEAS_N.PULSE."1" )
      I_Contact( "DB16007_U3_MEAS_STA_MEAS_B_CLIENT_INTERFACE".U03_FACE_B_MEAS_Read.Variable."Status Fixture 1" )
      wire#w1
      Contact( "DB7259_UNIT_3_STA_MEAS_B_ENABLE_DISABLE".ENABLED )
      wire#w3
      Coil( "DB16000_OPC_UA_TRIGGER_ALARM".CLIENT.U3_MEAS_STA_MEAS_N.ALARMS.CALIBRATION_PROC_A )
   END_RUNG
   RUNG wire#powerrail
      Contact( "DB16000_OPC_UA_TRIGGER_ALARM".CLIENT.U3_MEAS_STA_MEAS_N.ALARMS.CALIBRATION_PROC_A )
      I_Contact( "DB2120_MPP_ITC_IPC".RESET_FAULTS )
      wire#w2
      I_Contact( "DB7300_INTERLOCK_GENERAL".GENERAL_MACHINE.FROM_CELL_TO_MACHINE_GENERAL.MEAS_STA_RESET )
   END_RUNG wire#w1
   RUNG wire#w2
      I_Contact( "DB2001_MODES_GENERAL".MG_AUX_OPTIONS.AUX_BOOL[0] )
   END_RUNG wire#w1
   RUNG wire#w3
      Coil( "DB426_ALARMS_WARNINGS".ALARMS.UNIT_03.FACE_N_MEASURING."724411" )
   END_RUNG
   // the same network as SCL:
   #_w1 := "DB16007_U3_MEAS_STA_MEAS_B_CLIENT_INTERFACE".U03_FACE_B_MEAS_Read.Variable.Status = 1;
   #_w2 := NOT #_w1 AND "DB16000_OPC_UA_TRIGGER_ALARM".CLIENT.U3_MEAS_STA_MEAS_N.PULSE."1";   // falling edge
   "DB16000_OPC_UA_TRIGGER_ALARM".CLIENT.U3_MEAS_STA_MEAS_N.PULSE."1" := #_w1;
   "DB16000_OPC_UA_TRIGGER_ALARM".CLIENT.U3_MEAS_STA_MEAS_N.ALARMS.CALIBRATION_PROC_A := ((#_w2 AND NOT "DB16007_U3_MEAS_STA_MEAS_B_CLIENT_INTERFACE".U03_FACE_B_MEAS_Read.Variable."Status Fixture 1") OR ("DB16000_OPC_UA_TRIGGER_ALARM".CLIENT.U3_MEAS_STA_MEAS_N.ALARMS.CALIBRATION_PROC_A AND NOT "DB2120_MPP_ITC_IPC".RESET_FAULTS AND (NOT "DB7300_INTERLOCK_GENERAL".GENERAL_MACHINE.FROM_CELL_TO_MACHINE_GENERAL.MEAS_STA_RESET OR NOT "DB2001_MODES_GENERAL".MG_AUX_OPTIONS.AUX_BOOL[0]))) AND "DB7259_UNIT_3_STA_MEAS_B_ENABLE_DISABLE".ENABLED;
   "DB426_ALARMS_WARNINGS".ALARMS.UNIT_03.FACE_N_MEASURING."724411" := "DB16000_OPC_UA_TRIGGER_ALARM".CLIENT.U3_MEAS_STA_MEAS_N.ALARMS.CALIBRATION_PROC_A;
END_REGION

REGION Network 60: UNIT 3 MEASURING STATION FACE N DISTANCE CALCULATION ALARM
   RUNG wire#powerrail
      { S7_Templates := "SrcType := Int" } EQ_Contact(in1 := "DB16007_U3_MEAS_STA_MEAS_B_CLIENT_INTERFACE".U03_FACE_B_MEAS_Read.Variable.Status, in2 := -1)
      Contact( "DB16007_U3_MEAS_STA_MEAS_B_CLIENT_INTERFACE".U03_FACE_B_MEAS_Read.Variable.DistanceCalculation )
      wire#w1
      Contact( "DB7259_UNIT_3_STA_MEAS_B_ENABLE_DISABLE".ENABLED )
      wire#w3
      Coil( "DB16000_OPC_UA_TRIGGER_ALARM".CLIENT.U3_MEAS_STA_MEAS_N.ALARMS.DISTANCE_CALCULATION_A )
   END_RUNG
   RUNG wire#powerrail
      Contact( "DB16000_OPC_UA_TRIGGER_ALARM".CLIENT.U3_MEAS_STA_MEAS_N.ALARMS.DISTANCE_CALCULATION_A )
      I_Contact( "DB2120_MPP_ITC_IPC".RESET_FAULTS )
      wire#w2
      I_Contact( "DB7300_INTERLOCK_GENERAL".GENERAL_MACHINE.FROM_CELL_TO_MACHINE_GENERAL.MEAS_STA_RESET )
   END_RUNG wire#w1
   RUNG wire#w2
      I_Contact( "DB2001_MODES_GENERAL".MG_AUX_OPTIONS.AUX_BOOL[0] )
   END_RUNG wire#w1
   RUNG wire#w3
      Coil( "DB426_ALARMS_WARNINGS".ALARMS.UNIT_03.FACE_N_MEASURING."724412" )
   END_RUNG
   // the same network as SCL:
   "DB16000_OPC_UA_TRIGGER_ALARM".CLIENT.U3_MEAS_STA_MEAS_N.ALARMS.DISTANCE_CALCULATION_A := ((("DB16007_U3_MEAS_STA_MEAS_B_CLIENT_INTERFACE".U03_FACE_B_MEAS_Read.Variable.Status = (-1)) AND "DB16007_U3_MEAS_STA_MEAS_B_CLIENT_INTERFACE".U03_FACE_B_MEAS_Read.Variable.DistanceCalculation) OR ("DB16000_OPC_UA_TRIGGER_ALARM".CLIENT.U3_MEAS_STA_MEAS_N.ALARMS.DISTANCE_CALCULATION_A AND NOT "DB2120_MPP_ITC_IPC".RESET_FAULTS AND (NOT "DB7300_INTERLOCK_GENERAL".GENERAL_MACHINE.FROM_CELL_TO_MACHINE_GENERAL.MEAS_STA_RESET OR NOT "DB2001_MODES_GENERAL".MG_AUX_OPTIONS.AUX_BOOL[0]))) AND "DB7259_UNIT_3_STA_MEAS_B_ENABLE_DISABLE".ENABLED;
   "DB426_ALARMS_WARNINGS".ALARMS.UNIT_03.FACE_N_MEASURING."724412" := "DB16000_OPC_UA_TRIGGER_ALARM".CLIENT.U3_MEAS_STA_MEAS_N.ALARMS.DISTANCE_CALCULATION_A;
END_REGION

REGION Network 61: UNIT 3 MEASURING STATION FACE N DATABASE CONNECTION ALARM
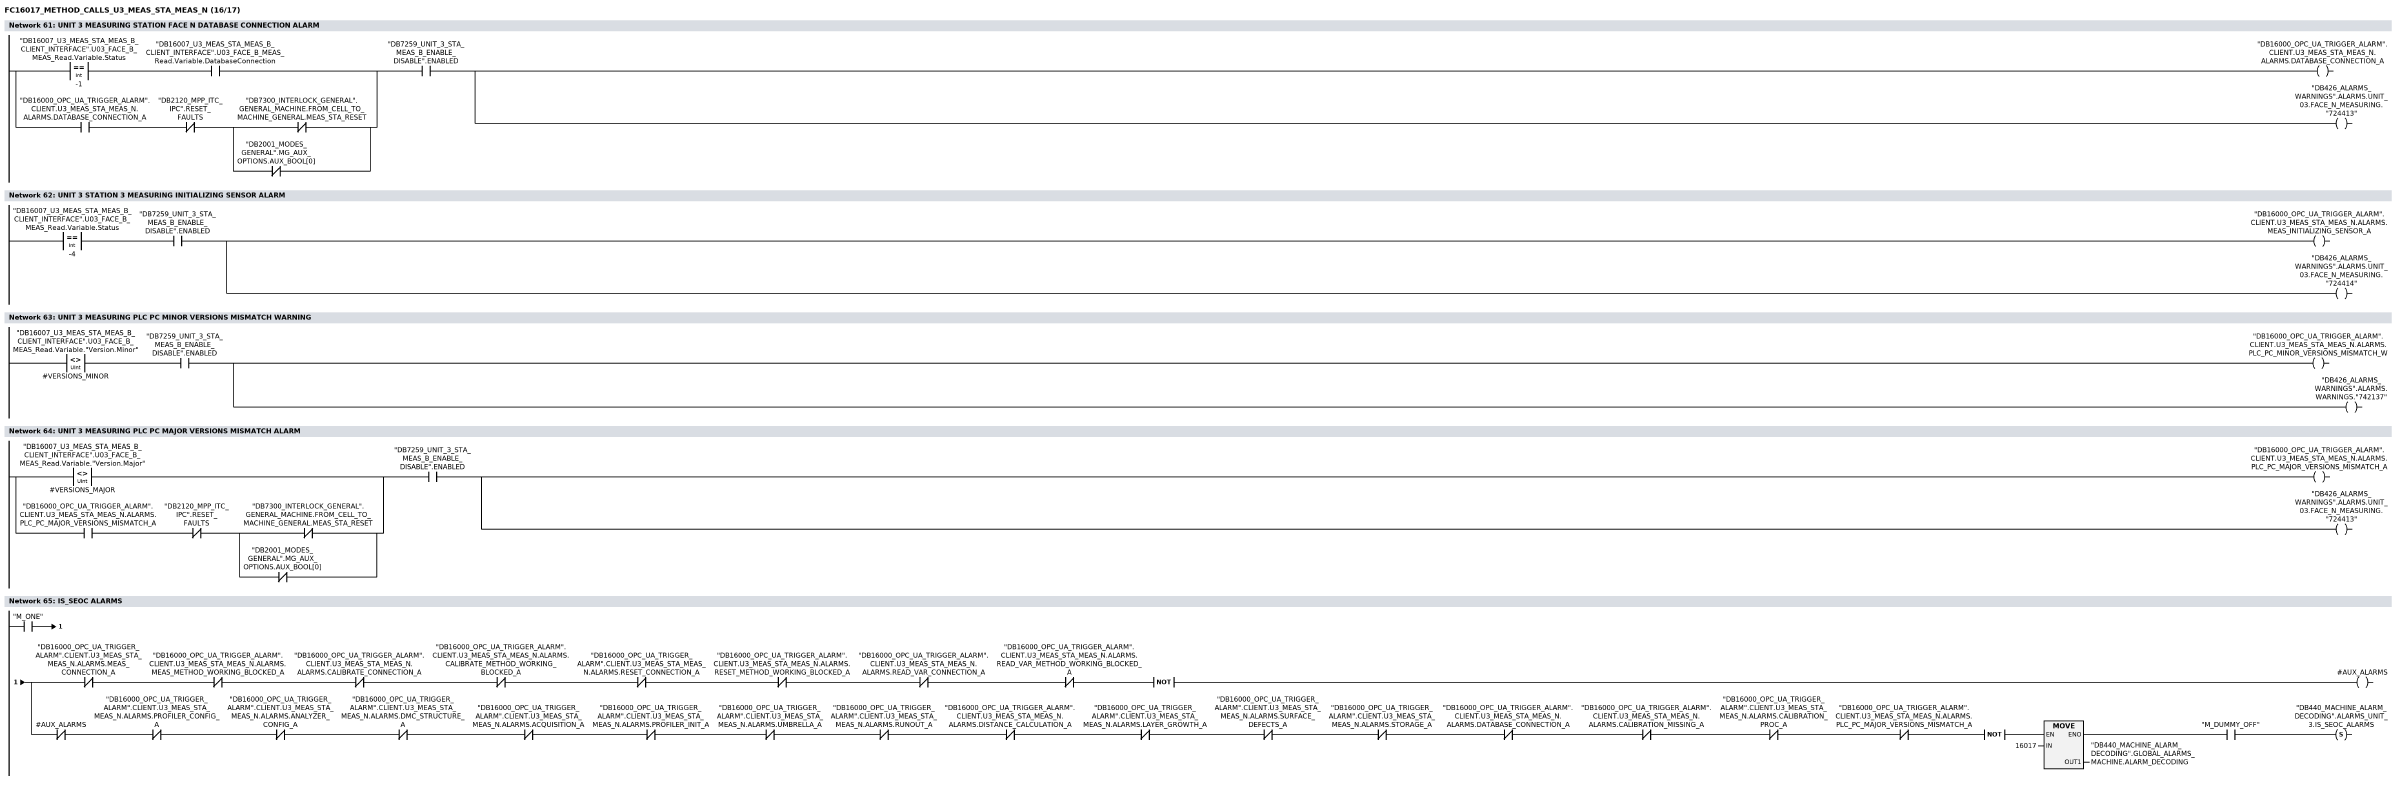
   RUNG wire#powerrail
      { S7_Templates := "SrcType := Int" } EQ_Contact(in1 := "DB16007_U3_MEAS_STA_MEAS_B_CLIENT_INTERFACE".U03_FACE_B_MEAS_Read.Variable.Status, in2 := -1)
      Contact( "DB16007_U3_MEAS_STA_MEAS_B_CLIENT_INTERFACE".U03_FACE_B_MEAS_Read.Variable.DatabaseConnection )
      wire#w1
      Contact( "DB7259_UNIT_3_STA_MEAS_B_ENABLE_DISABLE".ENABLED )
      wire#w3
      Coil( "DB16000_OPC_UA_TRIGGER_ALARM".CLIENT.U3_MEAS_STA_MEAS_N.ALARMS.DATABASE_CONNECTION_A )
   END_RUNG
   RUNG wire#powerrail
      Contact( "DB16000_OPC_UA_TRIGGER_ALARM".CLIENT.U3_MEAS_STA_MEAS_N.ALARMS.DATABASE_CONNECTION_A )
      I_Contact( "DB2120_MPP_ITC_IPC".RESET_FAULTS )
      wire#w2
      I_Contact( "DB7300_INTERLOCK_GENERAL".GENERAL_MACHINE.FROM_CELL_TO_MACHINE_GENERAL.MEAS_STA_RESET )
   END_RUNG wire#w1
   RUNG wire#w2
      I_Contact( "DB2001_MODES_GENERAL".MG_AUX_OPTIONS.AUX_BOOL[0] )
   END_RUNG wire#w1
   RUNG wire#w3
      Coil( "DB426_ALARMS_WARNINGS".ALARMS.UNIT_03.FACE_N_MEASURING."724413" )
   END_RUNG
   // the same network as SCL:
   "DB16000_OPC_UA_TRIGGER_ALARM".CLIENT.U3_MEAS_STA_MEAS_N.ALARMS.DATABASE_CONNECTION_A := ((("DB16007_U3_MEAS_STA_MEAS_B_CLIENT_INTERFACE".U03_FACE_B_MEAS_Read.Variable.Status = (-1)) AND "DB16007_U3_MEAS_STA_MEAS_B_CLIENT_INTERFACE".U03_FACE_B_MEAS_Read.Variable.DatabaseConnection) OR ("DB16000_OPC_UA_TRIGGER_ALARM".CLIENT.U3_MEAS_STA_MEAS_N.ALARMS.DATABASE_CONNECTION_A AND NOT "DB2120_MPP_ITC_IPC".RESET_FAULTS AND (NOT "DB7300_INTERLOCK_GENERAL".GENERAL_MACHINE.FROM_CELL_TO_MACHINE_GENERAL.MEAS_STA_RESET OR NOT "DB2001_MODES_GENERAL".MG_AUX_OPTIONS.AUX_BOOL[0]))) AND "DB7259_UNIT_3_STA_MEAS_B_ENABLE_DISABLE".ENABLED;
   "DB426_ALARMS_WARNINGS".ALARMS.UNIT_03.FACE_N_MEASURING."724413" := "DB16000_OPC_UA_TRIGGER_ALARM".CLIENT.U3_MEAS_STA_MEAS_N.ALARMS.DATABASE_CONNECTION_A;
END_REGION

REGION Network 62: UNIT 3 STATION 3 MEASURING INITIALIZING SENSOR ALARM
   RUNG wire#powerrail
      { S7_Templates := "SrcType := Int" } EQ_Contact(in1 := "DB16007_U3_MEAS_STA_MEAS_B_CLIENT_INTERFACE".U03_FACE_B_MEAS_Read.Variable.Status, in2 := -4)
      Contact( "DB7259_UNIT_3_STA_MEAS_B_ENABLE_DISABLE".ENABLED )
      wire#w1
      Coil( "DB16000_OPC_UA_TRIGGER_ALARM".CLIENT.U3_MEAS_STA_MEAS_N.ALARMS.MEAS_INITIALIZING_SENSOR_A )
   END_RUNG
   RUNG wire#w1
      Coil( "DB426_ALARMS_WARNINGS".ALARMS.UNIT_03.FACE_N_MEASURING."724414" )
   END_RUNG
   // the same network as SCL:
   "DB16000_OPC_UA_TRIGGER_ALARM".CLIENT.U3_MEAS_STA_MEAS_N.ALARMS.MEAS_INITIALIZING_SENSOR_A := ("DB16007_U3_MEAS_STA_MEAS_B_CLIENT_INTERFACE".U03_FACE_B_MEAS_Read.Variable.Status = (-4)) AND "DB7259_UNIT_3_STA_MEAS_B_ENABLE_DISABLE".ENABLED;
   "DB426_ALARMS_WARNINGS".ALARMS.UNIT_03.FACE_N_MEASURING."724414" := "DB16000_OPC_UA_TRIGGER_ALARM".CLIENT.U3_MEAS_STA_MEAS_N.ALARMS.MEAS_INITIALIZING_SENSOR_A;
END_REGION

